Omron CX-Programmer project 新工程 (CX-Programmer 9.61)

# PLC ND自动入壳机: CJ2H CPU65-EIP
I/O table (CPU CJ2H-CPU65-EIP): rack 0 slot 0 CJ1W-ETN21(ETN21Mode); rack 0 slot 1 CJ1W-SCU21-V1; rack 0 slot 2 CJ1W-NC433; rack 0 slot 3 CJ1W-NC433; rack 0 slot 4 CJ1W-NC433; rack 0 slot 5 CJ1W-NC433; rack 0 slot 6 CJ1W-NC433; rack 0 slot 7 CJ1W-AD041-V1; rack 0 slot 11 CJ2B-EIP21; rack 1 slot 0 CJ1W-ID261; rack 1 slot 1 CJ1W-ID261; rack 1 slot 2 CJ1W-ID261; rack 1 slot 3 CJ1W-ID231; rack 1 slot 4 CJ1W-ID261; rack 1 slot 5 CJ1W-ID231; rack 1 slot 6 CJ1W-OD261; rack 1 slot 7 CJ1W-OD261; rack 1 slot 8 CJ1W-OD231; rack 1 slot 9 CJ1W-OD261

## Global symbols (name address type ; comment)
0.00 BOOL  ; RK_02 电芯进料机械手夹爪气缸夹紧位
0.01 BOOL  ; RK_02 电芯进料机械手夹爪气缸张开位
0.02 BOOL  ; RK_02 电芯进料机械手#1压紧气缸松开位
0.03 BOOL  ; RK_02 电芯进料机械手#2压紧气缸松开位
0.04 BOOL  ; RK_03 电芯上料机械手夹爪气缸夹紧位
0.05 BOOL  ; RK_03 电芯上料机械手夹爪气缸张开位
0.06 BOOL  ; RK_03 电芯上料机械手#1压紧气缸松开位
0.07 BOOL  ; RK_03 电芯上料机械手#2压紧气缸松开位
0.08 BOOL  ; RK_03 电芯上料升降气缸下降位
0.09 BOOL  ; RK_03 电芯上料升降气缸上升位
0.10 BOOL  ; RK_04 电芯除尘伸缩气缸缩回位
0.11 BOOL  ; RK_04 电芯除尘伸缩气缸伸出位
0.12 BOOL  ; RK_05 #1入壳滚轮夹紧气缸夹紧位
0.13 BOOL  ; RK_05 #1入壳滚轮夹紧气缸松开位
0.14 BOOL  ; RK_05 #1入壳铝壳定位平台伸缩气缸缩回位
0.15 BOOL  ; RK_05 #1入壳铝壳定位平台伸缩气缸伸出位
1000.00 BOOL  ; RK_01 U0_X 电芯来料Y轴待料位设定确认
1000.01 BOOL  ; RK_01 U0_X 电芯来料Y轴上料位设定确认
1000.02 BOOL  ; RK_01 U0_X 电芯来料Y轴扫码位设定确认
1000.03 BOOL  ; RK_01 U0_X 电芯来料Y轴下料位设定确认
1001.00 BOOL  ; RK_02 U0_Y 电芯进料X轴待料位设定确认
1001.01 BOOL  ; RK_02 U0_Y 电芯进料X轴取料位设定确认
1001.02 BOOL  ; RK_02 U0_Y 电芯进料X轴扫码OK放料位设定确认
1001.03 BOOL  ; RK_02 U0_Y 电芯进料X轴扫码NG放料位设定确认
1002.00 BOOL  ; RK_02 U0_Z 电芯进料Z轴待料位（扫码）设定确认
1002.01 BOOL  ; RK_02 U0_Z 电芯进料Z轴取料位设定确认
1002.02 BOOL  ; RK_02 U0_Z 电芯进料Z轴扫码OK放料位设定确认
1002.03 BOOL  ; RK_02 U0_Z 电芯进料Z轴扫码NG放料位设定确认
1002.04 BOOL  ; RK_02 U0_Z 电芯进料Z轴扫码位设定确认
1003.00 BOOL  ; RK_03 U0_U 电芯上料X轴待料位设定确认
1003.01 BOOL  ; RK_03 U0_U 电芯上料X轴取料位设定确认
1003.02 BOOL  ; RK_03 U0_U 电芯上料X轴#1入壳放料位设定确认
1003.03 BOOL  ; RK_03 U0_U 电芯上料X轴#2入壳放料位设定确认
1004.00 BOOL  ; RK_05 U2_X #1入壳Y轴待料位设定确认
1004.01 BOOL  ; RK_05 U2_X #1入壳Y轴滚轮压紧位设定确认
1004.02 BOOL  ; RK_05 U2_X #1入壳Y轴滚轮松开位设定确认
1004.03 BOOL  ; RK_05 U2_X #1入壳Y轴入壳位设定确认
1004.04 BOOL  ; RK_05 U2_X #1入壳Y轴电芯定位夹爪松开位设定确认
1005.00 BOOL  ; RK_05 U2_Y #2入壳Y轴待料位设定确认
1005.01 BOOL  ; RK_05 U2_Y #2入壳Y轴滚轮压紧位设定确认
1005.02 BOOL  ; RK_05 U2_Y #2入壳Y轴滚轮松开位设定确认
1005.03 BOOL  ; RK_05 U2_Y #2入壳Y轴入壳位设定确认
1005.04 BOOL  ; RK_05 U2_Y #2入壳Y轴电芯定位夹爪松开位设定确认
1006.00 BOOL  ; RK_12 U4_X 预焊上下料X轴待料位设定确认
1006.01 BOOL  ; RK_12 U4_X 预焊上下料X轴除尘取料位设定确认
1006.02 BOOL  ; RK_12 U4_X 预焊上下料X轴#1移载放料位设定确认
1006.03 BOOL  ; RK_12 U4_X 预焊上下料X轴#2移载放料位设定确认
1006.04 BOOL  ; RK_12 U4_X 预焊上下料X轴#1移载取料位设定确认
1006.05 BOOL  ; RK_12 U4_X 预焊上下料X轴#2移载取料位设定确认
1006.06 BOOL  ; RK_12 U4_X 预焊上下料X轴OK放料位设定确认
1006.07 BOOL  ; RK_12 U4_X 预焊上下料X轴#1NG放料位设定确认
1006.08 BOOL  ; RK_12 U4_X 预焊上下料X轴#2NG放料位设定确认
1007.00 BOOL  ; RK_12 U4_Y 预焊上料Z轴待料位设定确认
1007.01 BOOL  ; RK_12 U4_Y 预焊上料Z轴除尘取料位设定确认
1007.02 BOOL  ; RK_12 U4_Y 预焊上料Z轴#1移载放料位设定确认
1007.03 BOOL  ; RK_12 U4_Y 预焊上料Z轴#2移载放料位设定确认
1008.00 BOOL  ; RK_12 U4_Z 预焊下料Z轴待料位设定确认
1008.01 BOOL  ; RK_12 U4_Z 预焊下料Z轴#1移载取料位设定确认
1008.02 BOOL  ; RK_12 U4_Z 预焊下料Z轴#2移载取料位设定确认
1008.03 BOOL  ; RK_12 U4_Z 预焊下料Z轴OK放料位设定确认
1008.04 BOOL  ; RK_12 U4_Z 预焊下料Z轴#1NG放料位设定确认
1008.05 BOOL  ; RK_12 U4_Z 预焊下料Z轴#2NG放料位设定确认
1009.00 BOOL  ; RK_13 U4_U #1移载Y轴待料位设定确认
1009.01 BOOL  ; RK_13 U4_U #1移载Y轴取放料位设定确认
1009.02 BOOL  ; RK_13 U4_U #1移载Y轴压装位设定确认
1009.03 BOOL  ; RK_13 U4_U #1移载Y轴#1轮廓检测位设定确认
1009.04 BOOL  ; RK_13 U4_U #1移载Y轴#2轮廓检测位设定确认
1009.05 BOOL  ; RK_13 U4_U #1移载Y轴激光焊接位设定确认
100.00 BOOL  ; RK_02 电芯进料机械手夹爪气缸夹紧
100.01 BOOL  ; RK_02 电芯进料机械手夹爪气缸张开
100.02 BOOL  ; RK_02 电芯进料机械手压紧气缸伸出
100.03 BOOL  ; RK_02 电芯进料机械手压紧气缸缩回
100.04 BOOL  ; RK_03 电芯上料机械手夹爪气缸夹紧
100.05 BOOL  ; RK_03 电芯上料机械手夹爪气缸张开
100.06 BOOL  ; RK_03 电芯上料机械手压紧气缸伸出
100.07 BOOL  ; RK_03 电芯上料机械手压紧气缸缩回
100.08 BOOL  ; RK_03 电芯上料升降气缸下降
100.09 BOOL  ; RK_03 电芯上料升降气缸上升
100.10 BOOL  ; RK_04 电芯除尘伸缩气缸缩回
100.11 BOOL  ; RK_04 电芯除尘伸缩气缸伸出
100.12 BOOL  ; RK_05 #1入壳滚轮夹紧气缸伸出
100.13 BOOL  ; RK_05 #1入壳滚轮夹紧气缸缩回
100.14 BOOL  ; RK_05 #1入壳铝壳定位平台伸缩气缸缩回
100.15 BOOL  ; RK_05 #1入壳铝壳定位平台伸缩气缸伸出
1010.00 BOOL  ; RK_13 U6_X #2移载Y轴待料位设定确认
1010.01 BOOL  ; RK_13 U6_X #2移载Y轴取放料位设定确认
1010.02 BOOL  ; RK_13 U6_X #2移载Y轴压装位设定确认
1010.03 BOOL  ; RK_13 U6_X #2移载Y轴#1轮廓检测位设定确认
1010.04 BOOL  ; RK_13 U6_X #2移载Y轴#2轮廓检测位设定确认
1010.05 BOOL  ; RK_13 U6_X #2移载Y轴激光焊接位设定确认
1011.00 BOOL  ; RK_16 U6_Y 激光焊接X轴待机位设定确认
1011.01 BOOL  ; RK_16 U6_Y 激光焊接X轴#1移载焊接位设定确认
1011.02 BOOL  ; RK_16 U6_Y 激光焊接X轴#2移载焊接位设定确认
1012.00 BOOL  ; RK_16 U6_Z 激光焊接Z轴待机位设定确认
1012.01 BOOL  ; RK_16 U6_Z 激光焊接Z轴#1移载焊接位设定确认
1012.02 BOOL  ; RK_16 U6_Z 激光焊接Z轴#2移载焊接位设定确认
1013.00 BOOL  ; RK_06 U8_X 电池上下料X轴待机位设定确认
1013.01 BOOL  ; RK_06 U8_X 电池上下料X轴铝壳除尘取料位设定确认
1013.02 BOOL  ; RK_06 U8_X 电池上下料X轴#1入壳放料位设定确认
1013.03 BOOL  ; RK_06 U8_X 电池上下料X轴#2入壳放料位设定确认
1013.04 BOOL  ; RK_06 U8_X 电池上下料X轴#1入壳取料位设定确认
1013.05 BOOL  ; RK_06 U8_X 电池上下料X轴#2入壳取料位设定确认
1013.06 BOOL  ; RK_06 U8_X 电池上下料X轴#1Hipot检测放料位设定确认
1013.07 BOOL  ; RK_06 U8_X 电池上下料X轴#2Hipot检测放料位设定确认
1014.00 BOOL  ; RK_07 U8_Y 铝壳进料X轴等待位设定确认
1014.01 BOOL  ; RK_07 U8_Y 铝壳进料X轴取料位设定确认
1014.02 BOOL  ; RK_07 U8_Y 铝壳进料X轴放料位设定确认
1015.00 BOOL  ; RK_07 U8_Z 铝壳上料移载Y轴待料位设定确认
1015.01 BOOL  ; RK_07 U8_Z 铝壳上料移载Y轴#1铝壳上料位设定确认
1015.02 BOOL  ; RK_07 U8_Z 铝壳上料移载Y轴#2铝壳上料位设定确认
1015.03 BOOL  ; RK_07 U8_Z 铝壳上料移载Y轴#3铝壳托盘下料位设定确认
1015.04 BOOL  ; RK_07 U8_Z 铝壳上料移载Y轴铝壳取料位设定确认
1016.00 BOOL  ; RK_10 U8_U 电池除尘上料X轴待料位设定确认
1016.01 BOOL  ; RK_10 U8_U 电池除尘上料X轴#1Hipot检测取料位设定确认
1016.02 BOOL  ; RK_10 U8_U 电池除尘上料X轴#2Hipot检测取料位设定确认
1016.03 BOOL  ; RK_10 U8_U 电池除尘上料X轴Hipot OK放料位设定确认
1016.04 BOOL  ; RK_10 U8_U 电池除尘上料X轴Hipot NG放料位设定确认
101.00 BOOL  ; RK_05 #1入壳铝壳定位平台升降气缸上升
101.01 BOOL  ; RK_05 #1入壳铝壳定位平台升降气缸下降
101.02 BOOL  ; RK_05 #1入壳铝壳定位伸缩气缸缩回
101.03 BOOL  ; RK_05 #1入壳铝壳定位伸缩气缸伸出
101.04 BOOL  ; RK_05 #1入壳铝壳定位夹爪气缸夹紧
101.05 BOOL  ; RK_05 #1入壳铝壳定位夹爪气缸张开
101.06 BOOL  ; RK_05 #2入壳滚轮夹紧气缸伸出
101.07 BOOL  ; RK_05 #2入壳滚轮夹紧气缸缩回
101.08 BOOL  ; RK_05 #2入壳铝壳定位平台伸缩气缸缩回
101.09 BOOL  ; RK_05 #2入壳铝壳定位平台伸缩气缸伸出
101.10 BOOL  ; RK_05 #2入壳铝壳定位平台升降气缸上升
101.11 BOOL  ; RK_05 #2入壳铝壳定位平台升降气缸下降
101.12 BOOL  ; RK_05 #2入壳铝壳定位伸缩气缸缩回
101.13 BOOL  ; RK_05 #2入壳铝壳定位伸缩气缸伸出
101.14 BOOL  ; RK_05 #2入壳铝壳定位夹爪气缸夹紧
101.15 BOOL  ; RK_05 #2入壳铝壳定位夹爪气缸张开
102.00 BOOL  ; RK_01 U0_X 电芯来料Y轴报警复位
102.01 BOOL  ; RK_01 U0_X 电芯来料Y轴使能
102.02 BOOL  ; RK_02 U0_Y 电芯进料X轴报警复位
102.03 BOOL  ; RK_02 U0_Y 电芯进料X轴使能
102.04 BOOL  ; RK_02 U0_Z 电芯进料Z轴报警复位
102.05 BOOL  ; RK_02 U0_Z 电芯进料Z轴使能
102.06 BOOL  ; RK_03 U0_U 电芯上料X轴报警复位
102.07 BOOL  ; RK_03 U0_U 电芯上料X轴使能
102.08 BOOL  ; RK_05 U2_X #1入壳Y轴报警复位
102.09 BOOL  ; RK_05 U2_X #1入壳Y轴使能
102.10 BOOL  ; RK_05 U2_Y #2入壳Y轴报警复位
102.11 BOOL  ; RK_05 U2_Y #2入壳Y轴使能
102.12 BOOL  ; RK_02 电芯进料Z轴刹车使能
102.13 BOOL  ; RK_05 #1入壳定位陶瓷棒夹紧气缸伸出
102.14 BOOL  ; RK_05 #1入壳定位陶瓷棒夹紧气缸缩回
102.15 BOOL  ; RK_05 #2入壳定位陶瓷棒夹紧气缸伸出
103.00 BOOL  ; RK_05 #2入壳定位陶瓷棒夹紧气缸缩回
103.01 BOOL  ; RK_04 电芯除尘吹气阀开
103.02 BOOL  ; RK_02 扫码NG拉带启动
103.03 BOOL  ; RK_05 #1入壳吸盘立真空
103.04 BOOL  ; RK_05 #2入壳吸盘立真空
103.05 BOOL  ; RK_05 #1入壳吸盘伸缩气缸伸出
103.06 BOOL  ; RK_05 #1入壳吸盘伸缩气缸缩回
103.07 BOOL  ; RK_05 #2入壳吸盘伸缩气缸伸出
103.08 BOOL  ; RK_05 #2入壳吸盘伸缩气缸缩回
103.09 BOOL  ; 前端设备对接输出信号（公共）
103.10 BOOL  ; 后端设备对接输出信号（公共）
103.11 BOOL  ; RK_05 #1入壳电芯定位夹爪气缸伸出
103.12 BOOL  ; RK_05 #1入壳电芯定位夹爪气缸缩回
103.13 BOOL  ; RK_05 #2入壳电芯定位夹爪气缸伸出
103.14 BOOL  ; RK_05 #2入壳电芯定位夹爪气缸缩回
103.15 BOOL  ; 0
104.00 BOOL  ; 0
104.01 BOOL  ; 0
104.02 BOOL  ; 0
104.03 BOOL  ; 0
104.04 BOOL  ; 0
104.05 BOOL  ; 0
104.06 BOOL  ; 0
104.07 BOOL  ; 0
104.08 BOOL  ; 0
104.09 BOOL  ; 0
104.10 BOOL  ; 0
104.11 BOOL  ; 0
104.12 BOOL  ; 0
104.13 BOOL  ; 0
104.14 BOOL  ; 0
104.15 BOOL  ; 0
105.00 BOOL  ; 0
105.01 BOOL  ; 0
105.02 BOOL  ; 0
105.03 BOOL  ; 0
105.04 BOOL  ; 0
105.05 BOOL  ; 0
105.06 BOOL  ; 0
105.07 BOOL  ; 0
105.08 BOOL  ; 0
105.09 BOOL  ; 0
105.10 BOOL  ; 0
105.11 BOOL  ; 0
105.12 BOOL  ; 0
105.13 BOOL  ; 0
105.14 BOOL  ; 0
105.15 BOOL  ; 0
106.00 BOOL  ; 0
106.01 BOOL  ; 0
106.02 BOOL  ; 0
106.03 BOOL  ; 0
106.04 BOOL  ; 0
106.05 BOOL  ; 0
106.06 BOOL  ; 0
106.07 BOOL  ; 0
106.08 BOOL  ; 0
106.09 BOOL  ; 0
106.10 BOOL  ; 0
106.11 BOOL  ; 0
106.12 BOOL  ; 0
106.13 BOOL  ; 0
106.14 BOOL  ; 0
106.15 BOOL  ; 0
107.00 BOOL  ; 0
107.01 BOOL  ; 0
107.02 BOOL  ; 0
107.03 BOOL  ; 0
107.04 BOOL  ; 0
107.05 BOOL  ; 0
107.06 BOOL  ; 0
107.07 BOOL  ; 0
107.08 BOOL  ; 0
107.09 BOOL  ; 0
107.10 BOOL  ; 0
107.11 BOOL  ; 0
107.12 BOOL  ; 0
107.13 BOOL  ; 0
107.14 BOOL  ; 0
107.15 BOOL  ; 0
108.00 BOOL  ; RK_11 电池除尘旋转伸缩气缸缩回
108.01 BOOL  ; RK_11 电池除尘旋转伸缩气缸伸出
108.02 BOOL  ; RK_11 电池除尘伸缩气缸伸出
108.03 BOOL  ; RK_11 电池除尘伸缩气缸缩回
108.04 BOOL  ; RK_11 电池除尘夹爪气缸夹紧
108.05 BOOL  ; RK_11 电池除尘夹爪气缸张开
108.06 BOOL  ; RK_12 预焊上料机械手夹爪气缸夹紧
108.07 BOOL  ; RK_12 预焊上料机械手夹爪气缸张开
108.08 BOOL  ; RK_12 预焊下料机械手夹爪气缸夹紧
108.09 BOOL  ; RK_12 预焊下料机械手夹爪气缸张开
108.10 BOOL  ; RK_13 #1移载升降气缸上升
108.11 BOOL  ; RK_13 #1移载升降气缸下降
108.12 BOOL  ; RK_13 #1移载定位#1伸缩气缸缩回
108.13 BOOL  ; RK_13 #1移载定位#1伸缩气缸伸出
108.14 BOOL  ; RK_13 #1移载定位#2伸缩气缸缩回
108.15 BOOL  ; RK_13 #1移载定位#2伸缩气缸伸出
109.00 BOOL  ; RK_13 #1移载导向#1伸缩气缸伸出
109.01 BOOL  ; RK_13 #1移载导向#1伸缩气缸缩回
109.02 BOOL  ; 扫码阻挡#1伸出输出
109.03 BOOL  ; 扫码阻挡#1缩回输出
109.04 BOOL  ; RK_13 #1移载左右定位伸缩气缸伸出
109.05 BOOL  ; RK_13 #1移载左右定位伸缩气缸缩回
109.06 BOOL  ; RK_13 #2移载升降气缸上升
109.07 BOOL  ; RK_13 #2移载升降气缸下降
109.08 BOOL  ; RK_13 #2移载定位#1伸缩气缸缩回
109.09 BOOL  ; RK_13 #2移载定位#1伸缩气缸伸出
109.10 BOOL  ; 扫码阻挡#2伸出输出
109.11 BOOL  ; 扫码阻挡#2缩回输出
109.12 BOOL  ; RK_13 #2移载导向#1伸缩气缸伸出
109.13 BOOL  ; RK_13 #2移载导向#1伸缩气缸缩回
109.14 BOOL  ; RK_13 #2移载导向#2伸缩气缸伸出
109.15 BOOL  ; RK_13 #2移载导向#2伸缩气缸缩回
10.00 BOOL  ; RK_13 #2移载左右定位伸缩气缸伸出位
10.01 BOOL  ; RK_13 #2移载左右定位伸缩气缸缩回位
10.02 BOOL  ; RK_14 #1压装升降气缸下降位
10.03 BOOL  ; RK_14 #1压装升降气缸上升位
10.04 BOOL  ; RK_14 #1压装#1吸盘升降气缸下降位
10.05 BOOL  ; RK_14 #1压装#1吸盘升降气缸上升位
10.06 BOOL  ; RK_14 #1压装#2吸盘升降气缸下降位
10.07 BOOL  ; RK_14 #1压装#2吸盘升降气缸上升位
10.08 BOOL  ; RK_14 #2压装升降气缸下降位
10.09 BOOL  ; RK_14 #2压装升降气缸上升位
10.10 BOOL  ; RK_14 #2压装#1吸盘升降气缸下降位
10.11 BOOL  ; RK_14 #2压装#1吸盘升降气缸上升位
10.12 BOOL  ; RK_14 #2压装#2吸盘升降气缸下降位
10.13 BOOL  ; RK_14 #2压装#2吸盘升降气缸上升位
10.14 BOOL  ; RK_15 轮廓检测#1伸缩气缸伸出位
10.15 BOOL  ; RK_15 轮廓检测#1伸缩气缸缩回位
110.00 BOOL  ; RK_13 #2移载左右定位伸缩气缸伸出
110.01 BOOL  ; RK_13 #2移载左右定位伸缩气缸缩回
110.02 BOOL  ; RK_14 #1压装升降气缸下降
110.03 BOOL  ; RK_14 #1压装升降气缸上升
110.04 BOOL  ; RK_14 #1压装#1吸盘升降气缸下降
110.05 BOOL  ; RK_14 #1压装#1吸盘升降气缸上升
110.06 BOOL  ; RK_14 #1压装#2吸盘升降气缸下降
110.07 BOOL  ; RK_14 #1压装#2吸盘升降气缸上升
110.08 BOOL  ; RK_14 #2压装升降气缸下降
110.09 BOOL  ; RK_14 #2压装升降气缸上升
110.10 BOOL  ; RK_14 #2压装#1吸盘升降气缸下降
110.11 BOOL  ; RK_14 #2压装#1吸盘升降气缸上升
110.12 BOOL  ; RK_14 #2压装#2吸盘升降气缸下降
110.13 BOOL  ; RK_14 #2压装#2吸盘升降气缸上升
110.14 BOOL  ; RK_15 轮廓检测#1伸缩气缸伸出
110.15 BOOL  ; RK_15 轮廓检测#1伸缩气缸缩回
111.00 BOOL  ; RK_15 轮廓检测#2伸缩气缸伸出
111.01 BOOL  ; RK_15 轮廓检测#2伸缩气缸缩回
111.02 BOOL  ; RK_12 轮廓检测NG拨料气缸伸出
111.03 BOOL  ; RK_12 轮廓检测NG拨料气缸缩回
111.04 BOOL  ; RK_11 电池除尘吹气阀开
111.05 BOOL  ; 0
111.06 BOOL  ; 0
111.07 BOOL  ; RK_16 激光焊接触发
111.08 BOOL  ; RK_16 PLC急停输出到激光设备（0=PLC急停输出，1=PLC无急停输出）
111.09 BOOL  ; RK_16 #1移载激光焊任务选择#2
111.10 BOOL  ; RK_16 移载激光焊任务选择#1
111.11 BOOL  ; RK_16 集尘器启动
111.12 BOOL  ; 0
111.13 BOOL  ; 0
111.14 BOOL  ; RK_14 #1压装吸盘立真空
111.15 BOOL  ; RK_14 #2压装吸盘立真空
112.00 BOOL  ; RK_12 U4_X 预焊上下料X轴报警复位
112.01 BOOL  ; RK_12 U4_X 预焊上下料X轴使能
112.02 BOOL  ; RK_12 U4_Y 预焊上料Z轴报警复位
112.03 BOOL  ; RK_12 U4_Y 预焊上料Z轴使能
112.04 BOOL  ; RK_12 U4_Z 预焊下料Z轴报警复位
112.05 BOOL  ; RK_12 U4_Z 预焊下料Z轴使能
112.06 BOOL  ; RK_13 U4_U #1移载Y轴报警复位
112.07 BOOL  ; RK_13 U4_U #1移载Y轴使能
112.08 BOOL  ; RK_13 U6_X #2移载Y轴报警复位
112.09 BOOL  ; RK_13 U6_X #2移载Y轴使能
112.10 BOOL  ; RK_16 U6_Y 激光焊接X轴报警复位
112.11 BOOL  ; RK_16 U6_Y 激光焊接X轴使能
112.12 BOOL  ; RK_16 U6_Z 激光焊接Z轴报警复位
112.13 BOOL  ; RK_16 U6_Z 激光焊接Z轴使能
112.14 BOOL  ; RK_12 预焊上料Z轴刹车使能
112.15 BOOL  ; RK_12 预焊下料Z轴刹车使能
113.00 BOOL  ; RK_16 激光焊接Z轴刹车使能
113.01 BOOL  ; 0
113.02 BOOL  ; 0
113.03 BOOL  ; 0
113.04 BOOL  ; 0
113.05 BOOL  ; RK_07 OK出料拉带启动
113.06 BOOL  ; 0
113.07 BOOL  ; 0
113.08 BOOL  ; 0
113.09 BOOL  ; RK_07 #1铝壳上料电机刹车使能
113.10 BOOL  ; RK_07 #2铝壳上料电机刹车使能
113.11 BOOL  ; RK_07 #3托盘下料电机刹车使能
113.12 BOOL  ; 三色灯_红（公共）
113.13 BOOL  ; 三色灯_绿（公共）
113.14 BOOL  ; 三色灯_黄（公共）
113.15 BOOL  ; 蜂鸣器（公共）
114.00 BOOL  ; RK_06 铝壳上料升降气缸下降
114.01 BOOL  ; RK_06 铝壳上料升降气缸上升
114.02 BOOL  ; RK_06 电池下料升降气缸下降
114.03 BOOL  ; RK_06 电池下料升降气缸上升
114.04 BOOL  ; RK_06 铝壳上料夹爪气缸夹紧
114.05 BOOL  ; RK_06 铝壳上料夹爪气缸张开
114.06 BOOL  ; RK_06 电池下料夹爪气缸夹紧
114.07 BOOL  ; RK_06 电池下料夹爪气缸张开
114.08 BOOL  ; RK_07 #1铝壳上料车定位升降气缸上升
114.09 BOOL  ; RK_07 #1铝壳上料车定位升降气缸下降
114.10 BOOL  ; RK_07 #2铝壳上料车定位升降气缸上升
114.11 BOOL  ; RK_07 #2铝壳上料车定位升降气缸下降
114.12 BOOL  ; RK_07 #3托盘下料车定位升降气缸上升
114.13 BOOL  ; RK_07 #3托盘下料车定位升降气缸下降
114.14 BOOL  ; RK_07 铝壳进料机械手升降气缸下降
114.15 BOOL  ; RK_07 铝壳进料机械手升降气缸上升
115.00 BOOL  ; RK_08 铝壳除尘旋转伸缩气缸缩回
115.01 BOOL  ; RK_08 铝壳除尘旋转伸缩气缸伸出
115.02 BOOL  ; RK_08 铝壳除尘伸缩气缸伸出
115.03 BOOL  ; RK_08 铝壳除尘伸缩气缸缩回
115.04 BOOL  ; RK_08 铝壳除尘夹爪气缸夹紧
115.05 BOOL  ; RK_08 铝壳除尘夹爪气缸张开
115.06 BOOL  ; RK_09 #1Hipot测试旋转伸缩气缸伸出
115.07 BOOL  ; RK_09 #1Hipot测试旋转伸缩气缸缩回
115.08 BOOL  ; RK_09 #1Hipot测试平台伸缩气缸缩回
115.09 BOOL  ; RK_09 #1Hipot测试平台伸缩气缸伸出
115.10 BOOL  ; RK_09 #1Hipot测试伸缩气缸伸出
115.11 BOOL  ; RK_09 #1Hipot测试伸缩气缸缩回
115.12 BOOL  ; RK_09 #2Hipot测试旋转伸缩气缸伸出
115.13 BOOL  ; RK_09 #2Hipot测试旋转伸缩气缸缩回
115.14 BOOL  ; RK_09 #2Hipot测试平台伸缩气缸缩回
115.15 BOOL  ; RK_09 #2Hipot测试平台伸缩气缸伸出
116.00 BOOL  ; RK_09 #2Hipot测试伸缩气缸伸出
116.01 BOOL  ; RK_09 #2Hipot测试伸缩气缸缩回
116.02 BOOL  ; RK_10 电池除尘上料机械手升降气缸下降
116.03 BOOL  ; RK_10 电池除尘上料机械手升降气缸上升
116.04 BOOL  ; RK_10 电池除尘上料机械手夹爪气缸夹紧
116.05 BOOL  ; RK_10 电池除尘上料机械手夹爪气缸张开
116.06 BOOL  ; RK_06 U8_X 电池上下料X轴报警复位
116.07 BOOL  ; RK_06 U8_X 电池上下料X轴使能
116.08 BOOL  ; RK_07 U8_Y 铝壳进料X轴报警复位
116.09 BOOL  ; RK_07 U8_Y 铝壳进料X轴使能
116.10 BOOL  ; RK_07 U8_Z 铝壳上料移载Y轴报警复位
116.11 BOOL  ; RK_07 U8_Z 铝壳上料移载Y轴使能
116.12 BOOL  ; RK_10 U8_U 电池除尘上料X轴报警复位
116.13 BOOL  ; RK_10 U8_U 电池除尘上料X轴使能
116.14 BOOL  ; RK_09 Hipot测试仪远程使能（取消）
116.15 BOOL  ; RK_07 #1铝壳上料启动指示
117.00 BOOL  ; RK_07 #2铝壳上料启动指示
117.01 BOOL  ; RK_07 #3托盘下料启动指示
117.02 BOOL  ; RK_07 铝壳上料移载吸盘立真空
117.03 BOOL  ; RK_07 铝壳进料吸盘立真空
117.04 BOOL  ; RK_07 #1铝壳上料电机正转
117.05 BOOL  ; RK_07 #1铝壳上料电机反转
117.06 BOOL  ; RK_10 Hipot检测NG拉带启动
117.07 BOOL  ; RK_08 铝壳除尘吹气阀开
117.08 BOOL  ; 0
117.09 BOOL  ; RK_07 #2铝壳上料电机正转
117.10 BOOL  ; RK_07 #2铝壳上料电机反转
117.11 BOOL  ; 启动指示_绿（公共）
117.12 BOOL  ; 停止指示_红（公共）
117.13 BOOL  ; 复位指示_黄（公共）
117.14 BOOL  ; RK_07 #3托盘下料电机正转
117.15 BOOL  ; RK_07 #3托盘下料电机反转
118.00 BOOL  ; 0
118.01 BOOL  ; 0
118.02 BOOL  ; 0
118.03 BOOL  ; 0
118.04 BOOL  ; 0
118.05 BOOL  ; 0
118.06 BOOL  ; 0
118.07 BOOL  ; 0
118.08 BOOL  ; 0
118.09 BOOL  ; 0
118.10 BOOL  ; 0
118.11 BOOL  ; 0
118.12 BOOL  ; 0
118.13 BOOL  ; 0
118.14 BOOL  ; 0
118.15 BOOL  ; 0
119.00 BOOL  ; 0
119.01 BOOL  ; 0
119.02 BOOL  ; 0
119.03 BOOL  ; 0
119.04 BOOL  ; 0
119.05 BOOL  ; 0
119.06 BOOL  ; 0
119.07 BOOL  ; 0
119.08 BOOL  ; 0
119.09 BOOL  ; 0
119.10 BOOL  ; 0
119.11 BOOL  ; 0
119.12 BOOL  ; 0
119.13 BOOL  ; 0
119.14 BOOL  ; 0
119.15 BOOL  ; 0
11.00 BOOL  ; RK_15 轮廓检测#2伸缩气缸伸出位
11.01 BOOL  ; RK_15 轮廓检测#2伸缩气缸缩回位
11.02 BOOL  ; RK_12 轮廓检测NG拨料气缸伸出位
11.03 BOOL  ; RK_12 轮廓检测NG拨料气缸缩回位
11.04 BOOL  ; RK_11 电池除尘有料感应
11.05 BOOL  ; RK_12 预焊上料机械手夹爪柔性报警
11.06 BOOL  ; RK_12 预焊下料机械手夹爪柔性报警
11.07 BOOL  ; RK_16 激光焊接完成信号
11.08 BOOL  ; RK_16 激光焊机故障信号
11.09 BOOL  ; RK_13 #1移载电池顶盖超高检测
11.10 BOOL  ; RK_16 激光焊机急停信号
11.11 BOOL  ; RK_13 #2移载电池顶盖超高检测
11.12 BOOL  ; RK_13 #1移载有料感应
11.13 BOOL  ; RK_13 #2移载有料感应
11.14 BOOL  ; RK_14 #1压装吸盘真空
11.15 BOOL  ; RK_14 #2压装吸盘真空
121.04 BOOL  ; RK_11 电池除尘吹气阀关
121.14 BOOL  ; RK_14 #1压装吸盘破真空
121.15 BOOL  ; RK_14 #2压装吸盘破真空
123.01 BOOL  ; RK_04 电芯除尘吹气阀关
123.02 BOOL  ; RK_02 扫码NG拉带停止
123.03 BOOL  ; RK_05 #1入壳吸盘破真空
123.04 BOOL  ; RK_05 #2入壳吸盘破真空
127.02 BOOL  ; RK_07 铝壳上料移载吸盘破真空
127.03 BOOL  ; RK_07 铝壳进料吸盘破真空
127.04 BOOL  ; RK_07 #1铝壳上料电机停止
127.06 BOOL  ; RK_10 Hipot检测NG拉带停止
127.07 BOOL  ; RK_08 铝壳除尘吹气阀关
127.09 BOOL  ; RK_07 #2铝壳上料电机停止
127.14 BOOL  ; RK_07 #3托盘下料电机停止
12.00 BOOL  ; RK_12 U4_X 预焊上下料X轴报警信号
12.01 BOOL  ; RK_12 U4_X 预焊上下料X轴准备好了信号
12.02 BOOL  ; RK_12 U4_Y 预焊上料Z轴报警信号
12.03 BOOL  ; RK_12 U4_Y 预焊上料Z轴准备好了信号
12.04 BOOL  ; RK_12 U4_Z 预焊下料Z轴报警信号
12.05 BOOL  ; RK_12 U4_Z 预焊下料Z轴准备好了信号
12.06 BOOL  ; RK_13 U4_U #1移载Y轴报警信号
12.07 BOOL  ; RK_13 U4_U #1移载Y轴准备好了信号
12.08 BOOL  ; RK_13 U6_X #2移载Y轴报警信号
12.09 BOOL  ; RK_13 U6_X #2移载Y轴准备好了信号
12.10 BOOL  ; RK_16 U6_Y 激光焊接X轴报警信号
12.11 BOOL  ; RK_16 U6_Y 激光焊接X轴准备好了信号
12.12 BOOL  ; RK_16 U6_Z 激光焊接Z轴报警信号
12.13 BOOL  ; RK_16 U6_Z 激光焊接Z轴准备好了信号
13.01 BOOL  ; RK_12 轮廓检测NG料槽#1有料感应
13.02 BOOL  ; RK_12 轮廓检测NG料槽#1料满感应
13.03 BOOL  ; RK_12 轮廓检测NG料槽#2有料感应
13.04 BOOL  ; RK_12 轮廓检测NG料槽#2料满感应
13.05 BOOL  ; RK_12 OK出料拉带放料位有料感应#1
13.06 BOOL  ; RK_12 OK出料拉带放料位有料感应#2
13.07 BOOL  ; RK_12 OK出料拉带出料位有料感应
14.00 BOOL  ; RK_06 铝壳上料升降气缸下降位
14.01 BOOL  ; RK_06 铝壳上料升降气缸上升位
14.02 BOOL  ; RK_06 电池下料升降气缸下降位
14.03 BOOL  ; RK_06 电池下料升降气缸上升位
14.04 BOOL  ; RK_06 铝壳上料夹爪气缸夹紧位
14.05 BOOL  ; RK_06 铝壳上料夹爪气缸张开位
14.06 BOOL  ; RK_06 电池下料夹爪气缸夹紧位
14.07 BOOL  ; RK_06 电池下料夹爪气缸张开位
14.08 BOOL  ; RK_07 #1铝壳上料车定位升降气缸上升位
14.09 BOOL  ; RK_07 #1铝壳上料车定位升降气缸下降位
14.10 BOOL  ; RK_07 #2铝壳上料车定位升降气缸上升位
14.11 BOOL  ; RK_07 #2铝壳上料车定位升降气缸下降位
14.12 BOOL  ; RK_07 #3托盘下料车定位升降气缸上升位
14.13 BOOL  ; RK_07 #3托盘下料车定位升降气缸下降位
14.14 BOOL  ; RK_07 铝壳进料机械手升降气缸下降位
14.15 BOOL  ; RK_07 铝壳进料机械手升降气缸上升位
150.00 BOOL  ; RK_01 U0_X 电芯来料Y轴待料位触发
150.01 BOOL  ; RK_01 U0_X 电芯来料Y轴上料位触发
150.02 BOOL  ; RK_01 U0_X 电芯来料Y轴扫码位触发
150.03 BOOL  ; RK_01 U0_X 电芯来料Y轴下料位触发
150.10 BOOL  ; RK_01 U0_X 电芯来料Y轴回原点触发
150.11 BOOL  ; RK_01 U0_X 电芯来料Y轴JOG+
150.12 BOOL  ; RK_01 U0_X 电芯来料Y轴JOG-
150.13 BOOL  ; RK_01 U0_X 电芯来料Y轴JOG高速
150.14 BOOL  ; RK_01 U0_X 电芯来料Y轴JOG低速
150.15 BOOL  ; 备用
151.00 BOOL  ; RK_02 U0_Y 电芯进料X轴待料位触发
151.01 BOOL  ; RK_02 U0_Y 电芯进料X轴取料位触发
151.02 BOOL  ; RK_02 U0_Y 电芯进料X轴扫码OK放料位触发
151.03 BOOL  ; RK_02 U0_Y 电芯进料X轴扫码NG放料位触发
151.10 BOOL  ; RK_02 U0_Y 电芯进料X轴回原点触发
151.11 BOOL  ; RK_02 U0_Y 电芯进料X轴JOG+
151.12 BOOL  ; RK_02 U0_Y 电芯进料X轴JOG-
151.13 BOOL  ; RK_02 U0_Y 电芯进料X轴JOG高速
151.14 BOOL  ; RK_02 U0_Y 电芯进料X轴JOG低速
151.15 BOOL  ; 备用
152.00 BOOL  ; RK_02 U0_Z 电芯进料Z轴待料位（扫码）触发
152.01 BOOL  ; RK_02 U0_Z 电芯进料Z轴取料位触发
152.02 BOOL  ; RK_02 U0_Z 电芯进料Z轴扫码OK放料位触发
152.03 BOOL  ; RK_02 U0_Z 电芯进料Z轴扫码NG放料位触发
152.04 BOOL  ; RK_02 U0_Z 电芯进料Z轴扫码位触发
152.10 BOOL  ; RK_02 U0_Z 电芯进料Z轴回原点触发
152.11 BOOL  ; RK_02 U0_Z 电芯进料Z轴JOG+
152.12 BOOL  ; RK_02 U0_Z 电芯进料Z轴JOG-
152.13 BOOL  ; RK_02 U0_Z 电芯进料Z轴JOG高速
152.14 BOOL  ; RK_02 U0_Z 电芯进料Z轴JOG低速
152.15 BOOL  ; 备用
153.00 BOOL  ; RK_03 U0_U 电芯上料X轴待料位触发
153.01 BOOL  ; RK_03 U0_U 电芯上料X轴取料位触发
153.02 BOOL  ; RK_03 U0_U 电芯上料X轴#1入壳放料位触发
153.03 BOOL  ; RK_03 U0_U 电芯上料X轴#2入壳放料位触发
153.10 BOOL  ; RK_03 U0_U 电芯上料X轴回原点触发
153.11 BOOL  ; RK_03 U0_U 电芯上料X轴JOG+
153.12 BOOL  ; RK_03 U0_U 电芯上料X轴JOG-
153.13 BOOL  ; RK_03 U0_U 电芯上料X轴JOG高速
153.14 BOOL  ; RK_03 U0_U 电芯上料X轴JOG低速
153.15 BOOL  ; 备用
154.00 BOOL  ; RK_05 U2_X #1入壳Y轴待料位触发
154.01 BOOL  ; RK_05 U2_X #1入壳Y轴滚轮压紧位触发
154.02 BOOL  ; RK_05 U2_X #1入壳Y轴滚轮松开位触发
154.03 BOOL  ; RK_05 U2_X #1入壳Y轴入壳位触发
154.04 BOOL  ; RK_05 U2_X #1入壳Y轴电芯定位夹爪松开位触发
154.10 BOOL  ; RK_05 U2_X #1入壳Y轴回原点触发
154.11 BOOL  ; RK_05 U2_X #1入壳Y轴JOG+
154.12 BOOL  ; RK_05 U2_X #1入壳Y轴JOG-
154.13 BOOL  ; RK_05 U2_X #1入壳Y轴JOG高速
154.14 BOOL  ; RK_05 U2_X #1入壳Y轴JOG低速
154.15 BOOL  ; 备用
1550.00 BOOL  ; SCU21_2 P1 Wait Release Switch
1550.01 BOOL  ; SCU21_2 P1 Continuous Trace Switch
1550.02 BOOL  ; SCU21_2 P1 One-shot Trace Switch
1550.03 BOOL  ; SCU21_2 P1 Abort Switch
1550.04 BOOL  ; SCU21_2 P1 Serial Gateway Prohibited Switch
1550.05 BOOL  ; SCU21_2 P1 Reserved
1550.06 BOOL  ; SCU21_2 P1 Loopback Test Switch
1550.07 BOOL  ; SCU21_2 P1 Reserved
1550.08 BOOL  ; SCU21_2 P2 Wait Release Switch
1550.09 BOOL  ; SCU21_2 P2 Continuous Trace Switch
1550.10 BOOL  ; SCU21_2 P2 One-shot Trace Switch
1550.11 BOOL  ; SCU21_2 P2 Abort Switch
1550.12 BOOL  ; SCU21_2 P2 Serial Gateway Prohibited Switch
1550.13 BOOL  ; SCU21_2 P2 Reserved
1550.14 BOOL  ; SCU21_2 P2 Loopback Test Switch
1550.15 BOOL  ; SCU21_2 P2 Reserved
1551.00 BOOL  ; SCU21_2 Protocol Data Error
1551.01 BOOL  ; SCU21_2 Error Log EEPROM Error
1551.02 BOOL  ; SCU21_2 Reserved
1551.03 BOOL  ; SCU21_2 Reserved
1551.04 BOOL  ; SCU21_2 Reserved
1551.05 BOOL  ; SCU21_2 Reserved
1551.06 BOOL  ; SCU21_2 Reserved
1551.07 BOOL  ; SCU21_2 Reserved
1551.08 BOOL  ; SCU21_2 Reserved
1551.09 BOOL  ; SCU21_2 Reserved
1551.10 BOOL  ; SCU21_2 Reserved
1551.11 BOOL  ; SCU21_2 Reserved
1551.12 BOOL  ; SCU21_2 Reserved
1551.13 BOOL  ; SCU21_2 Reserved
1551.14 BOOL  ; SCU21_2 Reserved
1551.15 BOOL  ; SCU21_2 Reserved
1552.00 BOOL  ; SCU21_2 Reserved
1552.01 BOOL  ; SCU21_2 Reserved
1552.02 BOOL  ; SCU21_2 Reserved
1552.03 BOOL  ; SCU21_2 Reserved
1552.04 BOOL  ; SCU21_2 Reserved
1552.05 BOOL  ; SCU21_2 Reserved
1552.06 BOOL  ; SCU21_2 Reserved
1552.07 BOOL  ; SCU21_2 Reserved
1552.08 BOOL  ; SCU21_2 Reserved
1552.09 BOOL  ; SCU21_2 Reserved
1552.10 BOOL  ; SCU21_2 Reserved
1552.11 BOOL  ; SCU21_2 Reserved
1552.12 BOOL  ; SCU21_2 Reserved
1552.13 BOOL  ; SCU21_2 Reserved
1552.14 BOOL  ; SCU21_2 Reserved
1552.15 BOOL  ; SCU21_2 Reserved
1553.00 BOOL  ; SCU21_2 Reserved
1553.01 BOOL  ; SCU21_2 Reserved
1553.02 BOOL  ; SCU21_2 Reserved
1553.03 BOOL  ; SCU21_2 Reserved
1553.04 BOOL  ; SCU21_2 Reserved
1553.05 BOOL  ; SCU21_2 Reserved
1553.06 BOOL  ; SCU21_2 Reserved
1553.07 BOOL  ; SCU21_2 Reserved
1553.08 BOOL  ; SCU21_2 Reserved
1553.09 BOOL  ; SCU21_2 Reserved
1553.10 BOOL  ; SCU21_2 Reserved
1553.11 BOOL  ; SCU21_2 Reserved
1553.12 BOOL  ; SCU21_2 Reserved
1553.13 BOOL  ; SCU21_2 Reserved
1553.14 BOOL  ; SCU21_2 Reserved
1553.15 BOOL  ; SCU21_2 Reserved
1554.00 BOOL  ; SCU21_2 Reserved
1554.01 BOOL  ; SCU21_2 Reserved
1554.02 BOOL  ; SCU21_2 Reserved
1554.03 BOOL  ; SCU21_2 Reserved
1554.04 BOOL  ; SCU21_2 Reserved
1554.05 BOOL  ; SCU21_2 Reserved
1554.06 BOOL  ; SCU21_2 Reserved
1554.07 BOOL  ; SCU21_2 Reserved
1554.08 BOOL  ; SCU21_2 Reserved
1554.09 BOOL  ; SCU21_2 Reserved
1554.10 BOOL  ; SCU21_2 Reserved
1554.11 BOOL  ; SCU21_2 Reserved
1554.12 BOOL  ; SCU21_2 Reserved
1554.13 BOOL  ; SCU21_2 Reserved
1554.14 BOOL  ; SCU21_2 Reserved
1554.15 BOOL  ; SCU21_2 Reserved
1555.00 BOOL  ; SCU21_2 P1 Parity: Even/Odd
1555.01 BOOL  ; SCU21_2 P1 Parity: Yes/No
1555.02 BOOL  ; SCU21_2 P1 Stop bits: 1 or 2 bits
1555.03 BOOL  ; SCU21_2 P1 Data length: 7 or 8 bits
1555.04 BOOL  ; SCU21_2 P1 Start bits: Always 1
1555.05 BOOL  ; SCU21_2 P1 Reserved
1555.06 BOOL  ; SCU21_2 P1 Reserved
1555.07 BOOL  ; SCU21_2 P1 Reserved
1555.08 BOOL  ; SCU21_2 P1 Baud rate
1555.09 BOOL  ; SCU21_2 P1 Baud rate
1555.10 BOOL  ; SCU21_2 P1 Baud rate
1555.11 BOOL  ; SCU21_2 P1 Baud rate
1555.12 BOOL  ; SCU21_2 P1 Serial communications mode
1555.13 BOOL  ; SCU21_2 P1 Serial communications mode
1555.14 BOOL  ; SCU21_2 P1 Serial communications mode
1555.15 BOOL  ; SCU21_2 P1 Serial communications mode
1556.00 BOOL  ; SCU21_2 P1 1:  operating; 0:  Stopped
1556.01 BOOL  ; SCU21_2 P1 1: System Setup error; 0: System Setup normal
1556.02 BOOL  ; SCU21_2 P1 Reserved
1556.03 BOOL  ; SCU21_2 P1 Reserved
1556.04 BOOL  ; SCU21_2 P1 Reserved
1556.05 BOOL  ; SCU21_2 P1 Reserved
1556.06 BOOL  ; SCU21_2 P1 Reserved
1556.07 BOOL  ; SCU21_2 P1 Reserved
1556.08 BOOL  ; SCU21_2 P1 Reserved
1556.09 BOOL  ; SCU21_2 P1 Reserved
1556.10 BOOL  ; SCU21_2 P1 Reserved
1556.11 BOOL  ; SCU21_2 P1 Reserved
1556.12 BOOL  ; SCU21_2 P1 Reserved
1556.13 BOOL  ; SCU21_2 P1 Terminating resistance
1556.14 BOOL  ; SCU21_2 P1 Hardware settings
1556.15 BOOL  ; SCU21_2 P1 Hardware settings
1557.00 BOOL  ; SCU21_2 P1 Reserved
1557.01 BOOL  ; SCU21_2 P1 Reserved
1557.02 BOOL  ; SCU21_2 P1 Reserved
1557.03 BOOL  ; SCU21_2 P1 RTS (RS) signal
1557.04 BOOL  ; SCU21_2 P1 CTS (CS) signal
1557.05 BOOL  ; SCU21_2 P1 Reserved
1557.06 BOOL  ; SCU21_2 P1 DSR (DR) signal
1557.07 BOOL  ; SCU21_2 P1 DTR (ER) signal
1557.08 BOOL  ; SCU21_2 P1 Local Unit busy receiving (Flow control)
1557.09 BOOL  ; SCU21_2 P1 Reserved
1557.10 BOOL  ; SCU21_2 P1 Remote Unit busy receiving (Flow control)
1557.11 BOOL  ; SCU21_2 P1 Reserved
1557.12 BOOL  ; SCU21_2 P1 Reserved
1557.13 BOOL  ; SCU21_2 P1 Reserved
1557.14 BOOL  ; SCU21_2 P1 Reserved
1557.15 BOOL  ; SCU21_2 P1 Reserved
1558.00 BOOL  ; SCU21_2 P1 Reserved
1558.01 BOOL  ; SCU21_2 P1 Reserved
1558.02 BOOL  ; SCU21_2 P1 Parity error
1558.03 BOOL  ; SCU21_2 P1 Framing error
1558.04 BOOL  ; SCU21_2 P1 Overrun error
1558.05 BOOL  ; SCU21_2 P1 Timeout error
1558.06 BOOL  ; SCU21_2 P1 Command error
1558.07 BOOL  ; SCU21_2 P1 FCS check error
1558.08 BOOL  ; SCU21_2 P1 Number of retries
1558.09 BOOL  ; SCU21_2 P1 Number of retries
1558.10 BOOL  ; SCU21_2 P1 Number of retries
1558.11 BOOL  ; SCU21_2 P1 Number of retries
1558.12 BOOL  ; SCU21_2 P1 Tr exceeded
1558.13 BOOL  ; SCU21_2 P1 Tfr exceeded
1558.14 BOOL  ; SCU21_2 P1 Tfs exceeded
1558.15 BOOL  ; SCU21_2 P1 Transmission error
1559.00 BOOL  ; SCU21_2 P1 Protocol status
1559.01 BOOL  ; SCU21_2 P1 Error codes
1559.02 BOOL  ; SCU21_2 P1 Error codes
1559.03 BOOL  ; SCU21_2 P1 Error codes
1559.04 BOOL  ; SCU21_2 P1 Reserved
1559.05 BOOL  ; SCU21_2 P1 Reserved
1559.06 BOOL  ; SCU21_2 P1 Reserved
1559.07 BOOL  ; SCU21_2 P1 Reserved
1559.08 BOOL  ; SCU21_2 P1 Serial Gateway Prohibited Flag
1559.09 BOOL  ; SCU21_2 P1 Sequence Waiting Flag
1559.10 BOOL  ; SCU21_2 P1 Sequence Abort Completion Flag
1559.11 BOOL  ; SCU21_2 P1 Sequence End Completion Flag
1559.12 BOOL  ; SCU21_2 P1 Tracing Flag
1559.13 BOOL  ; SCU21_2 P1 Aborted Flag
1559.14 BOOL  ; SCU21_2 P1 Step Troubleshooting Flag
1559.15 BOOL  ; SCU21_2 P1 Protocol Macro Executing Flag
155.00 BOOL  ; RK_05 U2_Y #2入壳Y轴待料位触发
155.01 BOOL  ; RK_05 U2_Y #2入壳Y轴滚轮压紧位触发
155.02 BOOL  ; RK_05 U2_Y #2入壳Y轴滚轮松开位触发
155.03 BOOL  ; RK_05 U2_Y #2入壳Y轴入壳位触发
155.04 BOOL  ; RK_05 U2_Y #2入壳Y轴电芯定位夹爪松开位触发
155.10 BOOL  ; RK_05 U2_Y #2入壳Y轴回原点触发
155.11 BOOL  ; RK_05 U2_Y #2入壳Y轴JOG+
155.12 BOOL  ; RK_05 U2_Y #2入壳Y轴JOG-
155.13 BOOL  ; RK_05 U2_Y #2入壳Y轴JOG高速
155.14 BOOL  ; RK_05 U2_Y #2入壳Y轴JOG低速
155.15 BOOL  ; 备用
1560.00 BOOL  ; SCU21_2 P1 Communications Sequence Number
1560.01 BOOL  ; SCU21_2 P1 Communications Sequence Number
1560.02 BOOL  ; SCU21_2 P1 Communications Sequence Number
1560.03 BOOL  ; SCU21_2 P1 Communications Sequence Number
1560.04 BOOL  ; SCU21_2 P1 Communications Sequence Number
1560.05 BOOL  ; SCU21_2 P1 Communications Sequence Number
1560.06 BOOL  ; SCU21_2 P1 Communications Sequence Number
1560.07 BOOL  ; SCU21_2 P1 Communications Sequence Number
1560.08 BOOL  ; SCU21_2 P1 Communications Sequence Number
1560.09 BOOL  ; SCU21_2 P1 Communications Sequence Number
1560.10 BOOL  ; SCU21_2 P1 Communications Sequence Number
1560.11 BOOL  ; SCU21_2 P1 Communications Sequence Number
1560.12 BOOL  ; SCU21_2 P1 Reserved
1560.13 BOOL  ; SCU21_2 P1 Reserved
1560.14 BOOL  ; SCU21_2 P1 Reserved
1560.15 BOOL  ; SCU21_2 P1 Reserved
1561.00 BOOL  ; SCU21_2 P1 Executed Reception Case Number
1561.01 BOOL  ; SCU21_2 P1 Executed Reception Case Number
1561.02 BOOL  ; SCU21_2 P1 Executed Reception Case Number
1561.03 BOOL  ; SCU21_2 P1 Executed Reception Case Number
1561.04 BOOL  ; SCU21_2 P1 Reserved
1561.05 BOOL  ; SCU21_2 P1 Reserved
1561.06 BOOL  ; SCU21_2 P1 Reserved
1561.07 BOOL  ; SCU21_2 P1 Reserved
1561.08 BOOL  ; SCU21_2 P1 Executed Step Number
1561.09 BOOL  ; SCU21_2 P1 Executed Step Number
1561.10 BOOL  ; SCU21_2 P1 Executed Step Number
1561.11 BOOL  ; SCU21_2 P1 Executed Step Number
1561.12 BOOL  ; SCU21_2 P1 Reserved
1561.13 BOOL  ; SCU21_2 P1 Reserved
1561.14 BOOL  ; SCU21_2 P1 Reserved
1561.15 BOOL  ; SCU21_2 P1 Reserved
1562.00 BOOL  ; SCU21_2 P1 Executed Reception Case Number Storage Flag
1562.01 BOOL  ; SCU21_2 P1 Executed Reception Case Number Storage Flag
1562.02 BOOL  ; SCU21_2 P1 Executed Reception Case Number Storage Flag
1562.03 BOOL  ; SCU21_2 P1 Executed Reception Case Number Storage Flag
1562.04 BOOL  ; SCU21_2 P1 Executed Reception Case Number Storage Flag
1562.05 BOOL  ; SCU21_2 P1 Executed Reception Case Number Storage Flag
1562.06 BOOL  ; SCU21_2 P1 Executed Reception Case Number Storage Flag
1562.07 BOOL  ; SCU21_2 P1 Executed Reception Case Number Storage Flag
1562.08 BOOL  ; SCU21_2 P1 Executed Reception Case Number Storage Flag
1562.09 BOOL  ; SCU21_2 P1 Executed Reception Case Number Storage Flag
1562.10 BOOL  ; SCU21_2 P1 Executed Reception Case Number Storage Flag
1562.11 BOOL  ; SCU21_2 P1 Executed Reception Case Number Storage Flag
1562.12 BOOL  ; SCU21_2 P1 Executed Reception Case Number Storage Flag
1562.13 BOOL  ; SCU21_2 P1 Executed Reception Case Number Storage Flag
1562.14 BOOL  ; SCU21_2 P1 Executed Reception Case Number Storage Flag
1562.15 BOOL  ; SCU21_2 P1 Executed Reception Case Number Storage Flag
1563.00 BOOL  ; SCU21_2 P1 Executed Step Number Storage Flag
1563.01 BOOL  ; SCU21_2 P1 Executed Step Number Storage Flag
1563.02 BOOL  ; SCU21_2 P1 Executed Step Number Storage Flag
1563.03 BOOL  ; SCU21_2 P1 Executed Step Number Storage Flag
1563.04 BOOL  ; SCU21_2 P1 Executed Step Number Storage Flag
1563.05 BOOL  ; SCU21_2 P1 Executed Step Number Storage Flag
1563.06 BOOL  ; SCU21_2 P1 Executed Step Number Storage Flag
1563.07 BOOL  ; SCU21_2 P1 Executed Step Number Storage Flag
1563.08 BOOL  ; SCU21_2 P1 Executed Step Number Storage Flag
1563.09 BOOL  ; SCU21_2 P1 Executed Step Number Storage Flag
1563.10 BOOL  ; SCU21_2 P1 Executed Step Number Storage Flag
1563.11 BOOL  ; SCU21_2 P1 Executed Step Number Storage Flag
1563.12 BOOL  ; SCU21_2 P1 Executed Step Number Storage Flag
1563.13 BOOL  ; SCU21_2 P1 Executed Step Number Storage Flag
1563.14 BOOL  ; SCU21_2 P1 Executed Step Number Storage Flag
1563.15 BOOL  ; SCU21_2 P1 Executed Step Number Storage Flag
1564.00 BOOL  ; SCU21_2 P1 Repeat Counter Present Value
1564.01 BOOL  ; SCU21_2 P1 Repeat Counter Present Value
1564.02 BOOL  ; SCU21_2 P1 Repeat Counter Present Value
1564.03 BOOL  ; SCU21_2 P1 Repeat Counter Present Value
1564.04 BOOL  ; SCU21_2 P1 Repeat Counter Present Value
1564.05 BOOL  ; SCU21_2 P1 Repeat Counter Present Value
1564.06 BOOL  ; SCU21_2 P1 Repeat Counter Present Value
1564.07 BOOL  ; SCU21_2 P1 Repeat Counter Present Value
1564.08 BOOL  ; SCU21_2 P1 Repeat Counter Setting Value
1564.09 BOOL  ; SCU21_2 P1 Repeat Counter Setting Value
1564.10 BOOL  ; SCU21_2 P1 Repeat Counter Setting Value
1564.11 BOOL  ; SCU21_2 P1 Repeat Counter Setting Value
1564.12 BOOL  ; SCU21_2 P1 Repeat Counter Setting Value
1564.13 BOOL  ; SCU21_2 P1 Repeat Counter Setting Value
1564.14 BOOL  ; SCU21_2 P1 Repeat Counter Setting Value
1564.15 BOOL  ; SCU21_2 P1 Repeat Counter Setting Value
1565.00 BOOL  ; SCU21_2 P2 Parity: Even/Odd
1565.01 BOOL  ; SCU21_2 P2 Parity: Yes/No
1565.02 BOOL  ; SCU21_2 P2 Stop bits: 1 or 2 bits
1565.03 BOOL  ; SCU21_2 P2 Data length: 7 or 8 bits
1565.04 BOOL  ; SCU21_2 P2 Start bits: Always 1
1565.05 BOOL  ; SCU21_2 P2 Reserved
1565.06 BOOL  ; SCU21_2 P2 Reserved
1565.07 BOOL  ; SCU21_2 P2 Reserved
1565.08 BOOL  ; SCU21_2 P2 Baud rate
1565.09 BOOL  ; SCU21_2 P2 Baud rate
1565.10 BOOL  ; SCU21_2 P2 Baud rate
1565.11 BOOL  ; SCU21_2 P2 Baud rate
1565.12 BOOL  ; SCU21_2 P2 Serial communications mode
1565.13 BOOL  ; SCU21_2 P2 Serial communications mode
1565.14 BOOL  ; SCU21_2 P2 Serial communications mode
1565.15 BOOL  ; SCU21_2 P2 Serial communications mode
1566.00 BOOL  ; SCU21_2 P2 1:  operating; 0:  Stopped
1566.01 BOOL  ; SCU21_2 P2 1: System Setup error; 0: System Setup normal
1566.02 BOOL  ; SCU21_2 P2 Reserved
1566.03 BOOL  ; SCU21_2 P2 Reserved
1566.04 BOOL  ; SCU21_2 P2 Reserved
1566.05 BOOL  ; SCU21_2 P2 Reserved
1566.06 BOOL  ; SCU21_2 P2 Reserved
1566.07 BOOL  ; SCU21_2 P2 Reserved
1566.08 BOOL  ; SCU21_2 P2 Reserved
1566.09 BOOL  ; SCU21_2 P2 Reserved
1566.10 BOOL  ; SCU21_2 P2 Reserved
1566.11 BOOL  ; SCU21_2 P2 Reserved
1566.12 BOOL  ; SCU21_2 P2 Reserved
1566.13 BOOL  ; SCU21_2 P2 Terminating resistance
1566.14 BOOL  ; SCU21_2 P2 Hardware settings
1566.15 BOOL  ; SCU21_2 P2 Hardware settings
1567.00 BOOL  ; SCU21_2 P2 Reserved
1567.01 BOOL  ; SCU21_2 P2 Reserved
1567.02 BOOL  ; SCU21_2 P2 Reserved
1567.03 BOOL  ; SCU21_2 P2 RTS (RS) signal
1567.04 BOOL  ; SCU21_2 P2 CTS (CS) signal
1567.05 BOOL  ; SCU21_2 P2 Reserved
1567.06 BOOL  ; SCU21_2 P2 DSR (DR) signal
1567.07 BOOL  ; SCU21_2 P2 DTR (ER) signal
1567.08 BOOL  ; SCU21_2 P2 Local Unit busy receiving (Flow control)
1567.09 BOOL  ; SCU21_2 P2 Reserved
1567.10 BOOL  ; SCU21_2 P2 Remote Unit busy receiving (Flow control)
1567.11 BOOL  ; SCU21_2 P2 Reserved
1567.12 BOOL  ; SCU21_2 P2 Reserved
1567.13 BOOL  ; SCU21_2 P2 Reserved
1567.14 BOOL  ; SCU21_2 P2 Reserved
1567.15 BOOL  ; SCU21_2 P2 Reserved
1568.00 BOOL  ; SCU21_2 P2 Reserved
1568.01 BOOL  ; SCU21_2 P2 Reserved
1568.02 BOOL  ; SCU21_2 P2 Parity error
1568.03 BOOL  ; SCU21_2 P2 Framing error
1568.04 BOOL  ; SCU21_2 P2 Overrun error
1568.05 BOOL  ; SCU21_2 P2 Timeout error
1568.06 BOOL  ; SCU21_2 P2 Command error
1568.07 BOOL  ; SCU21_2 P2 FCS check error
1568.08 BOOL  ; SCU21_2 P2 Number of retries
1568.09 BOOL  ; SCU21_2 P2 Number of retries
1568.10 BOOL  ; SCU21_2 P2 Number of retries
1568.11 BOOL  ; SCU21_2 P2 Number of retries
1568.12 BOOL  ; SCU21_2 P2 Tr exceeded
1568.13 BOOL  ; SCU21_2 P2 Tfr exceeded
1568.14 BOOL  ; SCU21_2 P2 Tfs exceeded
1568.15 BOOL  ; SCU21_2 P2 Transmission error
1569.00 BOOL  ; SCU21_2 P2 Protocol status
1569.01 BOOL  ; SCU21_2 P2 Error codes
1569.02 BOOL  ; SCU21_2 P2 Error codes
1569.03 BOOL  ; SCU21_2 P2 Error codes
1569.04 BOOL  ; SCU21_2 P2 Reserved
1569.05 BOOL  ; SCU21_2 P2 Reserved
1569.06 BOOL  ; SCU21_2 P2 Reserved
1569.07 BOOL  ; SCU21_2 P2 Reserved
1569.08 BOOL  ; SCU21_2 P2 Serial Gateway Prohibited Flag
1569.09 BOOL  ; SCU21_2 P2 Sequence Waiting Flag
1569.10 BOOL  ; SCU21_2 P2 Sequence Abort Completion Flag
1569.11 BOOL  ; SCU21_2 P2 Sequence End Completion Flag
1569.12 BOOL  ; SCU21_2 P2 Tracing Flag
1569.13 BOOL  ; SCU21_2 P2 Aborted Flag
1569.14 BOOL  ; SCU21_2 P2 Step Troubleshooting Flag
1569.15 BOOL  ; SCU21_2 P2 Protocol Macro Executing Flag
156.00 BOOL  ; RK_12 U4_X 预焊上下料X轴待料位触发
156.01 BOOL  ; RK_12 U4_X 预焊上下料X轴除尘取料位触发
156.02 BOOL  ; RK_12 U4_X 预焊上下料X轴#1移载放料位触发
156.03 BOOL  ; RK_12 U4_X 预焊上下料X轴#2移载放料位触发
156.04 BOOL  ; RK_12 U4_X 预焊上下料X轴#1移载取料位触发
156.05 BOOL  ; RK_12 U4_X 预焊上下料X轴#2移载取料位触发
156.06 BOOL  ; RK_12 U4_X 预焊上下料X轴OK放料位触发
156.07 BOOL  ; RK_12 U4_X 预焊上下料X轴#1NG放料位触发
156.08 BOOL  ; RK_12 U4_X 预焊上下料X轴#2NG放料位触发
156.10 BOOL  ; RK_12 U4_X 预焊上下料X轴回原点触发
156.11 BOOL  ; RK_12 U4_X 预焊上下料X轴JOG+
156.12 BOOL  ; RK_12 U4_X 预焊上下料X轴JOG-
156.13 BOOL  ; RK_12 U4_X 预焊上下料X轴JOG高速
156.14 BOOL  ; RK_12 U4_X 预焊上下料X轴JOG低速
156.15 BOOL  ; 备用
1570.00 BOOL  ; SCU21_2 P2 Communications Sequence Number
1570.01 BOOL  ; SCU21_2 P2 Communications Sequence Number
1570.02 BOOL  ; SCU21_2 P2 Communications Sequence Number
1570.03 BOOL  ; SCU21_2 P2 Communications Sequence Number
1570.04 BOOL  ; SCU21_2 P2 Communications Sequence Number
1570.05 BOOL  ; SCU21_2 P2 Communications Sequence Number
1570.06 BOOL  ; SCU21_2 P2 Communications Sequence Number
1570.07 BOOL  ; SCU21_2 P2 Communications Sequence Number
1570.08 BOOL  ; SCU21_2 P2 Communications Sequence Number
1570.09 BOOL  ; SCU21_2 P2 Communications Sequence Number
1570.10 BOOL  ; SCU21_2 P2 Communications Sequence Number
1570.11 BOOL  ; SCU21_2 P2 Communications Sequence Number
1570.12 BOOL  ; SCU21_2 P2 Reserved
1570.13 BOOL  ; SCU21_2 P2 Reserved
1570.14 BOOL  ; SCU21_2 P2 Reserved
1570.15 BOOL  ; SCU21_2 P2 Reserved
1571.00 BOOL  ; SCU21_2 P2 Executed Reception Case Number
1571.01 BOOL  ; SCU21_2 P2 Executed Reception Case Number
1571.02 BOOL  ; SCU21_2 P2 Executed Reception Case Number
1571.03 BOOL  ; SCU21_2 P2 Executed Reception Case Number
1571.04 BOOL  ; SCU21_2 P2 Reserved
1571.05 BOOL  ; SCU21_2 P2 Reserved
1571.06 BOOL  ; SCU21_2 P2 Reserved
1571.07 BOOL  ; SCU21_2 P2 Reserved
1571.08 BOOL  ; SCU21_2 P2 Executed Step Number
1571.09 BOOL  ; SCU21_2 P2 Executed Step Number
1571.10 BOOL  ; SCU21_2 P2 Executed Step Number
1571.11 BOOL  ; SCU21_2 P2 Executed Step Number
1571.12 BOOL  ; SCU21_2 P2 Reserved
1571.13 BOOL  ; SCU21_2 P2 Reserved
1571.14 BOOL  ; SCU21_2 P2 Reserved
1571.15 BOOL  ; SCU21_2 P2 Reserved
1572.00 BOOL  ; SCU21_2 P2 Executed Reception Case Number Storage Flag
1572.01 BOOL  ; SCU21_2 P2 Executed Reception Case Number Storage Flag
1572.02 BOOL  ; SCU21_2 P2 Executed Reception Case Number Storage Flag
1572.03 BOOL  ; SCU21_2 P2 Executed Reception Case Number Storage Flag
1572.04 BOOL  ; SCU21_2 P2 Executed Reception Case Number Storage Flag
1572.05 BOOL  ; SCU21_2 P2 Executed Reception Case Number Storage Flag
1572.06 BOOL  ; SCU21_2 P2 Executed Reception Case Number Storage Flag
1572.07 BOOL  ; SCU21_2 P2 Executed Reception Case Number Storage Flag
1572.08 BOOL  ; SCU21_2 P2 Executed Reception Case Number Storage Flag
1572.09 BOOL  ; SCU21_2 P2 Executed Reception Case Number Storage Flag
1572.10 BOOL  ; SCU21_2 P2 Executed Reception Case Number Storage Flag
1572.11 BOOL  ; SCU21_2 P2 Executed Reception Case Number Storage Flag
1572.12 BOOL  ; SCU21_2 P2 Executed Reception Case Number Storage Flag
1572.13 BOOL  ; SCU21_2 P2 Executed Reception Case Number Storage Flag
1572.14 BOOL  ; SCU21_2 P2 Executed Reception Case Number Storage Flag
1572.15 BOOL  ; SCU21_2 P2 Executed Reception Case Number Storage Flag
1573.00 BOOL  ; SCU21_2 P2 Executed Step Number Storage Flag
1573.01 BOOL  ; SCU21_2 P2 Executed Step Number Storage Flag
1573.02 BOOL  ; SCU21_2 P2 Executed Step Number Storage Flag
1573.03 BOOL  ; SCU21_2 P2 Executed Step Number Storage Flag
1573.04 BOOL  ; SCU21_2 P2 Executed Step Number Storage Flag
1573.05 BOOL  ; SCU21_2 P2 Executed Step Number Storage Flag
1573.06 BOOL  ; SCU21_2 P2 Executed Step Number Storage Flag
1573.07 BOOL  ; SCU21_2 P2 Executed Step Number Storage Flag
1573.08 BOOL  ; SCU21_2 P2 Executed Step Number Storage Flag
1573.09 BOOL  ; SCU21_2 P2 Executed Step Number Storage Flag
1573.10 BOOL  ; SCU21_2 P2 Executed Step Number Storage Flag
1573.11 BOOL  ; SCU21_2 P2 Executed Step Number Storage Flag
1573.12 BOOL  ; SCU21_2 P2 Executed Step Number Storage Flag
1573.13 BOOL  ; SCU21_2 P2 Executed Step Number Storage Flag
1573.14 BOOL  ; SCU21_2 P2 Executed Step Number Storage Flag
1573.15 BOOL  ; SCU21_2 P2 Executed Step Number Storage Flag
1574.00 BOOL  ; SCU21_2 P2 Repeat Counter Present Value
1574.01 BOOL  ; SCU21_2 P2 Repeat Counter Present Value
1574.02 BOOL  ; SCU21_2 P2 Repeat Counter Present Value
1574.03 BOOL  ; SCU21_2 P2 Repeat Counter Present Value
1574.04 BOOL  ; SCU21_2 P2 Repeat Counter Present Value
1574.05 BOOL  ; SCU21_2 P2 Repeat Counter Present Value
1574.06 BOOL  ; SCU21_2 P2 Repeat Counter Present Value
1574.07 BOOL  ; SCU21_2 P2 Repeat Counter Present Value
1574.08 BOOL  ; SCU21_2 P2 Repeat Counter Setting Value
1574.09 BOOL  ; SCU21_2 P2 Repeat Counter Setting Value
1574.10 BOOL  ; SCU21_2 P2 Repeat Counter Setting Value
1574.11 BOOL  ; SCU21_2 P2 Repeat Counter Setting Value
1574.12 BOOL  ; SCU21_2 P2 Repeat Counter Setting Value
1574.13 BOOL  ; SCU21_2 P2 Repeat Counter Setting Value
1574.14 BOOL  ; SCU21_2 P2 Repeat Counter Setting Value
1574.15 BOOL  ; SCU21_2 P2 Repeat Counter Setting Value
157.00 BOOL  ; RK_12 U4_Y 预焊上料Z轴待料位触发
157.01 BOOL  ; RK_12 U4_Y 预焊上料Z轴除尘取料位触发
157.02 BOOL  ; RK_12 U4_Y 预焊上料Z轴#1移载放料位触发
157.03 BOOL  ; RK_12 U4_Y 预焊上料Z轴#2移载放料位触发
157.10 BOOL  ; RK_12 U4_Y 预焊上料Z轴回原点触发
157.11 BOOL  ; RK_12 U4_Y 预焊上料Z轴JOG+
157.12 BOOL  ; RK_12 U4_Y 预焊上料Z轴JOG-
157.13 BOOL  ; RK_12 U4_Y 预焊上料Z轴JOG高速
157.14 BOOL  ; RK_12 U4_Y 预焊上料Z轴JOG低速
157.15 BOOL  ; 备用
158.00 BOOL  ; RK_12 U4_Z 预焊下料Z轴待料位触发
158.01 BOOL  ; RK_12 U4_Z 预焊下料Z轴#1移载取料位触发
158.02 BOOL  ; RK_12 U4_Z 预焊下料Z轴#2移载取料位触发
158.03 BOOL  ; RK_12 U4_Z 预焊下料Z轴OK放料位触发
158.04 BOOL  ; RK_12 U4_Z 预焊下料Z轴#1NG放料位触发
158.05 BOOL  ; RK_12 U4_Z 预焊下料Z轴#2NG放料位触发
158.10 BOOL  ; RK_12 U4_Z 预焊下料Z轴回原点触发
158.11 BOOL  ; RK_12 U4_Z 预焊下料Z轴JOG+
158.12 BOOL  ; RK_12 U4_Z 预焊下料Z轴JOG-
158.13 BOOL  ; RK_12 U4_Z 预焊下料Z轴JOG高速
158.14 BOOL  ; RK_12 U4_Z 预焊下料Z轴JOG低速
158.15 BOOL  ; 备用
159.00 BOOL  ; RK_13 U4_U #1移载Y轴待料位触发
159.01 BOOL  ; RK_13 U4_U #1移载Y轴取放料位触发
159.02 BOOL  ; RK_13 U4_U #1移载Y轴压装位触发
159.03 BOOL  ; RK_13 U4_U #1移载Y轴#1轮廓检测位触发
159.04 BOOL  ; RK_13 U4_U #1移载Y轴#2轮廓检测位触发
159.05 BOOL  ; RK_13 U4_U #1移载Y轴激光焊接位触发
159.10 BOOL  ; RK_13 U4_U #1移载Y轴回原点触发
159.11 BOOL  ; RK_13 U4_U #1移载Y轴JOG+
159.12 BOOL  ; RK_13 U4_U #1移载Y轴JOG-
159.13 BOOL  ; RK_13 U4_U #1移载Y轴JOG高速
159.14 BOOL  ; RK_13 U4_U #1移载Y轴JOG低速
159.15 BOOL  ; 备用
15.00 BOOL  ; RK_08 铝壳除尘旋转伸缩气缸原位
15.01 BOOL  ; RK_08 铝壳除尘旋转伸缩气缸到位
15.02 BOOL  ; RK_08 铝壳除尘伸缩气缸伸出位
15.03 BOOL  ; RK_08 铝壳除尘伸缩气缸缩回位
15.04 BOOL  ; RK_08 铝壳除尘夹爪气缸夹紧位
15.05 BOOL  ; RK_08 铝壳除尘夹爪气缸张开位
15.06 BOOL  ; RK_09 #1Hipot测试旋转伸缩气缸到位
15.07 BOOL  ; RK_09 #1Hipot测试旋转伸缩气缸原位
15.08 BOOL  ; RK_09 #1Hipot测试平台伸缩气缸缩回位
15.09 BOOL  ; RK_09 #1Hipot测试平台伸缩气缸伸出位
15.10 BOOL  ; RK_09 #1Hipot测试伸缩气缸伸出位
15.11 BOOL  ; RK_09 #1Hipot测试伸缩气缸缩回位
15.12 BOOL  ; RK_09 #2Hipot测试旋转伸缩气缸到位
15.13 BOOL  ; RK_09 #2Hipot测试旋转伸缩气缸原位
15.14 BOOL  ; RK_09 #2Hipot测试平台伸缩气缸缩回位
15.15 BOOL  ; RK_09 #2Hipot测试平台伸缩气缸伸出位
160.00 BOOL  ; RK_13 U6_X #2移载Y轴待料位触发
160.01 BOOL  ; RK_13 U6_X #2移载Y轴取放料位触发
160.02 BOOL  ; RK_13 U6_X #2移载Y轴压装位触发
160.03 BOOL  ; RK_13 U6_X #2移载Y轴#1轮廓检测位触发
160.04 BOOL  ; RK_13 U6_X #2移载Y轴#2轮廓检测位触发
160.05 BOOL  ; RK_13 U6_X #2移载Y轴激光焊接位触发
160.10 BOOL  ; RK_13 U6_X #2移载Y轴回原点触发
160.11 BOOL  ; RK_13 U6_X #2移载Y轴JOG+
160.12 BOOL  ; RK_13 U6_X #2移载Y轴JOG-
160.13 BOOL  ; RK_13 U6_X #2移载Y轴JOG高速
160.14 BOOL  ; RK_13 U6_X #2移载Y轴JOG低速
160.15 BOOL  ; 备用
161.00 BOOL  ; RK_16 U6_Y 激光焊接X轴待机位触发
161.01 BOOL  ; RK_16 U6_Y 激光焊接X轴#1移载焊接位触发
161.02 BOOL  ; RK_16 U6_Y 激光焊接X轴#2移载焊接位触发
161.10 BOOL  ; RK_16 U6_Y 激光焊接X轴回原点触发
161.11 BOOL  ; RK_16 U6_Y 激光焊接X轴JOG+
161.12 BOOL  ; RK_16 U6_Y 激光焊接X轴JOG-
161.13 BOOL  ; RK_16 U6_Y 激光焊接X轴JOG高速
161.14 BOOL  ; RK_16 U6_Y 激光焊接X轴JOG低速
161.15 BOOL  ; 备用
162.00 BOOL  ; RK_16 U6_Z 激光焊接Z轴待机位触发
162.01 BOOL  ; RK_16 U6_Z 激光焊接Z轴#1移载焊接位触发
162.02 BOOL  ; RK_16 U6_Z 激光焊接Z轴#2移载焊接位触发
162.10 BOOL  ; RK_16 U6_Z 激光焊接Z轴回原点触发
162.11 BOOL  ; RK_16 U6_Z 激光焊接Z轴JOG+
162.12 BOOL  ; RK_16 U6_Z 激光焊接Z轴JOG-
162.13 BOOL  ; RK_16 U6_Z 激光焊接Z轴JOG高速
162.14 BOOL  ; RK_16 U6_Z 激光焊接Z轴JOG低速
162.15 BOOL  ; 备用
163.00 BOOL  ; RK_06 U8_X 电池上下料X轴待机位触发
163.01 BOOL  ; RK_06 U8_X 电池上下料X轴铝壳除尘取料位触发
163.02 BOOL  ; RK_06 U8_X 电池上下料X轴#1入壳放料位触发
163.03 BOOL  ; RK_06 U8_X 电池上下料X轴#2入壳放料位触发
163.04 BOOL  ; RK_06 U8_X 电池上下料X轴#1入壳取料位触发
163.05 BOOL  ; RK_06 U8_X 电池上下料X轴#2入壳取料位触发
163.06 BOOL  ; RK_06 U8_X 电池上下料X轴#1Hipot检测放料位触发
163.07 BOOL  ; RK_06 U8_X 电池上下料X轴#2Hipot检测放料位触发
163.10 BOOL  ; RK_06 U8_X 电池上下料X轴回原点触发
163.11 BOOL  ; RK_06 U8_X 电池上下料X轴JOG+
163.12 BOOL  ; RK_06 U8_X 电池上下料X轴JOG-
163.13 BOOL  ; RK_06 U8_X 电池上下料X轴JOG高速
163.14 BOOL  ; RK_06 U8_X 电池上下料X轴JOG低速
163.15 BOOL  ; 备用
164.00 BOOL  ; RK_07 U8_Y 铝壳进料X轴等待位触发
164.01 BOOL  ; RK_07 U8_Y 铝壳进料X轴取料位触发
164.02 BOOL  ; RK_07 U8_Y 铝壳进料X轴放料位触发
164.10 BOOL  ; RK_07 U8_Y 铝壳进料X轴回原点触发
164.11 BOOL  ; RK_07 U8_Y 铝壳进料X轴JOG+
164.12 BOOL  ; RK_07 U8_Y 铝壳进料X轴JOG-
164.13 BOOL  ; RK_07 U8_Y 铝壳进料X轴JOG高速
164.14 BOOL  ; RK_07 U8_Y 铝壳进料X轴JOG低速
164.15 BOOL  ; 备用
165.00 BOOL  ; RK_07 U8_Z 铝壳上料移载Y轴待料位触发
165.01 BOOL  ; RK_07 U8_Z 铝壳上料移载Y轴#1铝壳上料位触发
165.02 BOOL  ; RK_07 U8_Z 铝壳上料移载Y轴#2铝壳上料位触发
165.03 BOOL  ; RK_07 U8_Z 铝壳上料移载Y轴#3铝壳托盘下料位触发
165.04 BOOL  ; RK_07 U8_Z 铝壳上料移载Y轴铝壳取料位触发
165.10 BOOL  ; RK_07 U8_Z 铝壳上料移载Y轴回原点触发
165.11 BOOL  ; RK_07 U8_Z 铝壳上料移载Y轴JOG+
165.12 BOOL  ; RK_07 U8_Z 铝壳上料移载Y轴JOG-
165.13 BOOL  ; RK_07 U8_Z 铝壳上料移载Y轴JOG高速
165.14 BOOL  ; RK_07 U8_Z 铝壳上料移载Y轴JOG低速
165.15 BOOL  ; 备用
166.00 BOOL  ; RK_10 U8_U 电池除尘上料X轴待料位触发
166.01 BOOL  ; RK_10 U8_U 电池除尘上料X轴#1Hipot检测取料位触发
166.02 BOOL  ; RK_10 U8_U 电池除尘上料X轴#2Hipot检测取料位触发
166.03 BOOL  ; RK_10 U8_U 电池除尘上料X轴Hipot OK放料位触发
166.04 BOOL  ; RK_10 U8_U 电池除尘上料X轴Hipot NG放料位触发
166.10 BOOL  ; RK_10 U8_U 电池除尘上料X轴回原点触发
166.11 BOOL  ; RK_10 U8_U 电池除尘上料X轴JOG+
166.12 BOOL  ; RK_10 U8_U 电池除尘上料X轴JOG-
166.13 BOOL  ; RK_10 U8_U 电池除尘上料X轴JOG高速
166.14 BOOL  ; RK_10 U8_U 电池除尘上料X轴JOG低速
166.15 BOOL  ; 备用
16.00 BOOL  ; RK_09 #2Hipot测试伸缩气缸伸出位
16.01 BOOL  ; RK_09 #2Hipot测试伸缩气缸缩回位
16.02 BOOL  ; RK_10 电池除尘上料机械手升降气缸下降位
16.03 BOOL  ; RK_10 电池除尘上料机械手升降气缸上升位
16.04 BOOL  ; RK_10 电池除尘上料机械手夹爪气缸夹紧位
16.05 BOOL  ; RK_10 电池除尘上料机械手夹爪气缸张开位
16.06 BOOL  ; RK_06 U8_X 电池上下料X轴报警信号
16.07 BOOL  ; RK_06 U8_X 电池上下料X轴准备好了信号
16.08 BOOL  ; RK_07 U8_Y 铝壳进料X轴报警信号
16.09 BOOL  ; RK_07 U8_Y 铝壳进料X轴准备好了信号
16.10 BOOL  ; RK_07 U8_Z 铝壳上料移载Y轴报警信号
16.11 BOOL  ; RK_07 U8_Z 铝壳上料移载Y轴准备好了信号
16.12 BOOL  ; RK_10 U8_U 电池除尘上料X轴报警信号
16.13 BOOL  ; RK_10 U8_U 电池除尘上料X轴准备好了信号
16.14 BOOL  ; RK_09 Hipot测试完成信号
16.15 BOOL  ; RK_07 #1铝壳上料启动按钮
17.00 BOOL  ; RK_07 #2铝壳上料启动按钮
17.01 BOOL  ; RK_07 #3托盘下料启动按钮
17.02 BOOL  ; RK_07 铝壳上料移载吸盘真空
17.03 BOOL  ; RK_07 铝壳进料吸盘真空
17.04 BOOL  ; RK_07 #1铝壳上料托盘到位感应
17.05 BOOL  ; RK_07 #1铝壳上料位物料车到位感应
17.06 BOOL  ; RK_07 #1铝壳上料初始位（#1）
17.07 BOOL  ; RK_07 #1铝壳上料一个托盘位（#2）
17.08 BOOL  ; RK_07 #1铝壳上料高限位（#3）
17.09 BOOL  ; RK_07 #2铝壳上料托盘到位感应
17.10 BOOL  ; RK_07 #2铝壳上料位物料车到位感应
17.11 BOOL  ; RK_07 #2铝壳上料初始位（#1）
17.12 BOOL  ; RK_07 #2铝壳上料一个托盘位（#2）
17.13 BOOL  ; RK_07 #2铝壳上料高限位（#3）
17.14 BOOL  ; RK_07 #3托盘下料上升到位感应
17.15 BOOL  ; RK_07 #3托盘下料位物料车到位感应
18.00 BOOL  ; RK_07 #3托盘下料初始位（#1）
18.01 BOOL  ; RK_07 #3托盘下料满托盘位（#2）
18.02 BOOL  ; RK_07 #3托盘下料高限位（#3）
18.03 BOOL  ; RK_07 铝壳上料移载托盘到位感应
18.04 BOOL  ; RK_08 铝壳除尘有料感应
18.05 BOOL  ; RK_09 #1Hipot测试有料感应
18.06 BOOL  ; RK_09 #2Hipot测试有料感应
18.07 BOOL  ; RK_10 Hipot检测NG拉带有料感应#1
18.08 BOOL  ; RK_10 Hipot检测NG拉带有料感应#2
18.09 BOOL  ; RK_10 Hipot检测NG拉带料满感应
18.10 BOOL  ; RK_06 铝壳上料夹爪柔性报警
18.11 BOOL  ; RK_06 电池下料夹爪柔性报警
18.12 BOOL  ; RK_07 铝壳进料机械手柔性报警
18.13 BOOL  ; RK_10 电池除尘上料机械手夹爪柔性报警
18.14 BOOL  ; 手/自动选择（公共）
18.15 BOOL  ; 启动按钮_绿（公共）
19.00 BOOL  ; 停止按钮_红（公共）
19.01 BOOL  ; 复位按钮_黄（公共）
19.02 BOOL  ; 机台进气压力（正压）（公共）
19.03 BOOL  ; 机台进气压力（负压）（公共）
19.04 BOOL  ; 主屏急停（公共）
19.05 BOOL  ; 铝壳上料端急停（公共）
19.06 BOOL  ; HipotNG端急停（公共）
19.07 BOOL  ; B机架#1门磁（公共）
19.08 BOOL  ; B机架#2门磁（公共）
19.09 BOOL  ; B机架#3门磁（公共）
19.10 BOOL  ; B机架#4门磁（公共）
19.11 BOOL  ; B机架#5门磁（公共）
19.12 BOOL  ; B机架#6门磁（公共）
19.13 BOOL  ; RK_07 #3托盘下料下降到位感应
19.14 BOOL  ; $?St$Bk?_#[5013] / RK_07 #3托盘下料位物料车到位感应#2 / $?St$Bk?_#[5013]
19.15 BOOL  ; $?St$Bk?_#[5014] / RK_07 铝壳上料移载托盘到位保护感应 / $?St$Bk?_#[5014]
1.00 BOOL  ; RK_05 #1入壳铝壳定位平台升降气缸上升位
1.01 BOOL  ; RK_05 #1入壳铝壳定位平台升降气缸下降位
1.02 BOOL  ; RK_05 #1入壳铝壳定位伸缩气缸缩回位
1.03 BOOL  ; RK_05 #1入壳铝壳定位伸缩气缸伸出位
1.04 BOOL  ; RK_05 #1入壳铝壳定位夹爪气缸夹紧位
1.05 BOOL  ; RK_05 #1入壳铝壳定位夹爪气缸张开位
1.06 BOOL  ; RK_05 #2入壳滚轮夹紧气缸夹紧位
1.07 BOOL  ; RK_05 #2入壳滚轮夹紧气缸松开位
1.08 BOOL  ; RK_05 #2入壳铝壳定位平台伸缩气缸缩回位
1.09 BOOL  ; RK_05 #2入壳铝壳定位平台伸缩气缸伸出位
1.10 BOOL  ; RK_05 #2入壳铝壳定位平台升降气缸上升位
1.11 BOOL  ; RK_05 #2入壳铝壳定位平台升降气缸下降位
1.12 BOOL  ; RK_05 #2入壳铝壳定位伸缩气缸缩回位
1.13 BOOL  ; RK_05 #2入壳铝壳定位伸缩气缸伸出位
1.14 BOOL  ; RK_05 #2入壳铝壳定位夹爪气缸夹紧位
1.15 BOOL  ; RK_05 #2入壳铝壳定位夹爪气缸张开位
2000.00 BOOL  ; RK_01 U0_X 电芯来料Y轴序列号使能
2000.01 BOOL  ; RK_01 U0_X 电芯来料Y轴启动
2000.02 BOOL  ; RK_01 U0_X 电芯来料Y轴独立启动
2000.03 BOOL  ; RK_01 U0_X 电芯来料Y轴绝对移动
2000.04 BOOL  ; RK_01 U0_X 电芯来料Y轴相对移动
2000.05 BOOL  ; RK_01 U0_X 电芯来料Y轴中断进给
2000.06 BOOL  ; RK_01 U0_X 电芯来料Y轴原点搜索
2000.07 BOOL  ; RK_01 U0_X 电芯来料Y轴原点返回
2000.08 BOOL  ; RK_01 U0_X 电芯来料Y轴当前位置预置
2000.09 BOOL  ; RK_01 U0_X 电芯来料Y轴点动
2000.10 BOOL  ; RK_01 U0_X 电芯来料Y轴方向定义
2000.11 BOOL  ; RK_01 U0_X 电芯来料Y轴示教
2000.12 BOOL  ; RK_01 U0_X 电芯来料Y轴释放禁止/复位
2000.13 BOOL  ; $?St$Bk?_#[5015] / RK_01 U0_X 电芯来料Y轴偏差计数器复位输出/ / 原点调整命令输出$?St$Bk?_#[5015]
2000.14 BOOL  ; RK_01 U0_X 电芯来料Y轴激活倍率
2000.15 BOOL  ; RK_01 U0_X 电芯来料Y轴停止
2001.00 BOOL  ; RK_01 U0_X 电芯来料Y轴Not Use
2001.01 BOOL  ; RK_01 U0_X 电芯来料Y轴Not Use
2001.02 BOOL  ; RK_01 U0_X 电芯来料Y轴Not Use
2001.03 BOOL  ; RK_01 U0_X 电芯来料Y轴Not Use
2001.04 BOOL  ; RK_01 U0_X 电芯来料Y轴Not Use
2001.05 BOOL  ; RK_01 U0_X 电芯来料Y轴Not Use
2001.06 BOOL  ; RK_01 U0_X 电芯来料Y轴Not Use
2001.07 BOOL  ; RK_01 U0_X 电芯来料Y轴Not Use
2001.08 BOOL  ; RK_01 U0_X 电芯来料Y轴强迫中断
2001.09 BOOL  ; RK_01 U0_X 电芯来料Y轴Not Use
2001.10 BOOL  ; RK_01 U0_X 电芯来料Y轴Not Use
2001.11 BOOL  ; RK_01 U0_X 电芯来料Y轴Not Use
2001.12 BOOL  ; RK_01 U0_X 电芯来料Y轴写数据
2001.13 BOOL  ; RK_01 U0_X 电芯来料Y轴读数据
2001.14 BOOL  ; RK_01 U0_X 电芯来料Y轴存数据
2001.15 BOOL  ; RK_01 U0_X 电芯来料Y轴Not Use
2002.00 BOOL  ; RK_02 U0_Y 电芯进料X轴序列号使能
2002.01 BOOL  ; RK_02 U0_Y 电芯进料X轴启动
2002.02 BOOL  ; RK_02 U0_Y 电芯进料X轴独立启动
2002.03 BOOL  ; RK_02 U0_Y 电芯进料X轴绝对移动
2002.04 BOOL  ; RK_02 U0_Y 电芯进料X轴相对移动
2002.05 BOOL  ; RK_02 U0_Y 电芯进料X轴中断进给
2002.06 BOOL  ; RK_02 U0_Y 电芯进料X轴原点搜索
2002.07 BOOL  ; RK_02 U0_Y 电芯进料X轴原点返回
2002.08 BOOL  ; RK_02 U0_Y 电芯进料X轴当前位置预置
2002.09 BOOL  ; RK_02 U0_Y 电芯进料X轴点动
2002.10 BOOL  ; RK_02 U0_Y 电芯进料X轴方向定义
2002.11 BOOL  ; RK_02 U0_Y 电芯进料X轴示教
2002.12 BOOL  ; RK_02 U0_Y 电芯进料X轴释放禁止/复位
2002.13 BOOL  ; $?St$Bk?_#[5016] / RK_02 U0_Y 电芯进料X轴偏差计数器复位输出/ / 原点调整命令输出$?St$Bk?_#[5016]
2002.14 BOOL  ; RK_02 U0_Y 电芯进料X轴激活倍率
2002.15 BOOL  ; RK_02 U0_Y 电芯进料X轴停止
2003.00 BOOL  ; RK_02 U0_Y 电芯进料X轴Not Use
2003.01 BOOL  ; RK_02 U0_Y 电芯进料X轴Not Use
2003.02 BOOL  ; RK_02 U0_Y 电芯进料X轴Not Use
2003.03 BOOL  ; RK_02 U0_Y 电芯进料X轴Not Use
2003.04 BOOL  ; RK_02 U0_Y 电芯进料X轴Not Use
2003.05 BOOL  ; RK_02 U0_Y 电芯进料X轴Not Use
2003.06 BOOL  ; RK_02 U0_Y 电芯进料X轴Not Use
2003.07 BOOL  ; RK_02 U0_Y 电芯进料X轴Not Use
2003.08 BOOL  ; RK_02 U0_Y 电芯进料X轴强迫中断
2003.09 BOOL  ; RK_02 U0_Y 电芯进料X轴Not Use
2003.10 BOOL  ; RK_02 U0_Y 电芯进料X轴Not Use
2003.11 BOOL  ; RK_02 U0_Y 电芯进料X轴Not Use
2003.12 BOOL  ; RK_02 U0_Y 电芯进料X轴写数据
2003.13 BOOL  ; RK_02 U0_Y 电芯进料X轴读数据
2003.14 BOOL  ; RK_02 U0_Y 电芯进料X轴存数据
2003.15 BOOL  ; RK_02 U0_Y 电芯进料X轴Not Use
2004.00 BOOL  ; RK_02 U0_Z 电芯进料Z轴序列号使能
2004.01 BOOL  ; RK_02 U0_Z 电芯进料Z轴启动
2004.02 BOOL  ; RK_02 U0_Z 电芯进料Z轴独立启动
2004.03 BOOL  ; RK_02 U0_Z 电芯进料Z轴绝对移动
2004.04 BOOL  ; RK_02 U0_Z 电芯进料Z轴相对移动
2004.05 BOOL  ; RK_02 U0_Z 电芯进料Z轴中断进给
2004.06 BOOL  ; RK_02 U0_Z 电芯进料Z轴原点搜索
2004.07 BOOL  ; RK_02 U0_Z 电芯进料Z轴原点返回
2004.08 BOOL  ; RK_02 U0_Z 电芯进料Z轴当前位置预置
2004.09 BOOL  ; RK_02 U0_Z 电芯进料Z轴点动
2004.10 BOOL  ; RK_02 U0_Z 电芯进料Z轴方向定义
2004.11 BOOL  ; RK_02 U0_Z 电芯进料Z轴示教
2004.12 BOOL  ; RK_02 U0_Z 电芯进料Z轴释放禁止/复位
2004.13 BOOL  ; $?St$Bk?_#[5017] / RK_02 U0_Z 电芯进料Z轴偏差计数器复位输出/ / 原点调整命令输出$?St$Bk?_#[5017]
2004.14 BOOL  ; RK_02 U0_Z 电芯进料Z轴激活倍率
2004.15 BOOL  ; RK_02 U0_Z 电芯进料Z轴停止
2005.00 BOOL  ; RK_02 U0_Z 电芯进料Z轴Not Use
2005.01 BOOL  ; RK_02 U0_Z 电芯进料Z轴Not Use
2005.02 BOOL  ; RK_02 U0_Z 电芯进料Z轴Not Use
2005.03 BOOL  ; RK_02 U0_Z 电芯进料Z轴Not Use
2005.04 BOOL  ; RK_02 U0_Z 电芯进料Z轴Not Use
2005.05 BOOL  ; RK_02 U0_Z 电芯进料Z轴Not Use
2005.06 BOOL  ; RK_02 U0_Z 电芯进料Z轴Not Use
2005.07 BOOL  ; RK_02 U0_Z 电芯进料Z轴Not Use
2005.08 BOOL  ; RK_02 U0_Z 电芯进料Z轴强迫中断
2005.09 BOOL  ; RK_02 U0_Z 电芯进料Z轴Not Use
2005.10 BOOL  ; RK_02 U0_Z 电芯进料Z轴Not Use
2005.11 BOOL  ; RK_02 U0_Z 电芯进料Z轴Not Use
2005.12 BOOL  ; RK_02 U0_Z 电芯进料Z轴写数据
2005.13 BOOL  ; RK_02 U0_Z 电芯进料Z轴读数据
2005.14 BOOL  ; RK_02 U0_Z 电芯进料Z轴存数据
2005.15 BOOL  ; RK_02 U0_Z 电芯进料Z轴Not Use
2006.00 BOOL  ; RK_03 U0_U 电芯上料X轴序列号使能
2006.01 BOOL  ; RK_03 U0_U 电芯上料X轴启动
2006.02 BOOL  ; RK_03 U0_U 电芯上料X轴独立启动
2006.03 BOOL  ; RK_03 U0_U 电芯上料X轴绝对移动
2006.04 BOOL  ; RK_03 U0_U 电芯上料X轴相对移动
2006.05 BOOL  ; RK_03 U0_U 电芯上料X轴中断进给
2006.06 BOOL  ; RK_03 U0_U 电芯上料X轴原点搜索
2006.07 BOOL  ; RK_03 U0_U 电芯上料X轴原点返回
2006.08 BOOL  ; RK_03 U0_U 电芯上料X轴当前位置预置
2006.09 BOOL  ; RK_03 U0_U 电芯上料X轴点动
2006.10 BOOL  ; RK_03 U0_U 电芯上料X轴方向定义
2006.11 BOOL  ; RK_03 U0_U 电芯上料X轴示教
2006.12 BOOL  ; RK_03 U0_U 电芯上料X轴释放禁止/复位
2006.13 BOOL  ; $?St$Bk?_#[5018] / RK_03 U0_U 电芯上料X轴偏差计数器复位输出/ / 原点调整命令输出$?St$Bk?_#[5018]
2006.14 BOOL  ; RK_03 U0_U 电芯上料X轴激活倍率
2006.15 BOOL  ; RK_03 U0_U 电芯上料X轴停止
2007.00 BOOL  ; RK_03 U0_U 电芯上料X轴Not Use
2007.01 BOOL  ; RK_03 U0_U 电芯上料X轴Not Use
2007.02 BOOL  ; RK_03 U0_U 电芯上料X轴Not Use
2007.03 BOOL  ; RK_03 U0_U 电芯上料X轴Not Use
2007.04 BOOL  ; RK_03 U0_U 电芯上料X轴Not Use
2007.05 BOOL  ; RK_03 U0_U 电芯上料X轴Not Use
2007.06 BOOL  ; RK_03 U0_U 电芯上料X轴Not Use
2007.07 BOOL  ; RK_03 U0_U 电芯上料X轴Not Use
2007.08 BOOL  ; RK_03 U0_U 电芯上料X轴强迫中断
2007.09 BOOL  ; RK_03 U0_U 电芯上料X轴Not Use
2007.10 BOOL  ; RK_03 U0_U 电芯上料X轴Not Use
2007.11 BOOL  ; RK_03 U0_U 电芯上料X轴Not Use
2007.12 BOOL  ; RK_03 U0_U 电芯上料X轴写数据
2007.13 BOOL  ; RK_03 U0_U 电芯上料X轴读数据
2007.14 BOOL  ; RK_03 U0_U 电芯上料X轴存数据
2007.15 BOOL  ; RK_03 U0_U 电芯上料X轴Not Use
2008.00 BOOL  ; RK_01 U0_X 电芯来料Y轴Not Use
2008.01 BOOL  ; RK_01 U0_X 电芯来料Y轴Not Use
2008.02 BOOL  ; RK_01 U0_X 电芯来料Y轴Not Use
2008.03 BOOL  ; RK_01 U0_X 电芯来料Y轴Not Use
2008.04 BOOL  ; RK_01 U0_X 电芯来料Y轴等待存储器操作标志位
2008.05 BOOL  ; RK_01 U0_X 电芯来料Y轴定位结束标志位
2008.06 BOOL  ; RK_01 U0_X 电芯来料Y轴无原点标志位
2008.07 BOOL  ; RK_01 U0_X 电芯来料Y轴原点停止标志位
2008.08 BOOL  ; RK_01 U0_X 电芯来料Y轴区域0监控标志位
2008.09 BOOL  ; RK_01 U0_X 电芯来料Y轴区域1监控标志位
2008.10 BOOL  ; RK_01 U0_X 电芯来料Y轴区域2监控标志位
2008.11 BOOL  ; RK_01 U0_X 电芯来料Y轴示教完成标志位
2008.12 BOOL  ; RK_01 U0_X 电芯来料Y轴错误标志位
2008.13 BOOL  ; RK_01 U0_X 电芯来料Y轴忙标志位
2008.14 BOOL  ; RK_01 U0_X 电芯来料Y轴数据传送标志
2008.15 BOOL  ; RK_01 U0_X 电芯来料Y轴减速停止执行标志
2009.00 BOOL  ; RK_01 U0_X 电芯来料Y轴Not Use
2009.01 BOOL  ; RK_01 U0_X 电芯来料Y轴Not Use
2009.02 BOOL  ; RK_01 U0_X 电芯来料Y轴Not Use
2009.03 BOOL  ; RK_01 U0_X 电芯来料Y轴Not Use
2009.04 BOOL  ; RK_01 U0_X 电芯来料Y轴Not Use
2009.05 BOOL  ; RK_01 U0_X 电芯来料Y轴Not Use
2009.06 BOOL  ; RK_01 U0_X 电芯来料Y轴Not Use
2009.07 BOOL  ; RK_01 U0_X 电芯来料Y轴Not Use
2009.08 BOOL  ; RK_01 U0_X 电芯来料Y轴CW极限输入信号
2009.09 BOOL  ; RK_01 U0_X 电芯来料Y轴CCW极限输入信号
2009.10 BOOL  ; RK_01 U0_X 电芯来料Y轴原点接近输入信号
2009.11 BOOL  ; RK_01 U0_X 电芯来料Y轴原点输入信号
2009.12 BOOL  ; RK_01 U0_X 电芯来料Y轴中断输入信号
2009.13 BOOL  ; RK_01 U0_X 电芯来料Y轴紧急停止输入信号
2009.14 BOOL  ; RK_01 U0_X 电芯来料Y轴定位完成信号
2009.15 BOOL  ; $?St$Bk?_#[5019] / RK_01 U0_X 电芯来料Y轴偏差计数器复位输出 / 原点调整命令输出$?St$Bk?_#[5019]
200.00 BOOL  ; PLC上电
200.01 BOOL  ; 紧急停止
200.02 BOOL  ; 自动启动
200.03 BOOL  ; 自动停止
200.04 BOOL  ; 报警清除
200.05 BOOL  ; 清料停止中
200.06 BOOL  ; 异常报警停止
200.09 BOOL  ; 设备内有电池
200.10 BOOL  ; 机台有错误
200.11 BOOL  ; 报警中
200.12 BOOL  ; 三色灯-绿灯
200.13 BOOL  ; 三色灯-红灯
200.14 BOOL  ; 三色灯-黄灯
200.15 BOOL  ; 三色灯-蜂鸣器
2010 CHANNEL  ; RK_01 U0_X 电芯来料Y轴错误代码
2010.00 BOOL  ; RK_01 U0_X 电芯来料Y轴错误代码
2010.01 BOOL  ; RK_01 U0_X 电芯来料Y轴错误代码
2010.02 BOOL  ; RK_01 U0_X 电芯来料Y轴错误代码
2010.03 BOOL  ; RK_01 U0_X 电芯来料Y轴错误代码
2010.04 BOOL  ; RK_01 U0_X 电芯来料Y轴错误代码
2010.05 BOOL  ; RK_01 U0_X 电芯来料Y轴错误代码
2010.06 BOOL  ; RK_01 U0_X 电芯来料Y轴错误代码
2010.07 BOOL  ; RK_01 U0_X 电芯来料Y轴错误代码
2010.08 BOOL  ; RK_01 U0_X 电芯来料Y轴错误代码
2010.09 BOOL  ; RK_01 U0_X 电芯来料Y轴错误代码
2010.10 BOOL  ; RK_01 U0_X 电芯来料Y轴错误代码
2010.11 BOOL  ; RK_01 U0_X 电芯来料Y轴错误代码
2010.12 BOOL  ; RK_01 U0_X 电芯来料Y轴错误代码
2010.13 BOOL  ; RK_01 U0_X 电芯来料Y轴错误代码
2010.14 BOOL  ; RK_01 U0_X 电芯来料Y轴错误代码
2010.15 BOOL  ; RK_01 U0_X 电芯来料Y轴错误代码
2011.00 BOOL  ; RK_02 U0_Y 电芯进料X轴Not Use
2011.01 BOOL  ; RK_02 U0_Y 电芯进料X轴Not Use
2011.02 BOOL  ; RK_02 U0_Y 电芯进料X轴Not Use
2011.03 BOOL  ; RK_02 U0_Y 电芯进料X轴Not Use
2011.04 BOOL  ; RK_02 U0_Y 电芯进料X轴等待存储器操作标志位
2011.05 BOOL  ; RK_02 U0_Y 电芯进料X轴定位结束标志位
2011.06 BOOL  ; RK_02 U0_Y 电芯进料X轴无原点标志位
2011.07 BOOL  ; RK_02 U0_Y 电芯进料X轴原点停止标志位
2011.08 BOOL  ; RK_02 U0_Y 电芯进料X轴区域0监控标志位
2011.09 BOOL  ; RK_02 U0_Y 电芯进料X轴区域1监控标志位
2011.10 BOOL  ; RK_02 U0_Y 电芯进料X轴区域2监控标志位
2011.11 BOOL  ; RK_02 U0_Y 电芯进料X轴示教完成标志位
2011.12 BOOL  ; RK_02 U0_Y 电芯进料X轴错误标志位
2011.13 BOOL  ; RK_02 U0_Y 电芯进料X轴忙标志位
2011.14 BOOL  ; RK_02 U0_Y 电芯进料X轴数据传送标志
2011.15 BOOL  ; RK_02 U0_Y 电芯进料X轴减速停止执行标志
2012.00 BOOL  ; RK_02 U0_Y 电芯进料X轴Not Use
2012.01 BOOL  ; RK_02 U0_Y 电芯进料X轴Not Use
2012.02 BOOL  ; RK_02 U0_Y 电芯进料X轴Not Use
2012.03 BOOL  ; RK_02 U0_Y 电芯进料X轴Not Use
2012.04 BOOL  ; RK_02 U0_Y 电芯进料X轴Not Use
2012.05 BOOL  ; RK_02 U0_Y 电芯进料X轴Not Use
2012.06 BOOL  ; RK_02 U0_Y 电芯进料X轴Not Use
2012.07 BOOL  ; RK_02 U0_Y 电芯进料X轴Not Use
2012.08 BOOL  ; RK_02 U0_Y 电芯进料X轴CW极限输入信号
2012.09 BOOL  ; RK_02 U0_Y 电芯进料X轴CCW极限输入信号
2012.10 BOOL  ; RK_02 U0_Y 电芯进料X轴原点接近输入信号
2012.11 BOOL  ; RK_02 U0_Y 电芯进料X轴原点输入信号
2012.12 BOOL  ; RK_02 U0_Y 电芯进料X轴中断输入信号
2012.13 BOOL  ; RK_02 U0_Y 电芯进料X轴紧急停止输入信号
2012.14 BOOL  ; RK_02 U0_Y 电芯进料X轴定位完成信号
2012.15 BOOL  ; $?St$Bk?_#[5020] / RK_02 U0_Y 电芯进料X轴偏差计数器复位输出 / 原点调整命令输出$?St$Bk?_#[5020]
2013 CHANNEL  ; RK_02 U0_Y 电芯进料X轴错误代码
2013.00 BOOL  ; RK_02 U0_Y 电芯进料X轴错误代码
2013.01 BOOL  ; RK_02 U0_Y 电芯进料X轴错误代码
2013.02 BOOL  ; RK_02 U0_Y 电芯进料X轴错误代码
2013.03 BOOL  ; RK_02 U0_Y 电芯进料X轴错误代码
2013.04 BOOL  ; RK_02 U0_Y 电芯进料X轴错误代码
2013.05 BOOL  ; RK_02 U0_Y 电芯进料X轴错误代码
2013.06 BOOL  ; RK_02 U0_Y 电芯进料X轴错误代码
2013.07 BOOL  ; RK_02 U0_Y 电芯进料X轴错误代码
2013.08 BOOL  ; RK_02 U0_Y 电芯进料X轴错误代码
2013.09 BOOL  ; RK_02 U0_Y 电芯进料X轴错误代码
2013.10 BOOL  ; RK_02 U0_Y 电芯进料X轴错误代码
2013.11 BOOL  ; RK_02 U0_Y 电芯进料X轴错误代码
2013.12 BOOL  ; RK_02 U0_Y 电芯进料X轴错误代码
2013.13 BOOL  ; RK_02 U0_Y 电芯进料X轴错误代码
2013.14 BOOL  ; RK_02 U0_Y 电芯进料X轴错误代码
2013.15 BOOL  ; RK_02 U0_Y 电芯进料X轴错误代码
2014.00 BOOL  ; RK_02 U0_Z 电芯进料Z轴Not Use
2014.01 BOOL  ; RK_02 U0_Z 电芯进料Z轴Not Use
2014.02 BOOL  ; RK_02 U0_Z 电芯进料Z轴Not Use
2014.03 BOOL  ; RK_02 U0_Z 电芯进料Z轴Not Use
2014.04 BOOL  ; RK_02 U0_Z 电芯进料Z轴等待存储器操作标志位
2014.05 BOOL  ; RK_02 U0_Z 电芯进料Z轴定位结束标志位
2014.06 BOOL  ; RK_02 U0_Z 电芯进料Z轴无原点标志位
2014.07 BOOL  ; RK_02 U0_Z 电芯进料Z轴原点停止标志位
2014.08 BOOL  ; RK_02 U0_Z 电芯进料Z轴区域0监控标志位
2014.09 BOOL  ; RK_02 U0_Z 电芯进料Z轴区域1监控标志位
2014.10 BOOL  ; RK_02 U0_Z 电芯进料Z轴区域2监控标志位
2014.11 BOOL  ; RK_02 U0_Z 电芯进料Z轴示教完成标志位
2014.12 BOOL  ; RK_02 U0_Z 电芯进料Z轴错误标志位
2014.13 BOOL  ; RK_02 U0_Z 电芯进料Z轴忙标志位
2014.14 BOOL  ; RK_02 U0_Z 电芯进料Z轴数据传送标志
2014.15 BOOL  ; RK_02 U0_Z 电芯进料Z轴减速停止执行标志
2015.00 BOOL  ; RK_02 U0_Z 电芯进料Z轴Not Use
2015.01 BOOL  ; RK_02 U0_Z 电芯进料Z轴Not Use
2015.02 BOOL  ; RK_02 U0_Z 电芯进料Z轴Not Use
2015.03 BOOL  ; RK_02 U0_Z 电芯进料Z轴Not Use
2015.04 BOOL  ; RK_02 U0_Z 电芯进料Z轴Not Use
2015.05 BOOL  ; RK_02 U0_Z 电芯进料Z轴Not Use
2015.06 BOOL  ; RK_02 U0_Z 电芯进料Z轴Not Use
2015.07 BOOL  ; RK_02 U0_Z 电芯进料Z轴Not Use
2015.08 BOOL  ; RK_02 U0_Z 电芯进料Z轴CW极限输入信号
2015.09 BOOL  ; RK_02 U0_Z 电芯进料Z轴CCW极限输入信号
2015.10 BOOL  ; RK_02 U0_Z 电芯进料Z轴原点接近输入信号
2015.11 BOOL  ; RK_02 U0_Z 电芯进料Z轴原点输入信号
2015.12 BOOL  ; RK_02 U0_Z 电芯进料Z轴中断输入信号
2015.13 BOOL  ; RK_02 U0_Z 电芯进料Z轴紧急停止输入信号
2015.14 BOOL  ; RK_02 U0_Z 电芯进料Z轴定位完成信号
2015.15 BOOL  ; $?St$Bk?_#[5021] / RK_02 U0_Z 电芯进料Z轴偏差计数器复位输出 / 原点调整命令输出$?St$Bk?_#[5021]
2016 CHANNEL  ; RK_02 U0_Z 电芯进料Z轴错误代码
2016.00 BOOL  ; RK_02 U0_Z 电芯进料Z轴错误代码
2016.01 BOOL  ; RK_02 U0_Z 电芯进料Z轴错误代码
2016.02 BOOL  ; RK_02 U0_Z 电芯进料Z轴错误代码
2016.03 BOOL  ; RK_02 U0_Z 电芯进料Z轴错误代码
2016.04 BOOL  ; RK_02 U0_Z 电芯进料Z轴错误代码
2016.05 BOOL  ; RK_02 U0_Z 电芯进料Z轴错误代码
2016.06 BOOL  ; RK_02 U0_Z 电芯进料Z轴错误代码
2016.07 BOOL  ; RK_02 U0_Z 电芯进料Z轴错误代码
2016.08 BOOL  ; RK_02 U0_Z 电芯进料Z轴错误代码
2016.09 BOOL  ; RK_02 U0_Z 电芯进料Z轴错误代码
2016.10 BOOL  ; RK_02 U0_Z 电芯进料Z轴错误代码
2016.11 BOOL  ; RK_02 U0_Z 电芯进料Z轴错误代码
2016.12 BOOL  ; RK_02 U0_Z 电芯进料Z轴错误代码
2016.13 BOOL  ; RK_02 U0_Z 电芯进料Z轴错误代码
2016.14 BOOL  ; RK_02 U0_Z 电芯进料Z轴错误代码
2016.15 BOOL  ; RK_02 U0_Z 电芯进料Z轴错误代码
2017.00 BOOL  ; RK_03 U0_U 电芯上料X轴Not Use
2017.01 BOOL  ; RK_03 U0_U 电芯上料X轴Not Use
2017.02 BOOL  ; RK_03 U0_U 电芯上料X轴Not Use
2017.03 BOOL  ; RK_03 U0_U 电芯上料X轴Not Use
2017.04 BOOL  ; RK_03 U0_U 电芯上料X轴等待存储器操作标志位
2017.05 BOOL  ; RK_03 U0_U 电芯上料X轴定位结束标志位
2017.06 BOOL  ; RK_03 U0_U 电芯上料X轴无原点标志位
2017.07 BOOL  ; RK_03 U0_U 电芯上料X轴原点停止标志位
2017.08 BOOL  ; RK_03 U0_U 电芯上料X轴区域0监控标志位
2017.09 BOOL  ; RK_03 U0_U 电芯上料X轴区域1监控标志位
2017.10 BOOL  ; RK_03 U0_U 电芯上料X轴区域2监控标志位
2017.11 BOOL  ; RK_03 U0_U 电芯上料X轴示教完成标志位
2017.12 BOOL  ; RK_03 U0_U 电芯上料X轴错误标志位
2017.13 BOOL  ; RK_03 U0_U 电芯上料X轴忙标志位
2017.14 BOOL  ; RK_03 U0_U 电芯上料X轴数据传送标志
2017.15 BOOL  ; RK_03 U0_U 电芯上料X轴减速停止执行标志
2018.00 BOOL  ; RK_03 U0_U 电芯上料X轴Not Use
2018.01 BOOL  ; RK_03 U0_U 电芯上料X轴Not Use
2018.02 BOOL  ; RK_03 U0_U 电芯上料X轴Not Use
2018.03 BOOL  ; RK_03 U0_U 电芯上料X轴Not Use
2018.04 BOOL  ; RK_03 U0_U 电芯上料X轴Not Use
2018.05 BOOL  ; RK_03 U0_U 电芯上料X轴Not Use
2018.06 BOOL  ; RK_03 U0_U 电芯上料X轴Not Use
2018.07 BOOL  ; RK_03 U0_U 电芯上料X轴Not Use
2018.08 BOOL  ; RK_03 U0_U 电芯上料X轴CW极限输入信号
2018.09 BOOL  ; RK_03 U0_U 电芯上料X轴CCW极限输入信号
2018.10 BOOL  ; RK_03 U0_U 电芯上料X轴原点接近输入信号
2018.11 BOOL  ; RK_03 U0_U 电芯上料X轴原点输入信号
2018.12 BOOL  ; RK_03 U0_U 电芯上料X轴中断输入信号
2018.13 BOOL  ; RK_03 U0_U 电芯上料X轴紧急停止输入信号
2018.14 BOOL  ; RK_03 U0_U 电芯上料X轴定位完成信号
2018.15 BOOL  ; $?St$Bk?_#[5022] / RK_03 U0_U 电芯上料X轴偏差计数器复位输出 / 原点调整命令输出$?St$Bk?_#[5022]
2019 CHANNEL  ; RK_03 U0_U 电芯上料X轴错误代码
2019.00 BOOL  ; RK_03 U0_U 电芯上料X轴错误代码
2019.01 BOOL  ; RK_03 U0_U 电芯上料X轴错误代码
2019.02 BOOL  ; RK_03 U0_U 电芯上料X轴错误代码
2019.03 BOOL  ; RK_03 U0_U 电芯上料X轴错误代码
2019.04 BOOL  ; RK_03 U0_U 电芯上料X轴错误代码
2019.05 BOOL  ; RK_03 U0_U 电芯上料X轴错误代码
2019.06 BOOL  ; RK_03 U0_U 电芯上料X轴错误代码
2019.07 BOOL  ; RK_03 U0_U 电芯上料X轴错误代码
2019.08 BOOL  ; RK_03 U0_U 电芯上料X轴错误代码
2019.09 BOOL  ; RK_03 U0_U 电芯上料X轴错误代码
2019.10 BOOL  ; RK_03 U0_U 电芯上料X轴错误代码
2019.11 BOOL  ; RK_03 U0_U 电芯上料X轴错误代码
2019.12 BOOL  ; RK_03 U0_U 电芯上料X轴错误代码
2019.13 BOOL  ; RK_03 U0_U 电芯上料X轴错误代码
2019.14 BOOL  ; RK_03 U0_U 电芯上料X轴错误代码
2019.15 BOOL  ; RK_03 U0_U 电芯上料X轴错误代码
201.00 BOOL  ; 整机在初始位
2020.00 BOOL  ; RK_05 U2_X #1入壳Y轴序列号使能
2020.01 BOOL  ; RK_05 U2_X #1入壳Y轴启动
2020.02 BOOL  ; RK_05 U2_X #1入壳Y轴独立启动
2020.03 BOOL  ; RK_05 U2_X #1入壳Y轴绝对移动
2020.04 BOOL  ; RK_05 U2_X #1入壳Y轴相对移动
2020.05 BOOL  ; RK_05 U2_X #1入壳Y轴中断进给
2020.06 BOOL  ; RK_05 U2_X #1入壳Y轴原点搜索
2020.07 BOOL  ; RK_05 U2_X #1入壳Y轴原点返回
2020.08 BOOL  ; RK_05 U2_X #1入壳Y轴当前位置预置
2020.09 BOOL  ; RK_05 U2_X #1入壳Y轴点动
2020.10 BOOL  ; RK_05 U2_X #1入壳Y轴方向定义
2020.11 BOOL  ; RK_05 U2_X #1入壳Y轴示教
2020.12 BOOL  ; RK_05 U2_X #1入壳Y轴释放禁止/复位
2020.13 BOOL  ; $?St$Bk?_#[5023] / RK_05 U2_X #1入壳Y轴偏差计数器复位输出/ / 原点调整命令输出$?St$Bk?_#[5023]
2020.14 BOOL  ; RK_05 U2_X #1入壳Y轴激活倍率
2020.15 BOOL  ; RK_05 U2_X #1入壳Y轴停止
2021.00 BOOL  ; RK_05 U2_X #1入壳Y轴Not Use
2021.01 BOOL  ; RK_05 U2_X #1入壳Y轴Not Use
2021.02 BOOL  ; RK_05 U2_X #1入壳Y轴Not Use
2021.03 BOOL  ; RK_05 U2_X #1入壳Y轴Not Use
2021.04 BOOL  ; RK_05 U2_X #1入壳Y轴Not Use
2021.05 BOOL  ; RK_05 U2_X #1入壳Y轴Not Use
2021.06 BOOL  ; RK_05 U2_X #1入壳Y轴Not Use
2021.07 BOOL  ; RK_05 U2_X #1入壳Y轴Not Use
2021.08 BOOL  ; RK_05 U2_X #1入壳Y轴强迫中断
2021.09 BOOL  ; RK_05 U2_X #1入壳Y轴Not Use
2021.10 BOOL  ; RK_05 U2_X #1入壳Y轴Not Use
2021.11 BOOL  ; RK_05 U2_X #1入壳Y轴Not Use
2021.12 BOOL  ; RK_05 U2_X #1入壳Y轴写数据
2021.13 BOOL  ; RK_05 U2_X #1入壳Y轴读数据
2021.14 BOOL  ; RK_05 U2_X #1入壳Y轴存数据
2021.15 BOOL  ; RK_05 U2_X #1入壳Y轴Not Use
2022.00 BOOL  ; RK_05 U2_Y #2入壳Y轴序列号使能
2022.01 BOOL  ; RK_05 U2_Y #2入壳Y轴启动
2022.02 BOOL  ; RK_05 U2_Y #2入壳Y轴独立启动
2022.03 BOOL  ; RK_05 U2_Y #2入壳Y轴绝对移动
2022.04 BOOL  ; RK_05 U2_Y #2入壳Y轴相对移动
2022.05 BOOL  ; RK_05 U2_Y #2入壳Y轴中断进给
2022.06 BOOL  ; RK_05 U2_Y #2入壳Y轴原点搜索
2022.07 BOOL  ; RK_05 U2_Y #2入壳Y轴原点返回
2022.08 BOOL  ; RK_05 U2_Y #2入壳Y轴当前位置预置
2022.09 BOOL  ; RK_05 U2_Y #2入壳Y轴点动
2022.10 BOOL  ; RK_05 U2_Y #2入壳Y轴方向定义
2022.11 BOOL  ; RK_05 U2_Y #2入壳Y轴示教
2022.12 BOOL  ; RK_05 U2_Y #2入壳Y轴释放禁止/复位
2022.13 BOOL  ; $?St$Bk?_#[5024] / RK_05 U2_Y #2入壳Y轴偏差计数器复位输出/ / 原点调整命令输出$?St$Bk?_#[5024]
2022.14 BOOL  ; RK_05 U2_Y #2入壳Y轴激活倍率
2022.15 BOOL  ; RK_05 U2_Y #2入壳Y轴停止
2023.00 BOOL  ; RK_05 U2_Y #2入壳Y轴Not Use
2023.01 BOOL  ; RK_05 U2_Y #2入壳Y轴Not Use
2023.02 BOOL  ; RK_05 U2_Y #2入壳Y轴Not Use
2023.03 BOOL  ; RK_05 U2_Y #2入壳Y轴Not Use
2023.04 BOOL  ; RK_05 U2_Y #2入壳Y轴Not Use
2023.05 BOOL  ; RK_05 U2_Y #2入壳Y轴Not Use
2023.06 BOOL  ; RK_05 U2_Y #2入壳Y轴Not Use
2023.07 BOOL  ; RK_05 U2_Y #2入壳Y轴Not Use
2023.08 BOOL  ; RK_05 U2_Y #2入壳Y轴强迫中断
2023.09 BOOL  ; RK_05 U2_Y #2入壳Y轴Not Use
2023.10 BOOL  ; RK_05 U2_Y #2入壳Y轴Not Use
2023.11 BOOL  ; RK_05 U2_Y #2入壳Y轴Not Use
2023.12 BOOL  ; RK_05 U2_Y #2入壳Y轴写数据
2023.13 BOOL  ; RK_05 U2_Y #2入壳Y轴读数据
2023.14 BOOL  ; RK_05 U2_Y #2入壳Y轴存数据
2023.15 BOOL  ; RK_05 U2_Y #2入壳Y轴Not Use
2028.00 BOOL  ; RK_05 U2_X #1入壳Y轴Not Use
2028.01 BOOL  ; RK_05 U2_X #1入壳Y轴Not Use
2028.02 BOOL  ; RK_05 U2_X #1入壳Y轴Not Use
2028.03 BOOL  ; RK_05 U2_X #1入壳Y轴Not Use
2028.04 BOOL  ; RK_05 U2_X #1入壳Y轴等待存储器操作标志位
2028.05 BOOL  ; RK_05 U2_X #1入壳Y轴定位结束标志位
2028.06 BOOL  ; RK_05 U2_X #1入壳Y轴无原点标志位
2028.07 BOOL  ; RK_05 U2_X #1入壳Y轴原点停止标志位
2028.08 BOOL  ; RK_05 U2_X #1入壳Y轴区域0监控标志位
2028.09 BOOL  ; RK_05 U2_X #1入壳Y轴区域1监控标志位
2028.10 BOOL  ; RK_05 U2_X #1入壳Y轴区域2监控标志位
2028.11 BOOL  ; RK_05 U2_X #1入壳Y轴示教完成标志位
2028.12 BOOL  ; RK_05 U2_X #1入壳Y轴错误标志位
2028.13 BOOL  ; RK_05 U2_X #1入壳Y轴忙标志位
2028.14 BOOL  ; RK_05 U2_X #1入壳Y轴数据传送标志
2028.15 BOOL  ; RK_05 U2_X #1入壳Y轴减速停止执行标志
2029.00 BOOL  ; RK_05 U2_X #1入壳Y轴Not Use
2029.01 BOOL  ; RK_05 U2_X #1入壳Y轴Not Use
2029.02 BOOL  ; RK_05 U2_X #1入壳Y轴Not Use
2029.03 BOOL  ; RK_05 U2_X #1入壳Y轴Not Use
2029.04 BOOL  ; RK_05 U2_X #1入壳Y轴Not Use
2029.05 BOOL  ; RK_05 U2_X #1入壳Y轴Not Use
2029.06 BOOL  ; RK_05 U2_X #1入壳Y轴Not Use
2029.07 BOOL  ; RK_05 U2_X #1入壳Y轴Not Use
2029.08 BOOL  ; RK_05 U2_X #1入壳Y轴CW极限输入信号
2029.09 BOOL  ; RK_05 U2_X #1入壳Y轴CCW极限输入信号
2029.10 BOOL  ; RK_05 U2_X #1入壳Y轴原点接近输入信号
2029.11 BOOL  ; RK_05 U2_X #1入壳Y轴原点输入信号
2029.12 BOOL  ; RK_05 U2_X #1入壳Y轴中断输入信号
2029.13 BOOL  ; RK_05 U2_X #1入壳Y轴紧急停止输入信号
2029.14 BOOL  ; RK_05 U2_X #1入壳Y轴定位完成信号
2029.15 BOOL  ; $?St$Bk?_#[5025] / RK_05 U2_X #1入壳Y轴偏差计数器复位输出 / 原点调整命令输出$?St$Bk?_#[5025]
2030 CHANNEL  ; RK_05 U2_X #1入壳Y轴错误代码
2030.00 BOOL  ; RK_05 U2_X #1入壳Y轴错误代码
2030.01 BOOL  ; RK_05 U2_X #1入壳Y轴错误代码
2030.02 BOOL  ; RK_05 U2_X #1入壳Y轴错误代码
2030.03 BOOL  ; RK_05 U2_X #1入壳Y轴错误代码
2030.04 BOOL  ; RK_05 U2_X #1入壳Y轴错误代码
2030.05 BOOL  ; RK_05 U2_X #1入壳Y轴错误代码
2030.06 BOOL  ; RK_05 U2_X #1入壳Y轴错误代码
2030.07 BOOL  ; RK_05 U2_X #1入壳Y轴错误代码
2030.08 BOOL  ; RK_05 U2_X #1入壳Y轴错误代码
2030.09 BOOL  ; RK_05 U2_X #1入壳Y轴错误代码
2030.10 BOOL  ; RK_05 U2_X #1入壳Y轴错误代码
2030.11 BOOL  ; RK_05 U2_X #1入壳Y轴错误代码
2030.12 BOOL  ; RK_05 U2_X #1入壳Y轴错误代码
2030.13 BOOL  ; RK_05 U2_X #1入壳Y轴错误代码
2030.14 BOOL  ; RK_05 U2_X #1入壳Y轴错误代码
2030.15 BOOL  ; RK_05 U2_X #1入壳Y轴错误代码
2031.00 BOOL  ; RK_05 U2_Y #2入壳Y轴Not Use
2031.01 BOOL  ; RK_05 U2_Y #2入壳Y轴Not Use
2031.02 BOOL  ; RK_05 U2_Y #2入壳Y轴Not Use
2031.03 BOOL  ; RK_05 U2_Y #2入壳Y轴Not Use
2031.04 BOOL  ; RK_05 U2_Y #2入壳Y轴等待存储器操作标志位
2031.05 BOOL  ; RK_05 U2_Y #2入壳Y轴定位结束标志位
2031.06 BOOL  ; RK_05 U2_Y #2入壳Y轴无原点标志位
2031.07 BOOL  ; RK_05 U2_Y #2入壳Y轴原点停止标志位
2031.08 BOOL  ; RK_05 U2_Y #2入壳Y轴区域0监控标志位
2031.09 BOOL  ; RK_05 U2_Y #2入壳Y轴区域1监控标志位
2031.10 BOOL  ; RK_05 U2_Y #2入壳Y轴区域2监控标志位
2031.11 BOOL  ; RK_05 U2_Y #2入壳Y轴示教完成标志位
2031.12 BOOL  ; RK_05 U2_Y #2入壳Y轴错误标志位
2031.13 BOOL  ; RK_05 U2_Y #2入壳Y轴忙标志位
2031.14 BOOL  ; RK_05 U2_Y #2入壳Y轴数据传送标志
2031.15 BOOL  ; RK_05 U2_Y #2入壳Y轴减速停止执行标志
2032.00 BOOL  ; RK_05 U2_Y #2入壳Y轴Not Use
2032.01 BOOL  ; RK_05 U2_Y #2入壳Y轴Not Use
2032.02 BOOL  ; RK_05 U2_Y #2入壳Y轴Not Use
2032.03 BOOL  ; RK_05 U2_Y #2入壳Y轴Not Use
2032.04 BOOL  ; RK_05 U2_Y #2入壳Y轴Not Use
2032.05 BOOL  ; RK_05 U2_Y #2入壳Y轴Not Use
2032.06 BOOL  ; RK_05 U2_Y #2入壳Y轴Not Use
2032.07 BOOL  ; RK_05 U2_Y #2入壳Y轴Not Use
2032.08 BOOL  ; RK_05 U2_Y #2入壳Y轴CW极限输入信号
2032.09 BOOL  ; RK_05 U2_Y #2入壳Y轴CCW极限输入信号
2032.10 BOOL  ; RK_05 U2_Y #2入壳Y轴原点接近输入信号
2032.11 BOOL  ; RK_05 U2_Y #2入壳Y轴原点输入信号
2032.12 BOOL  ; RK_05 U2_Y #2入壳Y轴中断输入信号
2032.13 BOOL  ; RK_05 U2_Y #2入壳Y轴紧急停止输入信号
2032.14 BOOL  ; RK_05 U2_Y #2入壳Y轴定位完成信号
2032.15 BOOL  ; $?St$Bk?_#[5026] / RK_05 U2_Y #2入壳Y轴偏差计数器复位输出 / 原点调整命令输出$?St$Bk?_#[5026]
2033 CHANNEL  ; RK_05 U2_Y #2入壳Y轴错误代码
2033.00 BOOL  ; RK_05 U2_Y #2入壳Y轴错误代码
2033.01 BOOL  ; RK_05 U2_Y #2入壳Y轴错误代码
2033.02 BOOL  ; RK_05 U2_Y #2入壳Y轴错误代码
2033.03 BOOL  ; RK_05 U2_Y #2入壳Y轴错误代码
2033.04 BOOL  ; RK_05 U2_Y #2入壳Y轴错误代码
2033.05 BOOL  ; RK_05 U2_Y #2入壳Y轴错误代码
2033.06 BOOL  ; RK_05 U2_Y #2入壳Y轴错误代码
2033.07 BOOL  ; RK_05 U2_Y #2入壳Y轴错误代码
2033.08 BOOL  ; RK_05 U2_Y #2入壳Y轴错误代码
2033.09 BOOL  ; RK_05 U2_Y #2入壳Y轴错误代码
2033.10 BOOL  ; RK_05 U2_Y #2入壳Y轴错误代码
2033.11 BOOL  ; RK_05 U2_Y #2入壳Y轴错误代码
2033.12 BOOL  ; RK_05 U2_Y #2入壳Y轴错误代码
2033.13 BOOL  ; RK_05 U2_Y #2入壳Y轴错误代码
2033.14 BOOL  ; RK_05 U2_Y #2入壳Y轴错误代码
2033.15 BOOL  ; RK_05 U2_Y #2入壳Y轴错误代码
2040.00 BOOL  ; RK_12 U4_X 预焊上下料X轴序列号使能
2040.01 BOOL  ; RK_12 U4_X 预焊上下料X轴启动
2040.02 BOOL  ; RK_12 U4_X 预焊上下料X轴独立启动
2040.03 BOOL  ; RK_12 U4_X 预焊上下料X轴绝对移动
2040.04 BOOL  ; RK_12 U4_X 预焊上下料X轴相对移动
2040.05 BOOL  ; RK_12 U4_X 预焊上下料X轴中断进给
2040.06 BOOL  ; RK_12 U4_X 预焊上下料X轴原点搜索
2040.07 BOOL  ; RK_12 U4_X 预焊上下料X轴原点返回
2040.08 BOOL  ; RK_12 U4_X 预焊上下料X轴当前位置预置
2040.09 BOOL  ; RK_12 U4_X 预焊上下料X轴点动
2040.10 BOOL  ; RK_12 U4_X 预焊上下料X轴方向定义
2040.11 BOOL  ; RK_12 U4_X 预焊上下料X轴示教
2040.12 BOOL  ; RK_12 U4_X 预焊上下料X轴释放禁止/复位
2040.13 BOOL  ; $?St$Bk?_#[5027] / RK_12 U4_X 预焊上下料X轴偏差计数器复位输出/ / 原点调整命令输出$?St$Bk?_#[5027]
2040.14 BOOL  ; RK_12 U4_X 预焊上下料X轴激活倍率
2040.15 BOOL  ; RK_12 U4_X 预焊上下料X轴停止
2041.00 BOOL  ; RK_12 U4_X 预焊上下料X轴Not Use
2041.01 BOOL  ; RK_12 U4_X 预焊上下料X轴Not Use
2041.02 BOOL  ; RK_12 U4_X 预焊上下料X轴Not Use
2041.03 BOOL  ; RK_12 U4_X 预焊上下料X轴Not Use
2041.04 BOOL  ; RK_12 U4_X 预焊上下料X轴Not Use
2041.05 BOOL  ; RK_12 U4_X 预焊上下料X轴Not Use
2041.06 BOOL  ; RK_12 U4_X 预焊上下料X轴Not Use
2041.07 BOOL  ; RK_12 U4_X 预焊上下料X轴Not Use
2041.08 BOOL  ; RK_12 U4_X 预焊上下料X轴强迫中断
2041.09 BOOL  ; RK_12 U4_X 预焊上下料X轴Not Use
2041.10 BOOL  ; RK_12 U4_X 预焊上下料X轴Not Use
2041.11 BOOL  ; RK_12 U4_X 预焊上下料X轴Not Use
2041.12 BOOL  ; RK_12 U4_X 预焊上下料X轴写数据
2041.13 BOOL  ; RK_12 U4_X 预焊上下料X轴读数据
2041.14 BOOL  ; RK_12 U4_X 预焊上下料X轴存数据
2041.15 BOOL  ; RK_12 U4_X 预焊上下料X轴Not Use
2042.00 BOOL  ; RK_12 U4_Y 预焊上料Z轴序列号使能
2042.01 BOOL  ; RK_12 U4_Y 预焊上料Z轴启动
2042.02 BOOL  ; RK_12 U4_Y 预焊上料Z轴独立启动
2042.03 BOOL  ; RK_12 U4_Y 预焊上料Z轴绝对移动
2042.04 BOOL  ; RK_12 U4_Y 预焊上料Z轴相对移动
2042.05 BOOL  ; RK_12 U4_Y 预焊上料Z轴中断进给
2042.06 BOOL  ; RK_12 U4_Y 预焊上料Z轴原点搜索
2042.07 BOOL  ; RK_12 U4_Y 预焊上料Z轴原点返回
2042.08 BOOL  ; RK_12 U4_Y 预焊上料Z轴当前位置预置
2042.09 BOOL  ; RK_12 U4_Y 预焊上料Z轴点动
2042.10 BOOL  ; RK_12 U4_Y 预焊上料Z轴方向定义
2042.11 BOOL  ; RK_12 U4_Y 预焊上料Z轴示教
2042.12 BOOL  ; RK_12 U4_Y 预焊上料Z轴释放禁止/复位
2042.13 BOOL  ; $?St$Bk?_#[5028] / RK_12 U4_Y 预焊上料Z轴偏差计数器复位输出/ / 原点调整命令输出$?St$Bk?_#[5028]
2042.14 BOOL  ; RK_12 U4_Y 预焊上料Z轴激活倍率
2042.15 BOOL  ; RK_12 U4_Y 预焊上料Z轴停止
2043.00 BOOL  ; RK_12 U4_Y 预焊上料Z轴Not Use
2043.01 BOOL  ; RK_12 U4_Y 预焊上料Z轴Not Use
2043.02 BOOL  ; RK_12 U4_Y 预焊上料Z轴Not Use
2043.03 BOOL  ; RK_12 U4_Y 预焊上料Z轴Not Use
2043.04 BOOL  ; RK_12 U4_Y 预焊上料Z轴Not Use
2043.05 BOOL  ; RK_12 U4_Y 预焊上料Z轴Not Use
2043.06 BOOL  ; RK_12 U4_Y 预焊上料Z轴Not Use
2043.07 BOOL  ; RK_12 U4_Y 预焊上料Z轴Not Use
2043.08 BOOL  ; RK_12 U4_Y 预焊上料Z轴强迫中断
2043.09 BOOL  ; RK_12 U4_Y 预焊上料Z轴Not Use
2043.10 BOOL  ; RK_12 U4_Y 预焊上料Z轴Not Use
2043.11 BOOL  ; RK_12 U4_Y 预焊上料Z轴Not Use
2043.12 BOOL  ; RK_12 U4_Y 预焊上料Z轴写数据
2043.13 BOOL  ; RK_12 U4_Y 预焊上料Z轴读数据
2043.14 BOOL  ; RK_12 U4_Y 预焊上料Z轴存数据
2043.15 BOOL  ; RK_12 U4_Y 预焊上料Z轴Not Use
2044.00 BOOL  ; RK_12 U4_Z 预焊下料Z轴序列号使能
2044.01 BOOL  ; RK_12 U4_Z 预焊下料Z轴启动
2044.02 BOOL  ; RK_12 U4_Z 预焊下料Z轴独立启动
2044.03 BOOL  ; RK_12 U4_Z 预焊下料Z轴绝对移动
2044.04 BOOL  ; RK_12 U4_Z 预焊下料Z轴相对移动
2044.05 BOOL  ; RK_12 U4_Z 预焊下料Z轴中断进给
2044.06 BOOL  ; RK_12 U4_Z 预焊下料Z轴原点搜索
2044.07 BOOL  ; RK_12 U4_Z 预焊下料Z轴原点返回
2044.08 BOOL  ; RK_12 U4_Z 预焊下料Z轴当前位置预置
2044.09 BOOL  ; RK_12 U4_Z 预焊下料Z轴点动
2044.10 BOOL  ; RK_12 U4_Z 预焊下料Z轴方向定义
2044.11 BOOL  ; RK_12 U4_Z 预焊下料Z轴示教
2044.12 BOOL  ; RK_12 U4_Z 预焊下料Z轴释放禁止/复位
2044.13 BOOL  ; $?St$Bk?_#[5029] / RK_12 U4_Z 预焊下料Z轴偏差计数器复位输出/ / 原点调整命令输出$?St$Bk?_#[5029]
2044.14 BOOL  ; RK_12 U4_Z 预焊下料Z轴激活倍率
2044.15 BOOL  ; RK_12 U4_Z 预焊下料Z轴停止
2045.00 BOOL  ; RK_12 U4_Z 预焊下料Z轴Not Use
2045.01 BOOL  ; RK_12 U4_Z 预焊下料Z轴Not Use
2045.02 BOOL  ; RK_12 U4_Z 预焊下料Z轴Not Use
2045.03 BOOL  ; RK_12 U4_Z 预焊下料Z轴Not Use
2045.04 BOOL  ; RK_12 U4_Z 预焊下料Z轴Not Use
2045.05 BOOL  ; RK_12 U4_Z 预焊下料Z轴Not Use
2045.06 BOOL  ; RK_12 U4_Z 预焊下料Z轴Not Use
2045.07 BOOL  ; RK_12 U4_Z 预焊下料Z轴Not Use
2045.08 BOOL  ; RK_12 U4_Z 预焊下料Z轴强迫中断
2045.09 BOOL  ; RK_12 U4_Z 预焊下料Z轴Not Use
2045.10 BOOL  ; RK_12 U4_Z 预焊下料Z轴Not Use
2045.11 BOOL  ; RK_12 U4_Z 预焊下料Z轴Not Use
2045.12 BOOL  ; RK_12 U4_Z 预焊下料Z轴写数据
2045.13 BOOL  ; RK_12 U4_Z 预焊下料Z轴读数据
2045.14 BOOL  ; RK_12 U4_Z 预焊下料Z轴存数据
2045.15 BOOL  ; RK_12 U4_Z 预焊下料Z轴Not Use
2046.00 BOOL  ; RK_13 U4_U #1移载Y轴序列号使能
2046.01 BOOL  ; RK_13 U4_U #1移载Y轴启动
2046.02 BOOL  ; RK_13 U4_U #1移载Y轴独立启动
2046.03 BOOL  ; RK_13 U4_U #1移载Y轴绝对移动
2046.04 BOOL  ; RK_13 U4_U #1移载Y轴相对移动
2046.05 BOOL  ; RK_13 U4_U #1移载Y轴中断进给
2046.06 BOOL  ; RK_13 U4_U #1移载Y轴原点搜索
2046.07 BOOL  ; RK_13 U4_U #1移载Y轴原点返回
2046.08 BOOL  ; RK_13 U4_U #1移载Y轴当前位置预置
2046.09 BOOL  ; RK_13 U4_U #1移载Y轴点动
2046.10 BOOL  ; RK_13 U4_U #1移载Y轴方向定义
2046.11 BOOL  ; RK_13 U4_U #1移载Y轴示教
2046.12 BOOL  ; RK_13 U4_U #1移载Y轴释放禁止/复位
2046.13 BOOL  ; $?St$Bk?_#[5030] / RK_13 U4_U #1移载Y轴偏差计数器复位输出/ / 原点调整命令输出$?St$Bk?_#[5030]
2046.14 BOOL  ; RK_13 U4_U #1移载Y轴激活倍率
2046.15 BOOL  ; RK_13 U4_U #1移载Y轴停止
2047.00 BOOL  ; RK_13 U4_U #1移载Y轴Not Use
2047.01 BOOL  ; RK_13 U4_U #1移载Y轴Not Use
2047.02 BOOL  ; RK_13 U4_U #1移载Y轴Not Use
2047.03 BOOL  ; RK_13 U4_U #1移载Y轴Not Use
2047.04 BOOL  ; RK_13 U4_U #1移载Y轴Not Use
2047.05 BOOL  ; RK_13 U4_U #1移载Y轴Not Use
2047.06 BOOL  ; RK_13 U4_U #1移载Y轴Not Use
2047.07 BOOL  ; RK_13 U4_U #1移载Y轴Not Use
2047.08 BOOL  ; RK_13 U4_U #1移载Y轴强迫中断
2047.09 BOOL  ; RK_13 U4_U #1移载Y轴Not Use
2047.10 BOOL  ; RK_13 U4_U #1移载Y轴Not Use
2047.11 BOOL  ; RK_13 U4_U #1移载Y轴Not Use
2047.12 BOOL  ; RK_13 U4_U #1移载Y轴写数据
2047.13 BOOL  ; RK_13 U4_U #1移载Y轴读数据
2047.14 BOOL  ; RK_13 U4_U #1移载Y轴存数据
2047.15 BOOL  ; RK_13 U4_U #1移载Y轴Not Use
2048.00 BOOL  ; RK_12 U4_X 预焊上下料X轴Not Use
2048.01 BOOL  ; RK_12 U4_X 预焊上下料X轴Not Use
2048.02 BOOL  ; RK_12 U4_X 预焊上下料X轴Not Use
2048.03 BOOL  ; RK_12 U4_X 预焊上下料X轴Not Use
2048.04 BOOL  ; RK_12 U4_X 预焊上下料X轴等待存储器操作标志位
2048.05 BOOL  ; RK_12 U4_X 预焊上下料X轴定位结束标志位
2048.06 BOOL  ; RK_12 U4_X 预焊上下料X轴无原点标志位
2048.07 BOOL  ; RK_12 U4_X 预焊上下料X轴原点停止标志位
2048.08 BOOL  ; RK_12 U4_X 预焊上下料X轴区域0监控标志位
2048.09 BOOL  ; RK_12 U4_X 预焊上下料X轴区域1监控标志位
2048.10 BOOL  ; RK_12 U4_X 预焊上下料X轴区域2监控标志位
2048.11 BOOL  ; RK_12 U4_X 预焊上下料X轴示教完成标志位
2048.12 BOOL  ; RK_12 U4_X 预焊上下料X轴错误标志位
2048.13 BOOL  ; RK_12 U4_X 预焊上下料X轴忙标志位
2048.14 BOOL  ; RK_12 U4_X 预焊上下料X轴数据传送标志
2048.15 BOOL  ; RK_12 U4_X 预焊上下料X轴减速停止执行标志
2049.00 BOOL  ; RK_12 U4_X 预焊上下料X轴Not Use
2049.01 BOOL  ; RK_12 U4_X 预焊上下料X轴Not Use
2049.02 BOOL  ; RK_12 U4_X 预焊上下料X轴Not Use
2049.03 BOOL  ; RK_12 U4_X 预焊上下料X轴Not Use
2049.04 BOOL  ; RK_12 U4_X 预焊上下料X轴Not Use
2049.05 BOOL  ; RK_12 U4_X 预焊上下料X轴Not Use
2049.06 BOOL  ; RK_12 U4_X 预焊上下料X轴Not Use
2049.07 BOOL  ; RK_12 U4_X 预焊上下料X轴Not Use
2049.08 BOOL  ; RK_12 U4_X 预焊上下料X轴CW极限输入信号
2049.09 BOOL  ; RK_12 U4_X 预焊上下料X轴CCW极限输入信号
2049.10 BOOL  ; RK_12 U4_X 预焊上下料X轴原点接近输入信号
2049.11 BOOL  ; RK_12 U4_X 预焊上下料X轴原点输入信号
2049.12 BOOL  ; RK_12 U4_X 预焊上下料X轴中断输入信号
2049.13 BOOL  ; RK_12 U4_X 预焊上下料X轴紧急停止输入信号
2049.14 BOOL  ; RK_12 U4_X 预焊上下料X轴定位完成信号
2049.15 BOOL  ; $?St$Bk?_#[5031] / RK_12 U4_X 预焊上下料X轴偏差计数器复位输出 / 原点调整命令输出$?St$Bk?_#[5031]
2050 CHANNEL  ; RK_12 U4_X 预焊上下料X轴错误代码
2050.00 BOOL  ; RK_12 U4_X 预焊上下料X轴错误代码
2050.01 BOOL  ; RK_12 U4_X 预焊上下料X轴错误代码
2050.02 BOOL  ; RK_12 U4_X 预焊上下料X轴错误代码
2050.03 BOOL  ; RK_12 U4_X 预焊上下料X轴错误代码
2050.04 BOOL  ; RK_12 U4_X 预焊上下料X轴错误代码
2050.05 BOOL  ; RK_12 U4_X 预焊上下料X轴错误代码
2050.06 BOOL  ; RK_12 U4_X 预焊上下料X轴错误代码
2050.07 BOOL  ; RK_12 U4_X 预焊上下料X轴错误代码
2050.08 BOOL  ; RK_12 U4_X 预焊上下料X轴错误代码
2050.09 BOOL  ; RK_12 U4_X 预焊上下料X轴错误代码
2050.10 BOOL  ; RK_12 U4_X 预焊上下料X轴错误代码
2050.11 BOOL  ; RK_12 U4_X 预焊上下料X轴错误代码
2050.12 BOOL  ; RK_12 U4_X 预焊上下料X轴错误代码
2050.13 BOOL  ; RK_12 U4_X 预焊上下料X轴错误代码
2050.14 BOOL  ; RK_12 U4_X 预焊上下料X轴错误代码
2050.15 BOOL  ; RK_12 U4_X 预焊上下料X轴错误代码
2051.00 BOOL  ; RK_12 U4_Y 预焊上料Z轴Not Use
2051.01 BOOL  ; RK_12 U4_Y 预焊上料Z轴Not Use
2051.02 BOOL  ; RK_12 U4_Y 预焊上料Z轴Not Use
2051.03 BOOL  ; RK_12 U4_Y 预焊上料Z轴Not Use
2051.04 BOOL  ; RK_12 U4_Y 预焊上料Z轴等待存储器操作标志位
2051.05 BOOL  ; RK_12 U4_Y 预焊上料Z轴定位结束标志位
2051.06 BOOL  ; RK_12 U4_Y 预焊上料Z轴无原点标志位
2051.07 BOOL  ; RK_12 U4_Y 预焊上料Z轴原点停止标志位
2051.08 BOOL  ; RK_12 U4_Y 预焊上料Z轴区域0监控标志位
2051.09 BOOL  ; RK_12 U4_Y 预焊上料Z轴区域1监控标志位
2051.10 BOOL  ; RK_12 U4_Y 预焊上料Z轴区域2监控标志位
2051.11 BOOL  ; RK_12 U4_Y 预焊上料Z轴示教完成标志位
2051.12 BOOL  ; RK_12 U4_Y 预焊上料Z轴错误标志位
2051.13 BOOL  ; RK_12 U4_Y 预焊上料Z轴忙标志位
2051.14 BOOL  ; RK_12 U4_Y 预焊上料Z轴数据传送标志
2051.15 BOOL  ; RK_12 U4_Y 预焊上料Z轴减速停止执行标志
2052.00 BOOL  ; RK_12 U4_Y 预焊上料Z轴Not Use
2052.01 BOOL  ; RK_12 U4_Y 预焊上料Z轴Not Use
2052.02 BOOL  ; RK_12 U4_Y 预焊上料Z轴Not Use
2052.03 BOOL  ; RK_12 U4_Y 预焊上料Z轴Not Use
2052.04 BOOL  ; RK_12 U4_Y 预焊上料Z轴Not Use
2052.05 BOOL  ; RK_12 U4_Y 预焊上料Z轴Not Use
2052.06 BOOL  ; RK_12 U4_Y 预焊上料Z轴Not Use
2052.07 BOOL  ; RK_12 U4_Y 预焊上料Z轴Not Use
2052.08 BOOL  ; RK_12 U4_Y 预焊上料Z轴CW极限输入信号
2052.09 BOOL  ; RK_12 U4_Y 预焊上料Z轴CCW极限输入信号
2052.10 BOOL  ; RK_12 U4_Y 预焊上料Z轴原点接近输入信号
2052.11 BOOL  ; RK_12 U4_Y 预焊上料Z轴原点输入信号
2052.12 BOOL  ; RK_12 U4_Y 预焊上料Z轴中断输入信号
2052.13 BOOL  ; RK_12 U4_Y 预焊上料Z轴紧急停止输入信号
2052.14 BOOL  ; RK_12 U4_Y 预焊上料Z轴定位完成信号
2052.15 BOOL  ; $?St$Bk?_#[5032] / RK_12 U4_Y 预焊上料Z轴偏差计数器复位输出 / 原点调整命令输出$?St$Bk?_#[5032]
2053 CHANNEL  ; RK_12 U4_Y 预焊上料Z轴错误代码
2053.00 BOOL  ; RK_12 U4_Y 预焊上料Z轴错误代码
2053.01 BOOL  ; RK_12 U4_Y 预焊上料Z轴错误代码
2053.02 BOOL  ; RK_12 U4_Y 预焊上料Z轴错误代码
2053.03 BOOL  ; RK_12 U4_Y 预焊上料Z轴错误代码
2053.04 BOOL  ; RK_12 U4_Y 预焊上料Z轴错误代码
2053.05 BOOL  ; RK_12 U4_Y 预焊上料Z轴错误代码
2053.06 BOOL  ; RK_12 U4_Y 预焊上料Z轴错误代码
2053.07 BOOL  ; RK_12 U4_Y 预焊上料Z轴错误代码
2053.08 BOOL  ; RK_12 U4_Y 预焊上料Z轴错误代码
2053.09 BOOL  ; RK_12 U4_Y 预焊上料Z轴错误代码
2053.10 BOOL  ; RK_12 U4_Y 预焊上料Z轴错误代码
2053.11 BOOL  ; RK_12 U4_Y 预焊上料Z轴错误代码
2053.12 BOOL  ; RK_12 U4_Y 预焊上料Z轴错误代码
2053.13 BOOL  ; RK_12 U4_Y 预焊上料Z轴错误代码
2053.14 BOOL  ; RK_12 U4_Y 预焊上料Z轴错误代码
2053.15 BOOL  ; RK_12 U4_Y 预焊上料Z轴错误代码
2054.00 BOOL  ; RK_12 U4_Z 预焊下料Z轴Not Use
2054.01 BOOL  ; RK_12 U4_Z 预焊下料Z轴Not Use
2054.02 BOOL  ; RK_12 U4_Z 预焊下料Z轴Not Use
2054.03 BOOL  ; RK_12 U4_Z 预焊下料Z轴Not Use
2054.04 BOOL  ; RK_12 U4_Z 预焊下料Z轴等待存储器操作标志位
2054.05 BOOL  ; RK_12 U4_Z 预焊下料Z轴定位结束标志位
2054.06 BOOL  ; RK_12 U4_Z 预焊下料Z轴无原点标志位
2054.07 BOOL  ; RK_12 U4_Z 预焊下料Z轴原点停止标志位
2054.08 BOOL  ; RK_12 U4_Z 预焊下料Z轴区域0监控标志位
2054.09 BOOL  ; RK_12 U4_Z 预焊下料Z轴区域1监控标志位
2054.10 BOOL  ; RK_12 U4_Z 预焊下料Z轴区域2监控标志位
2054.11 BOOL  ; RK_12 U4_Z 预焊下料Z轴示教完成标志位
2054.12 BOOL  ; RK_12 U4_Z 预焊下料Z轴错误标志位
2054.13 BOOL  ; RK_12 U4_Z 预焊下料Z轴忙标志位
2054.14 BOOL  ; RK_12 U4_Z 预焊下料Z轴数据传送标志
2054.15 BOOL  ; RK_12 U4_Z 预焊下料Z轴减速停止执行标志
2055.00 BOOL  ; RK_12 U4_Z 预焊下料Z轴Not Use
2055.01 BOOL  ; RK_12 U4_Z 预焊下料Z轴Not Use
2055.02 BOOL  ; RK_12 U4_Z 预焊下料Z轴Not Use
2055.03 BOOL  ; RK_12 U4_Z 预焊下料Z轴Not Use
2055.04 BOOL  ; RK_12 U4_Z 预焊下料Z轴Not Use
2055.05 BOOL  ; RK_12 U4_Z 预焊下料Z轴Not Use
2055.06 BOOL  ; RK_12 U4_Z 预焊下料Z轴Not Use
2055.07 BOOL  ; RK_12 U4_Z 预焊下料Z轴Not Use
2055.08 BOOL  ; RK_12 U4_Z 预焊下料Z轴CW极限输入信号
2055.09 BOOL  ; RK_12 U4_Z 预焊下料Z轴CCW极限输入信号
2055.10 BOOL  ; RK_12 U4_Z 预焊下料Z轴原点接近输入信号
2055.11 BOOL  ; RK_12 U4_Z 预焊下料Z轴原点输入信号
2055.12 BOOL  ; RK_12 U4_Z 预焊下料Z轴中断输入信号
2055.13 BOOL  ; RK_12 U4_Z 预焊下料Z轴紧急停止输入信号
2055.14 BOOL  ; RK_12 U4_Z 预焊下料Z轴定位完成信号
2055.15 BOOL  ; $?St$Bk?_#[5033] / RK_12 U4_Z 预焊下料Z轴偏差计数器复位输出 / 原点调整命令输出$?St$Bk?_#[5033]
2056 CHANNEL  ; RK_12 U4_Z 预焊下料Z轴错误代码
2056.00 BOOL  ; RK_12 U4_Z 预焊下料Z轴错误代码
2056.01 BOOL  ; RK_12 U4_Z 预焊下料Z轴错误代码
2056.02 BOOL  ; RK_12 U4_Z 预焊下料Z轴错误代码
2056.03 BOOL  ; RK_12 U4_Z 预焊下料Z轴错误代码
2056.04 BOOL  ; RK_12 U4_Z 预焊下料Z轴错误代码
2056.05 BOOL  ; RK_12 U4_Z 预焊下料Z轴错误代码
2056.06 BOOL  ; RK_12 U4_Z 预焊下料Z轴错误代码
2056.07 BOOL  ; RK_12 U4_Z 预焊下料Z轴错误代码
2056.08 BOOL  ; RK_12 U4_Z 预焊下料Z轴错误代码
2056.09 BOOL  ; RK_12 U4_Z 预焊下料Z轴错误代码
2056.10 BOOL  ; RK_12 U4_Z 预焊下料Z轴错误代码
2056.11 BOOL  ; RK_12 U4_Z 预焊下料Z轴错误代码
2056.12 BOOL  ; RK_12 U4_Z 预焊下料Z轴错误代码
2056.13 BOOL  ; RK_12 U4_Z 预焊下料Z轴错误代码
2056.14 BOOL  ; RK_12 U4_Z 预焊下料Z轴错误代码
2056.15 BOOL  ; RK_12 U4_Z 预焊下料Z轴错误代码
2057.00 BOOL  ; RK_13 U4_U #1移载Y轴Not Use
2057.01 BOOL  ; RK_13 U4_U #1移载Y轴Not Use
2057.02 BOOL  ; RK_13 U4_U #1移载Y轴Not Use
2057.03 BOOL  ; RK_13 U4_U #1移载Y轴Not Use
2057.04 BOOL  ; RK_13 U4_U #1移载Y轴等待存储器操作标志位
2057.05 BOOL  ; RK_13 U4_U #1移载Y轴定位结束标志位
2057.06 BOOL  ; RK_13 U4_U #1移载Y轴无原点标志位
2057.07 BOOL  ; RK_13 U4_U #1移载Y轴原点停止标志位
2057.08 BOOL  ; RK_13 U4_U #1移载Y轴区域0监控标志位
2057.09 BOOL  ; RK_13 U4_U #1移载Y轴区域1监控标志位
2057.10 BOOL  ; RK_13 U4_U #1移载Y轴区域2监控标志位
2057.11 BOOL  ; RK_13 U4_U #1移载Y轴示教完成标志位
2057.12 BOOL  ; RK_13 U4_U #1移载Y轴错误标志位
2057.13 BOOL  ; RK_13 U4_U #1移载Y轴忙标志位
2057.14 BOOL  ; RK_13 U4_U #1移载Y轴数据传送标志
2057.15 BOOL  ; RK_13 U4_U #1移载Y轴减速停止执行标志
2058.00 BOOL  ; RK_13 U4_U #1移载Y轴Not Use
2058.01 BOOL  ; RK_13 U4_U #1移载Y轴Not Use
2058.02 BOOL  ; RK_13 U4_U #1移载Y轴Not Use
2058.03 BOOL  ; RK_13 U4_U #1移载Y轴Not Use
2058.04 BOOL  ; RK_13 U4_U #1移载Y轴Not Use
2058.05 BOOL  ; RK_13 U4_U #1移载Y轴Not Use
2058.06 BOOL  ; RK_13 U4_U #1移载Y轴Not Use
2058.07 BOOL  ; RK_13 U4_U #1移载Y轴Not Use
2058.08 BOOL  ; RK_13 U4_U #1移载Y轴CW极限输入信号
2058.09 BOOL  ; RK_13 U4_U #1移载Y轴CCW极限输入信号
2058.10 BOOL  ; RK_13 U4_U #1移载Y轴原点接近输入信号
2058.11 BOOL  ; RK_13 U4_U #1移载Y轴原点输入信号
2058.12 BOOL  ; RK_13 U4_U #1移载Y轴中断输入信号
2058.13 BOOL  ; RK_13 U4_U #1移载Y轴紧急停止输入信号
2058.14 BOOL  ; RK_13 U4_U #1移载Y轴定位完成信号
2058.15 BOOL  ; $?St$Bk?_#[5034] / RK_13 U4_U #1移载Y轴偏差计数器复位输出 / 原点调整命令输出$?St$Bk?_#[5034]
2059 CHANNEL  ; RK_13 U4_U #1移载Y轴错误代码
2059.00 BOOL  ; RK_13 U4_U #1移载Y轴错误代码
2059.01 BOOL  ; RK_13 U4_U #1移载Y轴错误代码
2059.02 BOOL  ; RK_13 U4_U #1移载Y轴错误代码
2059.03 BOOL  ; RK_13 U4_U #1移载Y轴错误代码
2059.04 BOOL  ; RK_13 U4_U #1移载Y轴错误代码
2059.05 BOOL  ; RK_13 U4_U #1移载Y轴错误代码
2059.06 BOOL  ; RK_13 U4_U #1移载Y轴错误代码
2059.07 BOOL  ; RK_13 U4_U #1移载Y轴错误代码
2059.08 BOOL  ; RK_13 U4_U #1移载Y轴错误代码
2059.09 BOOL  ; RK_13 U4_U #1移载Y轴错误代码
2059.10 BOOL  ; RK_13 U4_U #1移载Y轴错误代码
2059.11 BOOL  ; RK_13 U4_U #1移载Y轴错误代码
2059.12 BOOL  ; RK_13 U4_U #1移载Y轴错误代码
2059.13 BOOL  ; RK_13 U4_U #1移载Y轴错误代码
2059.14 BOOL  ; RK_13 U4_U #1移载Y轴错误代码
2059.15 BOOL  ; RK_13 U4_U #1移载Y轴错误代码
205.00 BOOL  ; 整机停止中（Lamp）
205.01 BOOL  ; 清料停止中（Lamp）
205.02 BOOL  ; 整机复位（Lamp）
2060.00 BOOL  ; RK_13 U6_X #2移载Y轴序列号使能
2060.01 BOOL  ; RK_13 U6_X #2移载Y轴启动
2060.02 BOOL  ; RK_13 U6_X #2移载Y轴独立启动
2060.03 BOOL  ; RK_13 U6_X #2移载Y轴绝对移动
2060.04 BOOL  ; RK_13 U6_X #2移载Y轴相对移动
2060.05 BOOL  ; RK_13 U6_X #2移载Y轴中断进给
2060.06 BOOL  ; RK_13 U6_X #2移载Y轴原点搜索
2060.07 BOOL  ; RK_13 U6_X #2移载Y轴原点返回
2060.08 BOOL  ; RK_13 U6_X #2移载Y轴当前位置预置
2060.09 BOOL  ; RK_13 U6_X #2移载Y轴点动
2060.10 BOOL  ; RK_13 U6_X #2移载Y轴方向定义
2060.11 BOOL  ; RK_13 U6_X #2移载Y轴示教
2060.12 BOOL  ; RK_13 U6_X #2移载Y轴释放禁止/复位
2060.13 BOOL  ; $?St$Bk?_#[5035] / RK_13 U6_X #2移载Y轴偏差计数器复位输出/ / 原点调整命令输出$?St$Bk?_#[5035]
2060.14 BOOL  ; RK_13 U6_X #2移载Y轴激活倍率
2060.15 BOOL  ; RK_13 U6_X #2移载Y轴停止
2061.00 BOOL  ; RK_13 U6_X #2移载Y轴Not Use
2061.01 BOOL  ; RK_13 U6_X #2移载Y轴Not Use
2061.02 BOOL  ; RK_13 U6_X #2移载Y轴Not Use
2061.03 BOOL  ; RK_13 U6_X #2移载Y轴Not Use
2061.04 BOOL  ; RK_13 U6_X #2移载Y轴Not Use
2061.05 BOOL  ; RK_13 U6_X #2移载Y轴Not Use
2061.06 BOOL  ; RK_13 U6_X #2移载Y轴Not Use
2061.07 BOOL  ; RK_13 U6_X #2移载Y轴Not Use
2061.08 BOOL  ; RK_13 U6_X #2移载Y轴强迫中断
2061.09 BOOL  ; RK_13 U6_X #2移载Y轴Not Use
2061.10 BOOL  ; RK_13 U6_X #2移载Y轴Not Use
2061.11 BOOL  ; RK_13 U6_X #2移载Y轴Not Use
2061.12 BOOL  ; RK_13 U6_X #2移载Y轴写数据
2061.13 BOOL  ; RK_13 U6_X #2移载Y轴读数据
2061.14 BOOL  ; RK_13 U6_X #2移载Y轴存数据
2061.15 BOOL  ; RK_13 U6_X #2移载Y轴Not Use
2062.00 BOOL  ; RK_16 U6_Y 激光焊接X轴序列号使能
2062.01 BOOL  ; RK_16 U6_Y 激光焊接X轴启动
2062.02 BOOL  ; RK_16 U6_Y 激光焊接X轴独立启动
2062.03 BOOL  ; RK_16 U6_Y 激光焊接X轴绝对移动
2062.04 BOOL  ; RK_16 U6_Y 激光焊接X轴相对移动
2062.05 BOOL  ; RK_16 U6_Y 激光焊接X轴中断进给
2062.06 BOOL  ; RK_16 U6_Y 激光焊接X轴原点搜索
2062.07 BOOL  ; RK_16 U6_Y 激光焊接X轴原点返回
2062.08 BOOL  ; RK_16 U6_Y 激光焊接X轴当前位置预置
2062.09 BOOL  ; RK_16 U6_Y 激光焊接X轴点动
2062.10 BOOL  ; RK_16 U6_Y 激光焊接X轴方向定义
2062.11 BOOL  ; RK_16 U6_Y 激光焊接X轴示教
2062.12 BOOL  ; RK_16 U6_Y 激光焊接X轴释放禁止/复位
2062.13 BOOL  ; $?St$Bk?_#[5036] / RK_16 U6_Y 激光焊接X轴偏差计数器复位输出/ / 原点调整命令输出$?St$Bk?_#[5036]
2062.14 BOOL  ; RK_16 U6_Y 激光焊接X轴激活倍率
2062.15 BOOL  ; RK_16 U6_Y 激光焊接X轴停止
2063.00 BOOL  ; RK_16 U6_Y 激光焊接X轴Not Use
2063.01 BOOL  ; RK_16 U6_Y 激光焊接X轴Not Use
2063.02 BOOL  ; RK_16 U6_Y 激光焊接X轴Not Use
2063.03 BOOL  ; RK_16 U6_Y 激光焊接X轴Not Use
2063.04 BOOL  ; RK_16 U6_Y 激光焊接X轴Not Use
2063.05 BOOL  ; RK_16 U6_Y 激光焊接X轴Not Use
2063.06 BOOL  ; RK_16 U6_Y 激光焊接X轴Not Use
2063.07 BOOL  ; RK_16 U6_Y 激光焊接X轴Not Use
2063.08 BOOL  ; RK_16 U6_Y 激光焊接X轴强迫中断
2063.09 BOOL  ; RK_16 U6_Y 激光焊接X轴Not Use
2063.10 BOOL  ; RK_16 U6_Y 激光焊接X轴Not Use
2063.11 BOOL  ; RK_16 U6_Y 激光焊接X轴Not Use
2063.12 BOOL  ; RK_16 U6_Y 激光焊接X轴写数据
2063.13 BOOL  ; RK_16 U6_Y 激光焊接X轴读数据
2063.14 BOOL  ; RK_16 U6_Y 激光焊接X轴存数据
2063.15 BOOL  ; RK_16 U6_Y 激光焊接X轴Not Use
2064.00 BOOL  ; RK_16 U6_Z 激光焊接Z轴序列号使能
2064.01 BOOL  ; RK_16 U6_Z 激光焊接Z轴启动
2064.02 BOOL  ; RK_16 U6_Z 激光焊接Z轴独立启动
2064.03 BOOL  ; RK_16 U6_Z 激光焊接Z轴绝对移动
2064.04 BOOL  ; RK_16 U6_Z 激光焊接Z轴相对移动
2064.05 BOOL  ; RK_16 U6_Z 激光焊接Z轴中断进给
2064.06 BOOL  ; RK_16 U6_Z 激光焊接Z轴原点搜索
2064.07 BOOL  ; RK_16 U6_Z 激光焊接Z轴原点返回
2064.08 BOOL  ; RK_16 U6_Z 激光焊接Z轴当前位置预置
2064.09 BOOL  ; RK_16 U6_Z 激光焊接Z轴点动
2064.10 BOOL  ; RK_16 U6_Z 激光焊接Z轴方向定义
2064.11 BOOL  ; RK_16 U6_Z 激光焊接Z轴示教
2064.12 BOOL  ; RK_16 U6_Z 激光焊接Z轴释放禁止/复位
2064.13 BOOL  ; $?St$Bk?_#[5037] / RK_16 U6_Z 激光焊接Z轴偏差计数器复位输出/ / 原点调整命令输出$?St$Bk?_#[5037]
2064.14 BOOL  ; RK_16 U6_Z 激光焊接Z轴激活倍率
2064.15 BOOL  ; RK_16 U6_Z 激光焊接Z轴停止
2065.00 BOOL  ; RK_16 U6_Z 激光焊接Z轴Not Use
2065.01 BOOL  ; RK_16 U6_Z 激光焊接Z轴Not Use
2065.02 BOOL  ; RK_16 U6_Z 激光焊接Z轴Not Use
2065.03 BOOL  ; RK_16 U6_Z 激光焊接Z轴Not Use
2065.04 BOOL  ; RK_16 U6_Z 激光焊接Z轴Not Use
2065.05 BOOL  ; RK_16 U6_Z 激光焊接Z轴Not Use
2065.06 BOOL  ; RK_16 U6_Z 激光焊接Z轴Not Use
2065.07 BOOL  ; RK_16 U6_Z 激光焊接Z轴Not Use
2065.08 BOOL  ; RK_16 U6_Z 激光焊接Z轴强迫中断
2065.09 BOOL  ; RK_16 U6_Z 激光焊接Z轴Not Use
2065.10 BOOL  ; RK_16 U6_Z 激光焊接Z轴Not Use
2065.11 BOOL  ; RK_16 U6_Z 激光焊接Z轴Not Use
2065.12 BOOL  ; RK_16 U6_Z 激光焊接Z轴写数据
2065.13 BOOL  ; RK_16 U6_Z 激光焊接Z轴读数据
2065.14 BOOL  ; RK_16 U6_Z 激光焊接Z轴存数据
2065.15 BOOL  ; RK_16 U6_Z 激光焊接Z轴Not Use
2068.00 BOOL  ; RK_13 U6_X #2移载Y轴Not Use
2068.01 BOOL  ; RK_13 U6_X #2移载Y轴Not Use
2068.02 BOOL  ; RK_13 U6_X #2移载Y轴Not Use
2068.03 BOOL  ; RK_13 U6_X #2移载Y轴Not Use
2068.04 BOOL  ; RK_13 U6_X #2移载Y轴等待存储器操作标志位
2068.05 BOOL  ; RK_13 U6_X #2移载Y轴定位结束标志位
2068.06 BOOL  ; RK_13 U6_X #2移载Y轴无原点标志位
2068.07 BOOL  ; RK_13 U6_X #2移载Y轴原点停止标志位
2068.08 BOOL  ; RK_13 U6_X #2移载Y轴区域0监控标志位
2068.09 BOOL  ; RK_13 U6_X #2移载Y轴区域1监控标志位
2068.10 BOOL  ; RK_13 U6_X #2移载Y轴区域2监控标志位
2068.11 BOOL  ; RK_13 U6_X #2移载Y轴示教完成标志位
2068.12 BOOL  ; RK_13 U6_X #2移载Y轴错误标志位
2068.13 BOOL  ; RK_13 U6_X #2移载Y轴忙标志位
2068.14 BOOL  ; RK_13 U6_X #2移载Y轴数据传送标志
2068.15 BOOL  ; RK_13 U6_X #2移载Y轴减速停止执行标志
2069.00 BOOL  ; RK_13 U6_X #2移载Y轴Not Use
2069.01 BOOL  ; RK_13 U6_X #2移载Y轴Not Use
2069.02 BOOL  ; RK_13 U6_X #2移载Y轴Not Use
2069.03 BOOL  ; RK_13 U6_X #2移载Y轴Not Use
2069.04 BOOL  ; RK_13 U6_X #2移载Y轴Not Use
2069.05 BOOL  ; RK_13 U6_X #2移载Y轴Not Use
2069.06 BOOL  ; RK_13 U6_X #2移载Y轴Not Use
2069.07 BOOL  ; RK_13 U6_X #2移载Y轴Not Use
2069.08 BOOL  ; RK_13 U6_X #2移载Y轴CW极限输入信号
2069.09 BOOL  ; RK_13 U6_X #2移载Y轴CCW极限输入信号
2069.10 BOOL  ; RK_13 U6_X #2移载Y轴原点接近输入信号
2069.11 BOOL  ; RK_13 U6_X #2移载Y轴原点输入信号
2069.12 BOOL  ; RK_13 U6_X #2移载Y轴中断输入信号
2069.13 BOOL  ; RK_13 U6_X #2移载Y轴紧急停止输入信号
2069.14 BOOL  ; RK_13 U6_X #2移载Y轴定位完成信号
2069.15 BOOL  ; $?St$Bk?_#[5038] / RK_13 U6_X #2移载Y轴偏差计数器复位输出 / 原点调整命令输出$?St$Bk?_#[5038]
2070 CHANNEL  ; RK_13 U6_X #2移载Y轴错误代码
2070.00 BOOL  ; RK_13 U6_X #2移载Y轴错误代码
2070.01 BOOL  ; RK_13 U6_X #2移载Y轴错误代码
2070.02 BOOL  ; RK_13 U6_X #2移载Y轴错误代码
2070.03 BOOL  ; RK_13 U6_X #2移载Y轴错误代码
2070.04 BOOL  ; RK_13 U6_X #2移载Y轴错误代码
2070.05 BOOL  ; RK_13 U6_X #2移载Y轴错误代码
2070.06 BOOL  ; RK_13 U6_X #2移载Y轴错误代码
2070.07 BOOL  ; RK_13 U6_X #2移载Y轴错误代码
2070.08 BOOL  ; RK_13 U6_X #2移载Y轴错误代码
2070.09 BOOL  ; RK_13 U6_X #2移载Y轴错误代码
2070.10 BOOL  ; RK_13 U6_X #2移载Y轴错误代码
2070.11 BOOL  ; RK_13 U6_X #2移载Y轴错误代码
2070.12 BOOL  ; RK_13 U6_X #2移载Y轴错误代码
2070.13 BOOL  ; RK_13 U6_X #2移载Y轴错误代码
2070.14 BOOL  ; RK_13 U6_X #2移载Y轴错误代码
2070.15 BOOL  ; RK_13 U6_X #2移载Y轴错误代码
2071.00 BOOL  ; RK_16 U6_Y 激光焊接X轴Not Use
2071.01 BOOL  ; RK_16 U6_Y 激光焊接X轴Not Use
2071.02 BOOL  ; RK_16 U6_Y 激光焊接X轴Not Use
2071.03 BOOL  ; RK_16 U6_Y 激光焊接X轴Not Use
2071.04 BOOL  ; RK_16 U6_Y 激光焊接X轴等待存储器操作标志位
2071.05 BOOL  ; RK_16 U6_Y 激光焊接X轴定位结束标志位
2071.06 BOOL  ; RK_16 U6_Y 激光焊接X轴无原点标志位
2071.07 BOOL  ; RK_16 U6_Y 激光焊接X轴原点停止标志位
2071.08 BOOL  ; RK_16 U6_Y 激光焊接X轴区域0监控标志位
2071.09 BOOL  ; RK_16 U6_Y 激光焊接X轴区域1监控标志位
2071.10 BOOL  ; RK_16 U6_Y 激光焊接X轴区域2监控标志位
2071.11 BOOL  ; RK_16 U6_Y 激光焊接X轴示教完成标志位
2071.12 BOOL  ; RK_16 U6_Y 激光焊接X轴错误标志位
2071.13 BOOL  ; RK_16 U6_Y 激光焊接X轴忙标志位
2071.14 BOOL  ; RK_16 U6_Y 激光焊接X轴数据传送标志
2071.15 BOOL  ; RK_16 U6_Y 激光焊接X轴减速停止执行标志
2072.00 BOOL  ; RK_16 U6_Y 激光焊接X轴Not Use
2072.01 BOOL  ; RK_16 U6_Y 激光焊接X轴Not Use
2072.02 BOOL  ; RK_16 U6_Y 激光焊接X轴Not Use
2072.03 BOOL  ; RK_16 U6_Y 激光焊接X轴Not Use
2072.04 BOOL  ; RK_16 U6_Y 激光焊接X轴Not Use
2072.05 BOOL  ; RK_16 U6_Y 激光焊接X轴Not Use
2072.06 BOOL  ; RK_16 U6_Y 激光焊接X轴Not Use
2072.07 BOOL  ; RK_16 U6_Y 激光焊接X轴Not Use
2072.08 BOOL  ; RK_16 U6_Y 激光焊接X轴CW极限输入信号
2072.09 BOOL  ; RK_16 U6_Y 激光焊接X轴CCW极限输入信号
2072.10 BOOL  ; RK_16 U6_Y 激光焊接X轴原点接近输入信号
2072.11 BOOL  ; RK_16 U6_Y 激光焊接X轴原点输入信号
2072.12 BOOL  ; RK_16 U6_Y 激光焊接X轴中断输入信号
2072.13 BOOL  ; RK_16 U6_Y 激光焊接X轴紧急停止输入信号
2072.14 BOOL  ; RK_16 U6_Y 激光焊接X轴定位完成信号
2072.15 BOOL  ; $?St$Bk?_#[5039] / RK_16 U6_Y 激光焊接X轴偏差计数器复位输出 / 原点调整命令输出$?St$Bk?_#[5039]
2073 CHANNEL  ; RK_16 U6_Y 激光焊接X轴错误代码
2073.00 BOOL  ; RK_16 U6_Y 激光焊接X轴错误代码
2073.01 BOOL  ; RK_16 U6_Y 激光焊接X轴错误代码
2073.02 BOOL  ; RK_16 U6_Y 激光焊接X轴错误代码
2073.03 BOOL  ; RK_16 U6_Y 激光焊接X轴错误代码
2073.04 BOOL  ; RK_16 U6_Y 激光焊接X轴错误代码
2073.05 BOOL  ; RK_16 U6_Y 激光焊接X轴错误代码
2073.06 BOOL  ; RK_16 U6_Y 激光焊接X轴错误代码
2073.07 BOOL  ; RK_16 U6_Y 激光焊接X轴错误代码
2073.08 BOOL  ; RK_16 U6_Y 激光焊接X轴错误代码
2073.09 BOOL  ; RK_16 U6_Y 激光焊接X轴错误代码
2073.10 BOOL  ; RK_16 U6_Y 激光焊接X轴错误代码
2073.11 BOOL  ; RK_16 U6_Y 激光焊接X轴错误代码
2073.12 BOOL  ; RK_16 U6_Y 激光焊接X轴错误代码
2073.13 BOOL  ; RK_16 U6_Y 激光焊接X轴错误代码
2073.14 BOOL  ; RK_16 U6_Y 激光焊接X轴错误代码
2073.15 BOOL  ; RK_16 U6_Y 激光焊接X轴错误代码
2074.00 BOOL  ; RK_16 U6_Z 激光焊接Z轴Not Use
2074.01 BOOL  ; RK_16 U6_Z 激光焊接Z轴Not Use
2074.02 BOOL  ; RK_16 U6_Z 激光焊接Z轴Not Use
2074.03 BOOL  ; RK_16 U6_Z 激光焊接Z轴Not Use
2074.04 BOOL  ; RK_16 U6_Z 激光焊接Z轴等待存储器操作标志位
2074.05 BOOL  ; RK_16 U6_Z 激光焊接Z轴定位结束标志位
2074.06 BOOL  ; RK_16 U6_Z 激光焊接Z轴无原点标志位
2074.07 BOOL  ; RK_16 U6_Z 激光焊接Z轴原点停止标志位
2074.08 BOOL  ; RK_16 U6_Z 激光焊接Z轴区域0监控标志位
2074.09 BOOL  ; RK_16 U6_Z 激光焊接Z轴区域1监控标志位
2074.10 BOOL  ; RK_16 U6_Z 激光焊接Z轴区域2监控标志位
2074.11 BOOL  ; RK_16 U6_Z 激光焊接Z轴示教完成标志位
2074.12 BOOL  ; RK_16 U6_Z 激光焊接Z轴错误标志位
2074.13 BOOL  ; RK_16 U6_Z 激光焊接Z轴忙标志位
2074.14 BOOL  ; RK_16 U6_Z 激光焊接Z轴数据传送标志
2074.15 BOOL  ; RK_16 U6_Z 激光焊接Z轴减速停止执行标志
2075.00 BOOL  ; RK_16 U6_Z 激光焊接Z轴Not Use
2075.01 BOOL  ; RK_16 U6_Z 激光焊接Z轴Not Use
2075.02 BOOL  ; RK_16 U6_Z 激光焊接Z轴Not Use
2075.03 BOOL  ; RK_16 U6_Z 激光焊接Z轴Not Use
2075.04 BOOL  ; RK_16 U6_Z 激光焊接Z轴Not Use
2075.05 BOOL  ; RK_16 U6_Z 激光焊接Z轴Not Use
2075.06 BOOL  ; RK_16 U6_Z 激光焊接Z轴Not Use
2075.07 BOOL  ; RK_16 U6_Z 激光焊接Z轴Not Use
2075.08 BOOL  ; RK_16 U6_Z 激光焊接Z轴CW极限输入信号
2075.09 BOOL  ; RK_16 U6_Z 激光焊接Z轴CCW极限输入信号
2075.10 BOOL  ; RK_16 U6_Z 激光焊接Z轴原点接近输入信号
2075.11 BOOL  ; RK_16 U6_Z 激光焊接Z轴原点输入信号
2075.12 BOOL  ; RK_16 U6_Z 激光焊接Z轴中断输入信号
2075.13 BOOL  ; RK_16 U6_Z 激光焊接Z轴紧急停止输入信号
2075.14 BOOL  ; RK_16 U6_Z 激光焊接Z轴定位完成信号
2075.15 BOOL  ; $?St$Bk?_#[5040] / RK_16 U6_Z 激光焊接Z轴偏差计数器复位输出 / 原点调整命令输出$?St$Bk?_#[5040]
2076 CHANNEL  ; RK_16 U6_Z 激光焊接Z轴错误代码
2076.00 BOOL  ; RK_16 U6_Z 激光焊接Z轴错误代码
2076.01 BOOL  ; RK_16 U6_Z 激光焊接Z轴错误代码
2076.02 BOOL  ; RK_16 U6_Z 激光焊接Z轴错误代码
2076.03 BOOL  ; RK_16 U6_Z 激光焊接Z轴错误代码
2076.04 BOOL  ; RK_16 U6_Z 激光焊接Z轴错误代码
2076.05 BOOL  ; RK_16 U6_Z 激光焊接Z轴错误代码
2076.06 BOOL  ; RK_16 U6_Z 激光焊接Z轴错误代码
2076.07 BOOL  ; RK_16 U6_Z 激光焊接Z轴错误代码
2076.08 BOOL  ; RK_16 U6_Z 激光焊接Z轴错误代码
2076.09 BOOL  ; RK_16 U6_Z 激光焊接Z轴错误代码
2076.10 BOOL  ; RK_16 U6_Z 激光焊接Z轴错误代码
2076.11 BOOL  ; RK_16 U6_Z 激光焊接Z轴错误代码
2076.12 BOOL  ; RK_16 U6_Z 激光焊接Z轴错误代码
2076.13 BOOL  ; RK_16 U6_Z 激光焊接Z轴错误代码
2076.14 BOOL  ; RK_16 U6_Z 激光焊接Z轴错误代码
2076.15 BOOL  ; RK_16 U6_Z 激光焊接Z轴错误代码
2080.00 BOOL  ; RK_06 U8_X 电池上下料X轴序列号使能
2080.01 BOOL  ; RK_06 U8_X 电池上下料X轴启动
2080.02 BOOL  ; RK_06 U8_X 电池上下料X轴独立启动
2080.03 BOOL  ; RK_06 U8_X 电池上下料X轴绝对移动
2080.04 BOOL  ; RK_06 U8_X 电池上下料X轴相对移动
2080.05 BOOL  ; RK_06 U8_X 电池上下料X轴中断进给
2080.06 BOOL  ; RK_06 U8_X 电池上下料X轴原点搜索
2080.07 BOOL  ; RK_06 U8_X 电池上下料X轴原点返回
2080.08 BOOL  ; RK_06 U8_X 电池上下料X轴当前位置预置
2080.09 BOOL  ; RK_06 U8_X 电池上下料X轴点动
2080.10 BOOL  ; RK_06 U8_X 电池上下料X轴方向定义
2080.11 BOOL  ; RK_06 U8_X 电池上下料X轴示教
2080.12 BOOL  ; RK_06 U8_X 电池上下料X轴释放禁止/复位
2080.13 BOOL  ; $?St$Bk?_#[5041] / RK_06 U8_X 电池上下料X轴偏差计数器复位输出/ / 原点调整命令输出$?St$Bk?_#[5041]
2080.14 BOOL  ; RK_06 U8_X 电池上下料X轴激活倍率
2080.15 BOOL  ; RK_06 U8_X 电池上下料X轴停止
2081.00 BOOL  ; RK_06 U8_X 电池上下料X轴Not Use
2081.01 BOOL  ; RK_06 U8_X 电池上下料X轴Not Use
2081.02 BOOL  ; RK_06 U8_X 电池上下料X轴Not Use
2081.03 BOOL  ; RK_06 U8_X 电池上下料X轴Not Use
2081.04 BOOL  ; RK_06 U8_X 电池上下料X轴Not Use
2081.05 BOOL  ; RK_06 U8_X 电池上下料X轴Not Use
2081.06 BOOL  ; RK_06 U8_X 电池上下料X轴Not Use
2081.07 BOOL  ; RK_06 U8_X 电池上下料X轴Not Use
2081.08 BOOL  ; RK_06 U8_X 电池上下料X轴强迫中断
2081.09 BOOL  ; RK_06 U8_X 电池上下料X轴Not Use
2081.10 BOOL  ; RK_06 U8_X 电池上下料X轴Not Use
2081.11 BOOL  ; RK_06 U8_X 电池上下料X轴Not Use
2081.12 BOOL  ; RK_06 U8_X 电池上下料X轴写数据
2081.13 BOOL  ; RK_06 U8_X 电池上下料X轴读数据
2081.14 BOOL  ; RK_06 U8_X 电池上下料X轴存数据
2081.15 BOOL  ; RK_06 U8_X 电池上下料X轴Not Use
2082.00 BOOL  ; RK_07 U8_Y 铝壳进料X轴序列号使能
2082.01 BOOL  ; RK_07 U8_Y 铝壳进料X轴启动
2082.02 BOOL  ; RK_07 U8_Y 铝壳进料X轴独立启动
2082.03 BOOL  ; RK_07 U8_Y 铝壳进料X轴绝对移动
2082.04 BOOL  ; RK_07 U8_Y 铝壳进料X轴相对移动
2082.05 BOOL  ; RK_07 U8_Y 铝壳进料X轴中断进给
2082.06 BOOL  ; RK_07 U8_Y 铝壳进料X轴原点搜索
2082.07 BOOL  ; RK_07 U8_Y 铝壳进料X轴原点返回
2082.08 BOOL  ; RK_07 U8_Y 铝壳进料X轴当前位置预置
2082.09 BOOL  ; RK_07 U8_Y 铝壳进料X轴点动
2082.10 BOOL  ; RK_07 U8_Y 铝壳进料X轴方向定义
2082.11 BOOL  ; RK_07 U8_Y 铝壳进料X轴示教
2082.12 BOOL  ; RK_07 U8_Y 铝壳进料X轴释放禁止/复位
2082.13 BOOL  ; $?St$Bk?_#[5042] / RK_07 U8_Y 铝壳进料X轴偏差计数器复位输出/ / 原点调整命令输出$?St$Bk?_#[5042]
2082.14 BOOL  ; RK_07 U8_Y 铝壳进料X轴激活倍率
2082.15 BOOL  ; RK_07 U8_Y 铝壳进料X轴停止
2083.00 BOOL  ; RK_07 U8_Y 铝壳进料X轴Not Use
2083.01 BOOL  ; RK_07 U8_Y 铝壳进料X轴Not Use
2083.02 BOOL  ; RK_07 U8_Y 铝壳进料X轴Not Use
2083.03 BOOL  ; RK_07 U8_Y 铝壳进料X轴Not Use
2083.04 BOOL  ; RK_07 U8_Y 铝壳进料X轴Not Use
2083.05 BOOL  ; RK_07 U8_Y 铝壳进料X轴Not Use
2083.06 BOOL  ; RK_07 U8_Y 铝壳进料X轴Not Use
2083.07 BOOL  ; RK_07 U8_Y 铝壳进料X轴Not Use
2083.08 BOOL  ; RK_07 U8_Y 铝壳进料X轴强迫中断
2083.09 BOOL  ; RK_07 U8_Y 铝壳进料X轴Not Use
2083.10 BOOL  ; RK_07 U8_Y 铝壳进料X轴Not Use
2083.11 BOOL  ; RK_07 U8_Y 铝壳进料X轴Not Use
2083.12 BOOL  ; RK_07 U8_Y 铝壳进料X轴写数据
2083.13 BOOL  ; RK_07 U8_Y 铝壳进料X轴读数据
2083.14 BOOL  ; RK_07 U8_Y 铝壳进料X轴存数据
2083.15 BOOL  ; RK_07 U8_Y 铝壳进料X轴Not Use
2084.00 BOOL  ; RK_07 U8_Z 铝壳上料移载Y轴序列号使能
2084.01 BOOL  ; RK_07 U8_Z 铝壳上料移载Y轴启动
2084.02 BOOL  ; RK_07 U8_Z 铝壳上料移载Y轴独立启动
2084.03 BOOL  ; RK_07 U8_Z 铝壳上料移载Y轴绝对移动
2084.04 BOOL  ; RK_07 U8_Z 铝壳上料移载Y轴相对移动
2084.05 BOOL  ; RK_07 U8_Z 铝壳上料移载Y轴中断进给
2084.06 BOOL  ; RK_07 U8_Z 铝壳上料移载Y轴原点搜索
2084.07 BOOL  ; RK_07 U8_Z 铝壳上料移载Y轴原点返回
2084.08 BOOL  ; RK_07 U8_Z 铝壳上料移载Y轴当前位置预置
2084.09 BOOL  ; RK_07 U8_Z 铝壳上料移载Y轴点动
2084.10 BOOL  ; RK_07 U8_Z 铝壳上料移载Y轴方向定义
2084.11 BOOL  ; RK_07 U8_Z 铝壳上料移载Y轴示教
2084.12 BOOL  ; RK_07 U8_Z 铝壳上料移载Y轴释放禁止/复位
2084.13 BOOL  ; $?St$Bk?_#[5043] / RK_07 U8_Z 铝壳上料移载Y轴偏差计数器复位输出/ / 原点调整命令输出$?St$Bk?_#[5043]
2084.14 BOOL  ; RK_07 U8_Z 铝壳上料移载Y轴激活倍率
2084.15 BOOL  ; RK_07 U8_Z 铝壳上料移载Y轴停止
2085.00 BOOL  ; RK_07 U8_Z 铝壳上料移载Y轴Not Use
2085.01 BOOL  ; RK_07 U8_Z 铝壳上料移载Y轴Not Use
2085.02 BOOL  ; RK_07 U8_Z 铝壳上料移载Y轴Not Use
2085.03 BOOL  ; RK_07 U8_Z 铝壳上料移载Y轴Not Use
2085.04 BOOL  ; RK_07 U8_Z 铝壳上料移载Y轴Not Use
2085.05 BOOL  ; RK_07 U8_Z 铝壳上料移载Y轴Not Use
2085.06 BOOL  ; RK_07 U8_Z 铝壳上料移载Y轴Not Use
2085.07 BOOL  ; RK_07 U8_Z 铝壳上料移载Y轴Not Use
2085.08 BOOL  ; RK_07 U8_Z 铝壳上料移载Y轴强迫中断
2085.09 BOOL  ; RK_07 U8_Z 铝壳上料移载Y轴Not Use
2085.10 BOOL  ; RK_07 U8_Z 铝壳上料移载Y轴Not Use
2085.11 BOOL  ; RK_07 U8_Z 铝壳上料移载Y轴Not Use
2085.12 BOOL  ; RK_07 U8_Z 铝壳上料移载Y轴写数据
2085.13 BOOL  ; RK_07 U8_Z 铝壳上料移载Y轴读数据
2085.14 BOOL  ; RK_07 U8_Z 铝壳上料移载Y轴存数据
2085.15 BOOL  ; RK_07 U8_Z 铝壳上料移载Y轴Not Use
2086.00 BOOL  ; RK_10 U8_U 电池除尘上料X轴序列号使能
2086.01 BOOL  ; RK_10 U8_U 电池除尘上料X轴启动
2086.02 BOOL  ; RK_10 U8_U 电池除尘上料X轴独立启动
2086.03 BOOL  ; RK_10 U8_U 电池除尘上料X轴绝对移动
2086.04 BOOL  ; RK_10 U8_U 电池除尘上料X轴相对移动
2086.05 BOOL  ; RK_10 U8_U 电池除尘上料X轴中断进给
2086.06 BOOL  ; RK_10 U8_U 电池除尘上料X轴原点搜索
2086.07 BOOL  ; RK_10 U8_U 电池除尘上料X轴原点返回
2086.08 BOOL  ; RK_10 U8_U 电池除尘上料X轴当前位置预置
2086.09 BOOL  ; RK_10 U8_U 电池除尘上料X轴点动
2086.10 BOOL  ; RK_10 U8_U 电池除尘上料X轴方向定义
2086.11 BOOL  ; RK_10 U8_U 电池除尘上料X轴示教
2086.12 BOOL  ; RK_10 U8_U 电池除尘上料X轴释放禁止/复位
2086.13 BOOL  ; $?St$Bk?_#[5044] / RK_10 U8_U 电池除尘上料X轴偏差计数器复位输出/ / 原点调整命令输出$?St$Bk?_#[5044]
2086.14 BOOL  ; RK_10 U8_U 电池除尘上料X轴激活倍率
2086.15 BOOL  ; RK_10 U8_U 电池除尘上料X轴停止
2087.00 BOOL  ; RK_10 U8_U 电池除尘上料X轴Not Use
2087.01 BOOL  ; RK_10 U8_U 电池除尘上料X轴Not Use
2087.02 BOOL  ; RK_10 U8_U 电池除尘上料X轴Not Use
2087.03 BOOL  ; RK_10 U8_U 电池除尘上料X轴Not Use
2087.04 BOOL  ; RK_10 U8_U 电池除尘上料X轴Not Use
2087.05 BOOL  ; RK_10 U8_U 电池除尘上料X轴Not Use
2087.06 BOOL  ; RK_10 U8_U 电池除尘上料X轴Not Use
2087.07 BOOL  ; RK_10 U8_U 电池除尘上料X轴Not Use
2087.08 BOOL  ; RK_10 U8_U 电池除尘上料X轴强迫中断
2087.09 BOOL  ; RK_10 U8_U 电池除尘上料X轴Not Use
2087.10 BOOL  ; RK_10 U8_U 电池除尘上料X轴Not Use
2087.11 BOOL  ; RK_10 U8_U 电池除尘上料X轴Not Use
2087.12 BOOL  ; RK_10 U8_U 电池除尘上料X轴写数据
2087.13 BOOL  ; RK_10 U8_U 电池除尘上料X轴读数据
2087.14 BOOL  ; RK_10 U8_U 电池除尘上料X轴存数据
2087.15 BOOL  ; RK_10 U8_U 电池除尘上料X轴Not Use
2088.00 BOOL  ; RK_06 U8_X 电池上下料X轴Not Use
2088.01 BOOL  ; RK_06 U8_X 电池上下料X轴Not Use
2088.02 BOOL  ; RK_06 U8_X 电池上下料X轴Not Use
2088.03 BOOL  ; RK_06 U8_X 电池上下料X轴Not Use
2088.04 BOOL  ; RK_06 U8_X 电池上下料X轴等待存储器操作标志位
2088.05 BOOL  ; RK_06 U8_X 电池上下料X轴定位结束标志位
2088.06 BOOL  ; RK_06 U8_X 电池上下料X轴无原点标志位
2088.07 BOOL  ; RK_06 U8_X 电池上下料X轴原点停止标志位
2088.08 BOOL  ; RK_06 U8_X 电池上下料X轴区域0监控标志位
2088.09 BOOL  ; RK_06 U8_X 电池上下料X轴区域1监控标志位
2088.10 BOOL  ; RK_06 U8_X 电池上下料X轴区域2监控标志位
2088.11 BOOL  ; RK_06 U8_X 电池上下料X轴示教完成标志位
2088.12 BOOL  ; RK_06 U8_X 电池上下料X轴错误标志位
2088.13 BOOL  ; RK_06 U8_X 电池上下料X轴忙标志位
2088.14 BOOL  ; RK_06 U8_X 电池上下料X轴数据传送标志
2088.15 BOOL  ; RK_06 U8_X 电池上下料X轴减速停止执行标志
2089.00 BOOL  ; RK_06 U8_X 电池上下料X轴Not Use
2089.01 BOOL  ; RK_06 U8_X 电池上下料X轴Not Use
2089.02 BOOL  ; RK_06 U8_X 电池上下料X轴Not Use
2089.03 BOOL  ; RK_06 U8_X 电池上下料X轴Not Use
2089.04 BOOL  ; RK_06 U8_X 电池上下料X轴Not Use
2089.05 BOOL  ; RK_06 U8_X 电池上下料X轴Not Use
2089.06 BOOL  ; RK_06 U8_X 电池上下料X轴Not Use
2089.07 BOOL  ; RK_06 U8_X 电池上下料X轴Not Use
2089.08 BOOL  ; RK_06 U8_X 电池上下料X轴CW极限输入信号
2089.09 BOOL  ; RK_06 U8_X 电池上下料X轴CCW极限输入信号
2089.10 BOOL  ; RK_06 U8_X 电池上下料X轴原点接近输入信号
2089.11 BOOL  ; RK_06 U8_X 电池上下料X轴原点输入信号
2089.12 BOOL  ; RK_06 U8_X 电池上下料X轴中断输入信号
2089.13 BOOL  ; RK_06 U8_X 电池上下料X轴紧急停止输入信号
2089.14 BOOL  ; RK_06 U8_X 电池上下料X轴定位完成信号
2089.15 BOOL  ; $?St$Bk?_#[5045] / RK_06 U8_X 电池上下料X轴偏差计数器复位输出 / 原点调整命令输出$?St$Bk?_#[5045]
2090 CHANNEL  ; RK_06 U8_X 电池上下料X轴错误代码
2090.00 BOOL  ; RK_06 U8_X 电池上下料X轴错误代码
2090.01 BOOL  ; RK_06 U8_X 电池上下料X轴错误代码
2090.02 BOOL  ; RK_06 U8_X 电池上下料X轴错误代码
2090.03 BOOL  ; RK_06 U8_X 电池上下料X轴错误代码
2090.04 BOOL  ; RK_06 U8_X 电池上下料X轴错误代码
2090.05 BOOL  ; RK_06 U8_X 电池上下料X轴错误代码
2090.06 BOOL  ; RK_06 U8_X 电池上下料X轴错误代码
2090.07 BOOL  ; RK_06 U8_X 电池上下料X轴错误代码
2090.08 BOOL  ; RK_06 U8_X 电池上下料X轴错误代码
2090.09 BOOL  ; RK_06 U8_X 电池上下料X轴错误代码
2090.10 BOOL  ; RK_06 U8_X 电池上下料X轴错误代码
2090.11 BOOL  ; RK_06 U8_X 电池上下料X轴错误代码
2090.12 BOOL  ; RK_06 U8_X 电池上下料X轴错误代码
2090.13 BOOL  ; RK_06 U8_X 电池上下料X轴错误代码
2090.14 BOOL  ; RK_06 U8_X 电池上下料X轴错误代码
2090.15 BOOL  ; RK_06 U8_X 电池上下料X轴错误代码
2091.00 BOOL  ; RK_07 U8_Y 铝壳进料X轴Not Use
2091.01 BOOL  ; RK_07 U8_Y 铝壳进料X轴Not Use
2091.02 BOOL  ; RK_07 U8_Y 铝壳进料X轴Not Use
2091.03 BOOL  ; RK_07 U8_Y 铝壳进料X轴Not Use
2091.04 BOOL  ; RK_07 U8_Y 铝壳进料X轴等待存储器操作标志位
2091.05 BOOL  ; RK_07 U8_Y 铝壳进料X轴定位结束标志位
2091.06 BOOL  ; RK_07 U8_Y 铝壳进料X轴无原点标志位
2091.07 BOOL  ; RK_07 U8_Y 铝壳进料X轴原点停止标志位
2091.08 BOOL  ; RK_07 U8_Y 铝壳进料X轴区域0监控标志位
2091.09 BOOL  ; RK_07 U8_Y 铝壳进料X轴区域1监控标志位
2091.10 BOOL  ; RK_07 U8_Y 铝壳进料X轴区域2监控标志位
2091.11 BOOL  ; RK_07 U8_Y 铝壳进料X轴示教完成标志位
2091.12 BOOL  ; RK_07 U8_Y 铝壳进料X轴错误标志位
2091.13 BOOL  ; RK_07 U8_Y 铝壳进料X轴忙标志位
2091.14 BOOL  ; RK_07 U8_Y 铝壳进料X轴数据传送标志
2091.15 BOOL  ; RK_07 U8_Y 铝壳进料X轴减速停止执行标志
2092.00 BOOL  ; RK_07 U8_Y 铝壳进料X轴Not Use
2092.01 BOOL  ; RK_07 U8_Y 铝壳进料X轴Not Use
2092.02 BOOL  ; RK_07 U8_Y 铝壳进料X轴Not Use
2092.03 BOOL  ; RK_07 U8_Y 铝壳进料X轴Not Use
2092.04 BOOL  ; RK_07 U8_Y 铝壳进料X轴Not Use
2092.05 BOOL  ; RK_07 U8_Y 铝壳进料X轴Not Use
2092.06 BOOL  ; RK_07 U8_Y 铝壳进料X轴Not Use
2092.07 BOOL  ; RK_07 U8_Y 铝壳进料X轴Not Use
2092.08 BOOL  ; RK_07 U8_Y 铝壳进料X轴CW极限输入信号
2092.09 BOOL  ; RK_07 U8_Y 铝壳进料X轴CCW极限输入信号
2092.10 BOOL  ; RK_07 U8_Y 铝壳进料X轴原点接近输入信号
2092.11 BOOL  ; RK_07 U8_Y 铝壳进料X轴原点输入信号
2092.12 BOOL  ; RK_07 U8_Y 铝壳进料X轴中断输入信号
2092.13 BOOL  ; RK_07 U8_Y 铝壳进料X轴紧急停止输入信号
2092.14 BOOL  ; RK_07 U8_Y 铝壳进料X轴定位完成信号
2092.15 BOOL  ; $?St$Bk?_#[5046] / RK_07 U8_Y 铝壳进料X轴偏差计数器复位输出 / 原点调整命令输出$?St$Bk?_#[5046]
2093 CHANNEL  ; RK_07 U8_Y 铝壳进料X轴错误代码
2093.00 BOOL  ; RK_07 U8_Y 铝壳进料X轴错误代码
2093.01 BOOL  ; RK_07 U8_Y 铝壳进料X轴错误代码
2093.02 BOOL  ; RK_07 U8_Y 铝壳进料X轴错误代码
2093.03 BOOL  ; RK_07 U8_Y 铝壳进料X轴错误代码
2093.04 BOOL  ; RK_07 U8_Y 铝壳进料X轴错误代码
2093.05 BOOL  ; RK_07 U8_Y 铝壳进料X轴错误代码
2093.06 BOOL  ; RK_07 U8_Y 铝壳进料X轴错误代码
2093.07 BOOL  ; RK_07 U8_Y 铝壳进料X轴错误代码
2093.08 BOOL  ; RK_07 U8_Y 铝壳进料X轴错误代码
2093.09 BOOL  ; RK_07 U8_Y 铝壳进料X轴错误代码
2093.10 BOOL  ; RK_07 U8_Y 铝壳进料X轴错误代码
2093.11 BOOL  ; RK_07 U8_Y 铝壳进料X轴错误代码
2093.12 BOOL  ; RK_07 U8_Y 铝壳进料X轴错误代码
2093.13 BOOL  ; RK_07 U8_Y 铝壳进料X轴错误代码
2093.14 BOOL  ; RK_07 U8_Y 铝壳进料X轴错误代码
2093.15 BOOL  ; RK_07 U8_Y 铝壳进料X轴错误代码
2094.00 BOOL  ; RK_07 U8_Z 铝壳上料移载Y轴Not Use
2094.01 BOOL  ; RK_07 U8_Z 铝壳上料移载Y轴Not Use
2094.02 BOOL  ; RK_07 U8_Z 铝壳上料移载Y轴Not Use
2094.03 BOOL  ; RK_07 U8_Z 铝壳上料移载Y轴Not Use
2094.04 BOOL  ; RK_07 U8_Z 铝壳上料移载Y轴等待存储器操作标志位
2094.05 BOOL  ; RK_07 U8_Z 铝壳上料移载Y轴定位结束标志位
2094.06 BOOL  ; RK_07 U8_Z 铝壳上料移载Y轴无原点标志位
2094.07 BOOL  ; RK_07 U8_Z 铝壳上料移载Y轴原点停止标志位
2094.08 BOOL  ; RK_07 U8_Z 铝壳上料移载Y轴区域0监控标志位
2094.09 BOOL  ; RK_07 U8_Z 铝壳上料移载Y轴区域1监控标志位
2094.10 BOOL  ; RK_07 U8_Z 铝壳上料移载Y轴区域2监控标志位
2094.11 BOOL  ; RK_07 U8_Z 铝壳上料移载Y轴示教完成标志位
2094.12 BOOL  ; RK_07 U8_Z 铝壳上料移载Y轴错误标志位
2094.13 BOOL  ; RK_07 U8_Z 铝壳上料移载Y轴忙标志位
2094.14 BOOL  ; RK_07 U8_Z 铝壳上料移载Y轴数据传送标志
2094.15 BOOL  ; RK_07 U8_Z 铝壳上料移载Y轴减速停止执行标志
2095.00 BOOL  ; RK_07 U8_Z 铝壳上料移载Y轴Not Use
2095.01 BOOL  ; RK_07 U8_Z 铝壳上料移载Y轴Not Use
2095.02 BOOL  ; RK_07 U8_Z 铝壳上料移载Y轴Not Use
2095.03 BOOL  ; RK_07 U8_Z 铝壳上料移载Y轴Not Use
2095.04 BOOL  ; RK_07 U8_Z 铝壳上料移载Y轴Not Use
2095.05 BOOL  ; RK_07 U8_Z 铝壳上料移载Y轴Not Use
2095.06 BOOL  ; RK_07 U8_Z 铝壳上料移载Y轴Not Use
2095.07 BOOL  ; RK_07 U8_Z 铝壳上料移载Y轴Not Use
